D1100.10 BOOL  ; #2腔体机构关腔体氦检阀/关腔体抽气阀/关#2-1电池抽气阀（自动单检步）
D1100.11 BOOL  ; #2腔体机构关闭#2-1腔体阀/清氦判定（自动单检步）
D1100.12 BOOL  ; #2腔体机构打开#2-2腔体阀（自动单检步）
D1100.13 BOOL  ; #2腔体机构腔体抽气阀打开/延时开#2-2电池抽气阀（自动单检步）
D1100.14 BOOL  ; #2腔体机构关#2-2电池抽气阀（自动单检步）
D1100.15 BOOL  ; #2腔体机构开#2-2电池注氦阀（自动单检步）
D1101.00 BOOL  ; #2腔体机构关#2-2电池注氦阀（自动单检步）
D1101.01 BOOL  ; #2腔体机构（自动单检步）
D1101.02 BOOL  ; #2腔体机构开腔体氦检阀/延时关腔体抽气阀（自动单检步）
D1101.03 BOOL  ; #2腔体机构关腔体氦检阀（自动单检步）
D1101.04 BOOL  ; #2腔体机构开腔体#2-1阀（自动单检步）
D1101.05 BOOL  ; #2腔体机构开腔体抽真空阀/开电池抽真空阀（自动单检步）
D1101.06 BOOL  ; #2腔体机构关腔体抽真空阀/关电池抽真空阀（自动单检步）
D1101.07 BOOL  ; #2腔体机构清氦需求判定（自动单检步）
D1101.08 BOOL  ; #2腔体机构开腔体破真空阀/开电池破真空阀（自动单检步）
D1101.09 BOOL  ; #2腔体机构关腔体破真空阀/关电池破真空阀（自动单检步）
D1101.10 BOOL  ; #2腔体机构腔体顶升气缸下降（自动单检步）
D1101.11 BOOL  ; #2腔体机构腔体平移气缸到出料位（自动单检步）
D1101.12 BOOL  ; #2腔体机构腔体等待取料完成信号（自动单检步）
D1101.13 BOOL  ; #2腔体机构腔体平移气缸到上料位（自动单检步）
D1101.14 BOOL  ; #2腔体机构（自动单检步）
D1101.15 BOOL  ; #2腔体机构循环结束（自动单检步）
D1104 CHANNEL  ; #2腔体机构清氦步序号
D1104.00 BOOL  ; #2腔体机构自动开始（清氦步）
D1104.01 BOOL  ; #2腔体机构平移气缸到氦检位/数据初始化（清氦步）
D1104.02 BOOL  ; #2腔体机构腔体顶升气缸上升（清氦步）
D1104.03 BOOL  ; #2腔体机构氦检仪真空阀关闭（清氦步）
D1104.04 BOOL  ; #2腔体机构正压开腔体阀/负压关腔体阀/氦检阀打开
D1104.05 BOOL  ; #2腔体机构（清氦步）
D1104.06 BOOL  ; #2腔体机构腔体抽气阀打开/电池抽气阀打开（清氦步）
D1104.07 BOOL  ; #2腔体机构腔体抽气阀关闭/电池抽气阀关闭（清氦步）
D1104.08 BOOL  ; #2腔体机构（清氦步）
D1104.09 BOOL  ; #2腔体机构氦检清洁阀打开/电池破真空阀打开（清氦步）
D1104.10 BOOL  ; #2腔体机构氦检清洁阀关闭/电池破真空阀关闭（清氦步）
D1104.11 BOOL  ; #2腔体机构（清氦步）
D1104.12 BOOL  ; #2腔体机构清氦次数判定（清氦步）
D1104.13 BOOL  ; #2腔体机构（清氦步）
D1104.14 BOOL  ; #2腔体机构腔体抽气阀打开/电池抽气阀打开（清氦步）
D1104.15 BOOL  ; #2腔体机构关闭电池抽气阀（清氦步）
D1105.00 BOOL  ; #2腔体机构腔体氦检阀仪真空阀打开/延时关腔体抽气阀（清氦步）
D1105.01 BOOL  ; #2腔体机构（清氦步）
D1105.02 BOOL  ; #2腔体机构腔体氦检阀关闭（清氦步）
D1105.03 BOOL  ; #2腔体机构腔体抽气阀关闭/电池抽气阀关闭（清氦步）
D1105.04 BOOL  ; #2腔体机构是否需要重新清氦判定（清氦步）
D1105.05 BOOL  ; #2腔体机构（清氦步）
D1105.06 BOOL  ; #2腔体机构开腔体破真空阀/开电池破真空阀/开腔体阀（清氦步）
D1105.07 BOOL  ; #2腔体机构关腔体破真空阀/关电池破真空阀（清氦步）
D1105.08 BOOL  ; #2腔体机构（清氦步）
D1105.09 BOOL  ; #2腔体机构清氦完成标志（清氦步）
D1105.10 BOOL  ; #2腔体机构（清氦步）
D1105.11 BOOL  ; #2腔体机构腔体顶升气缸下降（清氦步）
D1105.12 BOOL  ; #2腔体机构腔体平移气缸到初始位（清氦步）
D1105.13 BOOL  ; #2腔体机构（清氦步）
D1105.14 BOOL  ; #2腔体机构（清氦步）
D1105.15 BOOL  ; #2腔体机构循环结束（清氦步）
D1107.00 BOOL  ; #2腔体机构复位（M）
D1107.01 BOOL  ; #2腔体关闭除破真空阀以外全部阀门（复位）
D1107.02 BOOL  ; #2腔体打开腔体阀门（复位）
D1107.03 BOOL  ; #2腔体破真空值未到达开破真空阀（复位）
D1107.04 BOOL  ; #2腔体破真空值到达关破真空阀（复位）
D1107.05 BOOL  ; #2腔体腔体顶升气缸下降（复位）
D1107.06 BOOL  ; #2腔体腔体平移气缸伸出（复位）
D1115.00 BOOL  ; #2腔体抽气阀打开允许（自检）
D1115.01 BOOL  ; #2腔体抽气阀打开需求（自检）
D1115.02 BOOL  ; #2腔体平移气缸在初始位（自检）
D1115.03 BOOL  ; #2腔体平移气缸在氦检位（自检）
D1115.04 BOOL  ; #2腔体真空泵开（自检）
D1115.05 BOOL  ; #2腔体平移气缸到初始位（自检）
D1115.06 BOOL  ; #2腔体平移气缸到氦检位（自检）
D1115.07 BOOL  ; #2腔体顶升气缸下降（自检）
D1115.08 BOOL  ; #2腔体顶升气缸上升（自检）
D1115.09 BOOL  ; #2腔体开抽真空阀（自检）
D1115.10 BOOL  ; #2腔体关抽真空阀（自检）
D1115.11 BOOL  ; #2腔体开破真空阀（自检）
D1115.12 BOOL  ; #2腔体关破真空阀（自检）
D1115.13 BOOL  ; #2腔体破真空阀状态（自检）
D1115.14 BOOL  ; #2腔体抽真空阀状态（自检）
D1117.00 BOOL  ; #2腔体机构标漏运行条件
D1117.01 BOOL  ; #2腔体机构标漏开始运行条件
D1117.02 BOOL  ; #2腔体机构标漏步进条件
D1117.15 BOOL  ; #2腔体机构标漏步进
D1118 CHANNEL  ; #2腔体标漏步序号
D1118.00 BOOL  ; #2腔体机构自动开始（标漏步）
D1118.01 BOOL  ; #2腔体机构（标漏步）
D1118.02 BOOL  ; #2腔体机构（标漏步）
D1118.03 BOOL  ; #2腔体机构（标漏步）
D1118.04 BOOL  ; #2腔体机构（标漏步）
D1118.05 BOOL  ; #2腔体机构（标漏步）
D1118.06 BOOL  ; #2腔体机构（标漏步）
D1118.07 BOOL  ; #2腔体机构开#2-1腔体阀（标漏步）
D1118.08 BOOL  ; #2腔体机构开#2腔抽气阀（标漏步）
D1118.09 BOOL  ; #2腔体机构关#2腔体抽气阀（标漏步）
D1118.10 BOOL  ; #2腔体机构（标漏步）
D1118.11 BOOL  ; #2腔体机构（标漏步）
D1118.12 BOOL  ; #2腔体机构开始#2-1氦检（标漏步）
D1118.13 BOOL  ; #2腔体机构关#2腔体氦检阀（标漏步）
D1118.14 BOOL  ; #2腔体机构关#2-1腔体阀（标漏步）
D1118.15 BOOL  ; #2腔体机构开#2-2腔体阀（标漏步）
D1119.00 BOOL  ; #2腔体机构开#2腔抽真空阀（标漏步）
D1119.01 BOOL  ; #2腔体机构关#2腔抽真空阀（标漏步）
D1119.02 BOOL  ; #2腔体机构（标漏步）
D1119.03 BOOL  ; #2腔体机构（标漏步）
D1119.04 BOOL  ; #2腔体机构开始#2-2氦检（标漏步）
D1119.05 BOOL  ; #2腔体机构关#2腔体氦检阀（标漏步）
D1119.06 BOOL  ; #2腔体机构关#2-2腔体阀（标漏步）
D1119.07 BOOL  ; #2腔体机构（标漏步）
D1119.08 BOOL  ; #2腔体机构（标漏步）
D1119.09 BOOL  ; #2腔体机构（标漏步）
D1119.10 BOOL  ; #2腔体机构（标漏步）
D1119.11 BOOL  ; #2腔体机构（标漏步）
D1119.12 BOOL  ; #2腔体机构（标漏步）
D1119.13 BOOL  ; #2腔体机构（标漏步）
D1119.14 BOOL  ; #2腔体机构跳转至#3腔标漏步（标漏步）
D1119.15 BOOL  ; #2腔体机构循环结束（标漏步）
D112 CHANNEL  ; 泄漏率（Pa.m3/s_Float）
D1120.00 BOOL  ; #3氦检机构初始位
D1120.05 BOOL  ; #3氦检机构停止标志
D1120.06 BOOL  ; #3氦检机构清料完成标志
D1120.07 BOOL  ; #3腔体机构异常标志
D1121.00 BOOL  ; #3腔体机构运行条件（自动步）
D1121.01 BOOL  ; #3腔体机构运行条件（自动单检步）
D1121.02 BOOL  ; #3腔体机构运行条件（清氦步）
D1122.00 BOOL  ; #3腔体机构平移气缸安全移动条件
D1122.12 BOOL  ; #3腔体机构腔体抽真空需求（测试）
D1122.13 BOOL  ; #3腔体机构正常清氦需求（正压测试）
D1122.14 BOOL  ; #3腔体氦检阀打开允许条件
D1122.15 BOOL  ; #3腔体机构腔体抽气阀打开允许
D1123.00 BOOL  ; #3腔体机构单步/自动循环运行中（总）
D1123.10 BOOL  ; $?St$Bk?_#[183] / #3腔体机构记忆清除(SW) / $?St$Bk?_#[183]
D1123.12 BOOL  ; #3腔体自检启动(SW)
D1123.13 BOOL  ; #3腔体自检停止(SW)
D1123.14 BOOL  ; #3腔体机构复位按钮（SW）
D1123.15 BOOL  ; #3腔体机构单步（SW）
D1124.00 BOOL  ; #3腔体机构单步运行中
D1124.01 BOOL  ; #3腔体机构单步/自动循环运行中（自动步）
D1124.02 BOOL  ; #3腔体机构自动循环运行中（自动单检步）
D1124.03 BOOL  ; #3腔体机构自动循环运行中（清氦步）
D1124.04 BOOL  ; #3-1腔体单腔自检(SW)
D1124.05 BOOL  ; #3-2腔体单腔自检(SW)
D1124.06 BOOL  ; #3腔体自检运行中
D1125.00 BOOL  ; #3腔体机构开始运行条件（自动步）
D1125.01 BOOL  ; #3腔体机构步进条件（自动步）
D1125.02 BOOL  ; #3腔体机构开始运行条件（自动单检步）
D1125.03 BOOL  ; #3腔体机构步进条件（自动单检步）
D1125.04 BOOL  ; #3腔体机构开始运行条件（清氦步）
D1125.05 BOOL  ; #3腔体机构步进条件（清氦步）
D1125.13 BOOL  ; #3腔体机构步进（清氦步）
D1125.14 BOOL  ; #3腔体机构步进（自动单检步）
D1125.15 BOOL  ; #3腔体机构步进（自动步）
D1126 CHANNEL  ; #3腔体机构自动步序号
D1126.00 BOOL  ; #3腔体机构自动开始（自动步）
D1126.01 BOOL  ; #3腔体机构平移气缸到氦检位/数据初始化（自动步）
D1126.02 BOOL  ; #3腔体机构腔体顶升气缸上升（自动步）
D1126.03 BOOL  ; #3腔体机构等待氦检阀打开条件及腔体抽气阀打开条件/开腔体阀（自动步）
D1126.04 BOOL  ; #3腔体机构（自动步）
D1126.05 BOOL  ; #3腔体机构腔体抽气阀打开/延时开电池抽气阀（自动步）
D1126.06 BOOL  ; #3腔体机构关电池抽气阀（自动步）
D1126.07 BOOL  ; #3腔体机构开电池注氦阀（自动步）
D1126.08 BOOL  ; #3腔体机构关电池注氦阀（自动步）
D1126.09 BOOL  ; #3腔体机构（自动步）
D1126.10 BOOL  ; #3腔体机构开腔体氦检阀/延时关腔体抽气阀（自动步）
D1126.11 BOOL  ; #3腔体机构（自动步）
D1126.12 BOOL  ; #3腔体机构关腔体氦检阀（自动步）
D1126.13 BOOL  ; #3腔体机构（自动步）
D1126.14 BOOL  ; #3腔体机构开腔体#3-1腔体阀/开腔体#3-2腔体阀（自动步）
D1126.15 BOOL  ; #3腔体机构开腔体抽真空阀/开电池抽真空阀（自动步）
D1127.00 BOOL  ; #3腔体机构关腔体抽真空阀/关电池抽真空阀/开腔体阀（自动步）
D1127.01 BOOL  ; #3腔体机构清氦需求判定（自动步）
D1127.02 BOOL  ; #3腔体机构开腔体破真空阀/开电池破真空阀（自动步）
D1127.03 BOOL  ; #3腔体机构关腔体破真空阀/关电池破真空阀（自动步）
D1127.04 BOOL  ; #3腔体机构复测需求判定（自动步）
D1127.05 BOOL  ; #3腔体机构（自动步）
D1127.06 BOOL  ; #3腔体机构腔体顶升气缸下降（自动步）
D1127.07 BOOL  ; #3腔体机构（自动步）
D1127.08 BOOL  ; #3腔体机构腔体平移气缸到出料位（自动步）
D1127.09 BOOL  ; #3腔体机构腔体等待取料完成信号（自动步）
D1127.10 BOOL  ; #3腔体机构（自动步）
D1127.11 BOOL  ; #3腔体机构平移气缸到上料位（自动步）
D1127.12 BOOL  ; #3腔体机构（自动步）
D1127.13 BOOL  ; #3腔体机构（自动步）
D1127.14 BOOL  ; #3腔体机构（自动步）
D1127.15 BOOL  ; #3腔体机构循环结束（自动步）
D1130 CHANNEL  ; #3腔体机构单检步序号
D1130.00 BOOL  ; #3腔体机构自动开始（自动单检步）
D1130.01 BOOL  ; #3腔体机构平移气缸到氦检位/数据初始化（自动单检步）
D1130.02 BOOL  ; #3腔体机构腔体顶升气缸上升（自动单检步）
D1130.03 BOOL  ; #3腔体机构关闭#3-2腔体阀（自动单检步）
D1130.04 BOOL  ; #3腔体机构腔体抽气阀打开/延时开#3-1电池抽气阀（自动单检步）
D1130.05 BOOL  ; #3腔体机构关#3-1电池抽气阀（自动单检步）
D1130.06 BOOL  ; #3腔体机构开#3-1电池注氦阀（自动单检步）
D1130.07 BOOL  ; #3腔体机构关#3-1电池注氦阀（自动单检步）
D1130.08 BOOL  ; #3腔体机构（自动单检步）
D1130.09 BOOL  ; #3腔体机构开腔体氦检阀/延时关腔体抽气阀（自动单检步）
D1130.10 BOOL  ; #3腔体机构关腔体氦检阀/关腔体抽气阀/关#3-1电池抽气阀（自动单检步）
D1130.11 BOOL  ; #3腔体机构关闭#3-1腔体阀/清氦判定（自动单检步）
D1130.12 BOOL  ; #3腔体机构打开#3-2腔体阀（自动单检步）
D1130.13 BOOL  ; #3腔体机构腔体抽气阀打开/延时开#3-2电池抽气阀（自动单检步）
D1130.14 BOOL  ; #3腔体机构关#3-2电池抽气阀（自动单检步）
D1130.15 BOOL  ; #3腔体机构开#3-2电池注氦阀（自动单检步）
D1131.00 BOOL  ; #3腔体机构关#3-2电池注氦阀（自动单检步）
D1131.01 BOOL  ; #3腔体机构（自动单检步）
D1131.02 BOOL  ; #3腔体机构开腔体氦检阀/延时关腔体抽气阀（自动单检步）
D1131.03 BOOL  ; #3腔体机构关腔体氦检阀（自动单检步）
D1131.04 BOOL  ; #3腔体机构开腔体#3-1阀（自动单检步）
D1131.05 BOOL  ; #3腔体机构开腔体抽真空阀/开电池抽真空阀（自动单检步）
D1131.06 BOOL  ; #3腔体机构关腔体抽真空阀/关电池抽真空阀（自动单检步）
D1131.07 BOOL  ; #3腔体机构清氦需求判定（自动单检步）
D1131.08 BOOL  ; #3腔体机构开腔体破真空阀/开电池破真空阀（自动单检步）
D1131.09 BOOL  ; #3腔体机构关腔体破真空阀/关电池破真空阀（自动单检步）
D1131.10 BOOL  ; #3腔体机构腔体顶升气缸下降（自动单检步）
D1131.11 BOOL  ; #3腔体机构腔体平移气缸到出料位（自动单检步）
D1131.12 BOOL  ; #3腔体机构腔体等待取料完成信号（自动单检步）
D1131.13 BOOL  ; #3腔体机构腔体平移气缸到上料位（自动单检步）
D1131.14 BOOL  ; #3腔体机构（自动单检步）
D1131.15 BOOL  ; #3腔体机构循环结束（自动单检步）
D1134 CHANNEL  ; #3腔体机构清氦步序号
D1134.00 BOOL  ; #3腔体机构自动开始（清氦步）
D1134.01 BOOL  ; #3腔体机构平移气缸到氦检位/数据初始化（清氦步）
D1134.02 BOOL  ; #3腔体机构腔体顶升气缸上升（清氦步）
D1134.03 BOOL  ; #3腔体机构氦检仪真空阀关闭（清氦步）
D1134.04 BOOL  ; #3腔体机构正压开腔体阀/负压关腔体阀/氦检阀打开
D1134.05 BOOL  ; #3腔体机构（清氦步）
D1134.06 BOOL  ; #3腔体机构腔体抽气阀打开/电池抽气阀打开（清氦步）
D1134.07 BOOL  ; #3腔体机构腔体抽气阀关闭/电池抽气阀关闭（清氦步）
D1134.08 BOOL  ; #3腔体机构（清氦步）
D1134.09 BOOL  ; #3腔体机构氦检清洁阀打开/电池破真空阀打开（清氦步）
D1134.10 BOOL  ; #3腔体机构氦检清洁阀关闭/电池破真空阀关闭（清氦步）
D1134.11 BOOL  ; #3腔体机构（清氦步）
D1134.12 BOOL  ; #3腔体机构清氦次数判定（清氦步）
D1134.13 BOOL  ; #3腔体机构（清氦步）
D1134.14 BOOL  ; #3腔体机构腔体抽气阀打开/电池抽气阀打开（清氦步）
D1134.15 BOOL  ; #3腔体机构关闭电池抽气阀（清氦步）
D1135.00 BOOL  ; #3腔体机构腔体氦检阀仪真空阀打开/延时关腔体抽气阀（清氦步）
D1135.01 BOOL  ; #3腔体机构（清氦步）
D1135.02 BOOL  ; #3腔体机构腔体氦检阀关闭（清氦步）
D1135.03 BOOL  ; #3腔体机构腔体抽气阀关闭/电池抽气阀关闭（清氦步）
D1135.04 BOOL  ; #3腔体机构是否需要重新清氦判定（清氦步）
D1135.05 BOOL  ; #3腔体机构（清氦步）
D1135.06 BOOL  ; #3腔体机构开腔体破真空阀/开电池破真空阀/开腔体阀（清氦步）
D1135.07 BOOL  ; #3腔体机构关腔体破真空阀/关电池破真空阀（清氦步）
D1135.08 BOOL  ; #3腔体机构（清氦步）
D1135.09 BOOL  ; #3腔体机构清氦完成标志（清氦步）
D1135.10 BOOL  ; #3腔体机构（清氦步）
D1135.11 BOOL  ; #3腔体机构腔体顶升气缸下降（清氦步）
D1135.12 BOOL  ; #3腔体机构腔体平移气缸到初始位（清氦步）
D1135.13 BOOL  ; #3腔体机构（清氦步）
D1135.14 BOOL  ; #3腔体机构（清氦步）
D1135.15 BOOL  ; #3腔体机构循环结束（清氦步）
D1137.00 BOOL  ; #3腔体机构复位（M）
D1137.01 BOOL  ; #3腔体关闭除破真空阀以外全部阀门（复位）
D1137.02 BOOL  ; #3腔体打开腔体阀门（复位）
D1137.03 BOOL  ; #3腔体破真空值未到达开破真空阀（复位）
D1137.04 BOOL  ; #3腔体破真空值到达关破真空阀（复位）
D1137.05 BOOL  ; #3腔体腔体顶升气缸下降（复位）
D1137.06 BOOL  ; #3腔体腔体平移气缸伸出（复位）
D114 CHANNEL  ; 泄漏率（Pa.m3/s_Float_指数）
D1143.00 BOOL  ; 进料机械手执行清料动作
D1145.00 BOOL  ; #3腔体抽气阀打开允许（自检）
D1145.01 BOOL  ; #3腔体抽气阀打开需求（自检）
D1145.02 BOOL  ; #3腔体平移气缸在初始位（自检）
D1145.03 BOOL  ; #3腔体平移气缸在氦检位（自检）
D1145.04 BOOL  ; #3腔体真空泵开（自检）
D1145.05 BOOL  ; #3腔体平移气缸到初始位（自检）
D1145.06 BOOL  ; #3腔体平移气缸到氦检位（自检）
D1145.07 BOOL  ; #3腔体顶升气缸下降（自检）
D1145.08 BOOL  ; #3腔体顶升气缸上升（自检）
D1145.09 BOOL  ; #3腔体开抽真空阀（自检）
D1145.10 BOOL  ; #3腔体关抽真空阀（自检）
D1145.11 BOOL  ; #3腔体开破真空阀（自检）
D1145.12 BOOL  ; #3腔体关破真空阀（自检）
D1145.13 BOOL  ; #3腔体破真空阀状态（自检）
D1145.14 BOOL  ; #3腔体抽真空阀状态（自检）
D1147.00 BOOL  ; #3腔体机构标漏运行条件
D1147.01 BOOL  ; #3腔体机构标漏开始运行条件
D1147.02 BOOL  ; #3腔体机构标漏步进条件
D1147.15 BOOL  ; #3腔体机构标漏步进
D1148 CHANNEL  ; #3腔体标漏步序号
D1148.00 BOOL  ; #3腔体机构自动开始（标漏步）
D1148.01 BOOL  ; #3腔体机构（标漏步）
D1148.02 BOOL  ; #3腔体机构（标漏步）
D1148.03 BOOL  ; #3腔体机构（标漏步）
D1148.04 BOOL  ; #3腔体机构（标漏步）
D1148.05 BOOL  ; #3腔体机构（标漏步）
D1148.06 BOOL  ; #3腔体机构（标漏步）
D1148.07 BOOL  ; #3腔体机构开#3-1腔体阀（标漏步）
D1148.08 BOOL  ; #3腔体机构开#3腔抽气阀（标漏步）
D1148.09 BOOL  ; #3腔体机构关#3腔体抽气阀（标漏步）
D1148.10 BOOL  ; #3腔体机构（标漏步）
D1148.11 BOOL  ; #3腔体机构（标漏步）
D1148.12 BOOL  ; #3腔体机构开始#3-1氦检（标漏步）
D1148.13 BOOL  ; #3腔体机构关#3腔体氦检阀（标漏步）
D1148.14 BOOL  ; #3腔体机构关#3-1腔体阀（标漏步）
D1148.15 BOOL  ; #3腔体机构开#3-2腔体阀（标漏步）
D1149.00 BOOL  ; #3腔体机构开#3腔抽真空阀（标漏步）
D1149.01 BOOL  ; #3腔体机构关#3腔抽真空阀（标漏步）
D1149.02 BOOL  ; #3腔体机构（标漏步）
D1149.03 BOOL  ; #3腔体机构（标漏步）
D1149.04 BOOL  ; #3腔体机构开始#3-2氦检（标漏步）
D1149.05 BOOL  ; #3腔体机构关#3腔体氦检阀（标漏步）
D1149.06 BOOL  ; #3腔体机构关#3-2腔体阀（标漏步）
D1149.07 BOOL  ; #3腔体机构开所有腔体总阀（标漏步）
D1149.08 BOOL  ; #3腔体机构开所有腔体破真空阀（标漏步）
D1149.09 BOOL  ; #3腔体机构关所有腔体破真空阀（标漏步）
D1149.10 BOOL  ; #3腔体机构所有顶升气缸下降（标漏步）
D1149.11 BOOL  ; #3腔体机构所有腔体平移气缸回初始位（标漏步）
D1149.12 BOOL  ; #3腔体机构关标漏阀（标漏步）
D1149.13 BOOL  ; #3腔体机构（标漏步）
D1149.14 BOOL  ; #3腔体机构（标漏步）
D1149.15 BOOL  ; #3腔体机构循环结束（标漏步）
D1150.00 BOOL  ; 出料伺服机构初始位
D1150.05 BOOL  ; 出料伺服机构停止标志
D1150.06 BOOL  ; 出料伺服机构清料完成标志
D1150.07 BOOL  ; 出料伺服机构异常标志
D1153.00 BOOL  ; 出料机械手执行清料动作
D1153.10 BOOL  ; 下料夹爪有料记忆清除（SW）
D1153.14 BOOL  ; 出料伺服机构复位按钮（SW）
D1156 CHANNEL  ; 下料模组自动流程
D1156.00 BOOL  ; 下料模组运行前检测
D1156.01 BOOL  ; 下料模组运行备用
D1156.02 BOOL  ; 下料x模组运行到对应下料位
D1156.03 BOOL  ; 下料Z模组运行前检测
D1156.04 BOOL  ; 下料Z模组运行
D1156.05 BOOL  ; 下料模组夹爪夹紧
D1156.06 BOOL  ; 下料模组运行备用
D1156.07 BOOL  ; 下料Z模组到待机位
D1156.08 BOOL  ; 等待数据校验完成
D1156.09 BOOL  ; 下料模组是否放全OK料检测
D1156.10 BOOL  ; 下料X模组到OK下料位
D1156.11 BOOL  ; 下料Z模组OK下降检测
D1156.12 BOOL  ; 下料Z模组到OK下料位
D1156.13 BOOL  ; 下料模组放全OK料开夹爪
D1156.14 BOOL  ; 下料Z模组到待机位
D1156.15 BOOL  ; *下料模组去腔体取料流程&全OK下料结束
D1158 CHANNEL  ; 下料模组全NG流程
D1158.00 BOOL  ; 下料模组全OK/NG料流程准备
D1158.01 BOOL  ; 下料模组放NG料：预留
D1158.02 BOOL  ; 下料模组放NG：预留
D1158.03 BOOL  ; 下料模组放NG料：出料X轴到NG缓存位/变距气缸缩回
D1158.04 BOOL  ; 预留
D1158.05 BOOL  ; 预留
D1158.06 BOOL  ; 预留
D1158.07 BOOL  ; 预留
D1158.08 BOOL  ; 下料模组放1#NG Z轴下降
D1158.09 BOOL  ; 下料模组开夹爪放NG料
D1158.10 BOOL  ; 下料Z模组放完1#NG回待机位
D1158.11 BOOL  ; 下料模组放双NG:放NG料完成，有腔体测试完成直接跳过，无腔体测试完成X轴返回待机位
D1158.12 BOOL  ; 下料模组放双NG备用
D1158.13 BOOL  ; 下料模组放双NG备用
D1158.14 BOOL  ; 下料模组放双NG备用
D1158.15 BOOL  ; 下料模组放双NG结束
D116 CHANNEL  ; 检漏口压力（Pa_Float）
D1160 CHANNEL  ; 下料模组（取）放1OK/1NG流程
D1160.00 BOOL  ; *下料模组（取）放1OK/1NG流程运行前检测
D1160.01 BOOL  ; 下料X模组到达对应X位置
D1160.02 BOOL  ; 下料Z模组下降前检测
D1160.03 BOOL  ; 下料Z模组下降放NG料
D1160.04 BOOL  ; 下料模组开NG夹爪
D1160.05 BOOL  ; 下料Z模组放完NG回待机位
D1160.06 BOOL  ; 下料模组放缓存OR取缓存
D1160.07 BOOL  ; 下料X模组到放缓存位
D1160.08 BOOL  ; 下料Z模组下降放缓存
D1160.09 BOOL  ; 下料模组放缓存开夹爪or夹紧
D1160.10 BOOL  ; 下料模组缓存有料检测
D1160.11 BOOL  ; 下料Z模组到待机位
D1160.12 BOOL  ; *下料模组（取）放1OK/1NG X轴到OK下料位
D1160.13 BOOL  ; *下料模组（取）放1OK/1NG流程备用
D1160.14 BOOL  ; *下料模组（取）放1OK/1NG流程备用
D1160.15 BOOL  ; *下料模组（取）放1OK/1NG流程结束
D1166 CHANNEL  ; 下料模组X/Z初始化
D1166.00 BOOL  ; 下料模组初始化准备
D1166.01 BOOL  ; 下料Z模组初始化
D1166.02 BOOL  ; 下料Z模组到待机位
D1166.03 BOOL  ; 下料X模组初始化
D1166.04 BOOL  ; 下料X模组到待机位
D1166.05 BOOL  ; 下料模组运行许可
D1166.06 BOOL  ; 下料模组初始化结束
D1168 CHANNEL  ; 下料模组手动跟踪联动
D1168.00 BOOL  ; 下料模组手动跟踪Z回待机位
D1168.01 BOOL  ; 下料模组手动跟踪X到对应位置
D1168.02 BOOL  ; 下料Z轴手动下降前安全判定
D1168.03 BOOL  ; 下料Z模组手动下降
D1168.04 BOOL  ; 下料X/Z模组跟踪联动需求清除
D1168.05 BOOL  ; 下料X/Z模组手动联动结束
D1170.00 BOOL  ; #4氦检机构初始位
D1170.05 BOOL  ; #4氦检机构停止标志
D1170.06 BOOL  ; #4氦检机构清料完成标志
D1170.07 BOOL  ; #4腔体机构异常标志
D1171.00 BOOL  ; #4腔体机构运行条件（自动步）
D1171.01 BOOL  ; #4腔体机构运行条件（自动单检步）
D1171.02 BOOL  ; #4腔体机构运行条件（清氦步）
D1172.00 BOOL  ; #4腔体机构平移气缸安全移动条件
D1172.12 BOOL  ; #4腔体机构腔体抽真空需求（测试）
D1172.13 BOOL  ; #4腔体机构正常清氦需求（正压测试）
D1172.14 BOOL  ; #4腔体氦检阀打开允许条件
D1172.15 BOOL  ; #4腔体机构腔体抽气阀打开允许
D1173.00 BOOL  ; #4腔体机构单步/自动循环运行中（总）
D1173.10 BOOL  ; #4腔体机构记忆清除(SW)
D1173.11 BOOL  ; #4腔体标漏(SW)
D1173.12 BOOL  ; #4腔体自检启动(SW)
D1173.13 BOOL  ; #4腔体自检停止(SW)
D1173.14 BOOL  ; #4腔体机构复位按钮（SW）
D1173.15 BOOL  ; #4腔体机构单步（SW）
D1174.00 BOOL  ; #4腔体机构单步运行中
D1174.01 BOOL  ; #4腔体机构单步/自动循环运行中（自动步）
D1174.02 BOOL  ; #4腔体机构自动循环运行中（自动单检步）
D1174.03 BOOL  ; #4腔体机构自动循环运行中（清氦步）
D1174.04 BOOL  ; #4-1腔体单腔自检(SW)
D1174.05 BOOL  ; #4-2腔体单腔自检(SW)
D1174.06 BOOL  ; #4腔体自检运行中
D1174.10 BOOL  ; #4腔体机构单步运行条件
D1175.00 BOOL  ; #4腔体机构开始运行条件（自动步）
D1175.01 BOOL  ; #4腔体机构步进条件（自动步）
D1175.02 BOOL  ; #4腔体机构开始运行条件（自动单检步）
D1175.03 BOOL  ; #4腔体机构步进条件（自动单检步）
D1175.04 BOOL  ; #4腔体机构开始运行条件（清氦步）
D1175.05 BOOL  ; #4腔体机构步进条件（清氦步）
D1175.13 BOOL  ; #4腔体机构步进（清氦步）
D1175.14 BOOL  ; #4腔体机构步进（自动单检步）
D1175.15 BOOL  ; #4腔体机构步进（自动步）
D1176 CHANNEL  ; #4腔体机构自动步序号
D1176.00 BOOL  ; #4腔体机构自动开始（自动步）
D1176.01 BOOL  ; #4腔体机构平移气缸到氦检位/数据初始化（自动步）
D1176.02 BOOL  ; #4腔体机构腔体顶升气缸上升（自动步）
D1176.03 BOOL  ; #4腔体机构等待氦检阀打开条件及腔体抽气阀打开条件/开腔体阀（自动步）
D1176.04 BOOL  ; #4腔体机构（自动步）
D1176.05 BOOL  ; #4腔体机构腔体抽气阀打开/延时开电池抽气阀（自动步）
D1176.06 BOOL  ; #4腔体机构关电池抽气阀（自动步）
D1176.07 BOOL  ; #4腔体机构开电池注氦阀（自动步）
D1176.08 BOOL  ; #4腔体机构关电池注氦阀（自动步）
D1176.09 BOOL  ; #4腔体机构（自动步）
D1176.10 BOOL  ; #4腔体机构开腔体氦检阀/延时关腔体抽气阀（自动步）
D1176.11 BOOL  ; #4腔体机构（自动步）
D1176.12 BOOL  ; #4腔体机构关腔体氦检阀（自动步）
D1176.13 BOOL  ; #4腔体机构（自动步）
D1176.14 BOOL  ; #4腔体机构开腔体#4-1腔体阀/开腔体#4-2腔体阀（自动步）
D1176.15 BOOL  ; #4腔体机构开腔体抽真空阀/开电池抽真空阀（自动步）
D1177.00 BOOL  ; #4腔体机构关腔体抽真空阀/关电池抽真空阀/开腔体阀（自动步）
D1177.01 BOOL  ; #4腔体机构清氦需求判定（自动步）
D1177.02 BOOL  ; #4腔体机构开腔体破真空阀/开电池破真空阀（自动步）
D1177.03 BOOL  ; #4腔体机构关腔体破真空阀/关电池破真空阀（自动步）
D1177.04 BOOL  ; #4腔体机构复测需求判定（自动步）
D1177.05 BOOL  ; #4腔体机构（自动步）
D1177.06 BOOL  ; #4腔体机构腔体顶升气缸下降（自动步）
D1177.07 BOOL  ; #4腔体机构（自动步）
D1177.08 BOOL  ; #4腔体机构腔体平移气缸到出料位（自动步）
D1177.09 BOOL  ; #4腔体机构腔体等待取料完成信号（自动步）
D1177.10 BOOL  ; #4腔体机构（自动步）
D1177.11 BOOL  ; #4腔体机构平移气缸到上料位（自动步）
D1177.12 BOOL  ; #4腔体机构（自动步）
D1177.13 BOOL  ; #4腔体机构（自动步）
D1177.14 BOOL  ; #4腔体机构（自动步）
D1177.15 BOOL  ; #4腔体机构循环结束（自动步）
D118 CHANNEL  ; 检漏口压力（Pa_Float_指数）
D1180 CHANNEL  ; #4腔体机构单检步序号
D1180.00 BOOL  ; #4腔体机构自动开始（自动单检步）
D1180.01 BOOL  ; #4腔体机构平移气缸到氦检位/数据初始化（自动单检步）
D1180.02 BOOL  ; #4腔体机构腔体顶升气缸上升（自动单检步）
D1180.03 BOOL  ; #4腔体机构关闭#4-2腔体阀（自动单检步）
D1180.04 BOOL  ; #4腔体机构腔体抽气阀打开/延时开#4-1电池抽气阀（自动单检步）
D1180.05 BOOL  ; #4腔体机构关#4-1电池抽气阀（自动单检步）
D1180.06 BOOL  ; #4腔体机构开#4-1电池注氦阀（自动单检步）
D1180.07 BOOL  ; #4腔体机构关#4-1电池注氦阀（自动单检步）
D1180.08 BOOL  ; #4腔体机构（自动单检步）
D1180.09 BOOL  ; #4腔体机构开腔体氦检阀/延时关腔体抽气阀（自动单检步）
D1180.10 BOOL  ; #4腔体机构关腔体氦检阀/关腔体抽气阀/关#4-1电池抽气阀（自动单检步）
D1180.11 BOOL  ; #4腔体机构关闭#4-1腔体阀/清氦判定（自动单检步）
D1180.12 BOOL  ; #4腔体机构打开#4-2腔体阀（自动单检步）
D1180.13 BOOL  ; #4腔体机构腔体抽气阀打开/延时开#4-2电池抽气阀（自动单检步）
D1180.14 BOOL  ; #4腔体机构关#4-2电池抽气阀（自动单检步）
D1180.15 BOOL  ; #4腔体机构开#4-2电池注氦阀（自动单检步）
D1181.00 BOOL  ; #4腔体机构关#4-2电池注氦阀（自动单检步）
D1181.01 BOOL  ; #4腔体机构（自动单检步）
D1181.02 BOOL  ; #4腔体机构开腔体氦检阀/延时关腔体抽气阀（自动单检步）
D1181.03 BOOL  ; #4腔体机构关腔体氦检阀（自动单检步）
D1181.04 BOOL  ; #4腔体机构开腔体#4-1阀（自动单检步）
D1181.05 BOOL  ; #4腔体机构开腔体抽真空阀/开电池抽真空阀（自动单检步）
D1181.06 BOOL  ; #4腔体机构关腔体抽真空阀/关电池抽真空阀（自动单检步）
D1181.07 BOOL  ; #4腔体机构清氦需求判定（自动单检步）
D1181.08 BOOL  ; #4腔体机构开腔体破真空阀/开电池破真空阀（自动单检步）
D1181.09 BOOL  ; #4腔体机构关腔体破真空阀/关电池破真空阀（自动单检步）
D1181.10 BOOL  ; #4腔体机构腔体顶升气缸下降（自动单检步）
D1181.11 BOOL  ; #4腔体机构腔体平移气缸到出料位（自动单检步）
D1181.12 BOOL  ; #4腔体机构腔体等待取料完成信号（自动单检步）
D1181.13 BOOL  ; #4腔体机构腔体平移气缸到上料位（自动单检步）
D1181.14 BOOL  ; #4腔体机构（自动单检步）
D1181.15 BOOL  ; #4腔体机构循环结束（自动单检步）
D1184 CHANNEL  ; #4腔体机构清氦步序号
D1184.00 BOOL  ; #4腔体机构自动开始（清氦步）
D1184.01 BOOL  ; #4腔体机构平移气缸到氦检位/数据初始化（清氦步）
D1184.02 BOOL  ; #4腔体机构腔体顶升气缸上升（清氦步）
D1184.03 BOOL  ; #4腔体机构氦检仪真空阀关闭（清氦步）
D1184.04 BOOL  ; #4腔体机构正压开腔体阀/负压关腔体阀/氦检阀打开
D1184.05 BOOL  ; #4腔体机构（清氦步）
D1184.06 BOOL  ; #4腔体机构腔体抽气阀打开/电池抽气阀打开（清氦步）
D1184.07 BOOL  ; #4腔体机构腔体抽气阀关闭/电池抽气阀关闭（清氦步）
D1184.08 BOOL  ; #4腔体机构（清氦步）
D1184.09 BOOL  ; #4腔体机构氦检清洁阀打开/电池破真空阀打开（清氦步）
D1184.10 BOOL  ; #4腔体机构氦检清洁阀关闭/电池破真空阀关闭（清氦步）
D1184.11 BOOL  ; #4腔体机构（清氦步）
D1184.12 BOOL  ; #4腔体机构清氦次数判定（清氦步）
D1184.13 BOOL  ; #4腔体机构（清氦步）
D1184.14 BOOL  ; #4腔体机构腔体抽气阀打开/电池抽气阀打开（清氦步）
D1184.15 BOOL  ; #4腔体机构关闭电池抽气阀（清氦步）
D1185.00 BOOL  ; #4腔体机构腔体氦检阀仪真空阀打开/延时关腔体抽气阀（清氦步）
D1185.01 BOOL  ; #4腔体机构（清氦步）
D1185.02 BOOL  ; #4腔体机构腔体氦检阀关闭（清氦步）
D1185.03 BOOL  ; #4腔体机构腔体抽气阀关闭/电池抽气阀关闭（清氦步）
D1185.04 BOOL  ; #4腔体机构是否需要重新清氦判定（清氦步）
D1185.05 BOOL  ; #4腔体机构（清氦步）
D1185.06 BOOL  ; #4腔体机构开腔体破真空阀/开电池破真空阀/开腔体阀（清氦步）
D1185.07 BOOL  ; #4腔体机构关腔体破真空阀/关电池破真空阀（清氦步）
D1185.08 BOOL  ; #4腔体机构（清氦步）
D1185.09 BOOL  ; #4腔体机构清氦完成标志（清氦步）
D1185.10 BOOL  ; #4腔体机构（清氦步）
D1185.11 BOOL  ; #4腔体机构腔体顶升气缸下降（清氦步）
D1185.12 BOOL  ; #4腔体机构腔体平移气缸到初始位（清氦步）
D1185.13 BOOL  ; #4腔体机构（清氦步）
D1185.14 BOOL  ; #4腔体机构（清氦步）
D1185.15 BOOL  ; #4腔体机构循环结束（清氦步）
D1187.00 BOOL  ; #4腔体机构复位（M）
D1187.01 BOOL  ; #4腔体关闭除破真空阀以外全部阀门（复位）
D1187.02 BOOL  ; #4腔体打开腔体阀门（复位）
D1187.03 BOOL  ; #4腔体破真空值未到达开破真空阀（复位）
D1187.04 BOOL  ; #4腔体破真空值到达关破真空阀（复位）
D1187.05 BOOL  ; #4腔体腔体顶升气缸下降（复位）
D1187.06 BOOL  ; #4腔体腔体平移气缸伸出（复位）
D1195.00 BOOL  ; #4腔体抽气阀打开允许（自检）
D1195.01 BOOL  ; #4腔体抽气阀打开需求（自检）
D1195.02 BOOL  ; #4腔体平移气缸在初始位（自检）
D1195.03 BOOL  ; #4腔体平移气缸在氦检位（自检）
D1195.04 BOOL  ; #4腔体真空泵开（自检）
D1195.05 BOOL  ; #4腔体平移气缸到初始位（自检）
D1195.06 BOOL  ; #4腔体平移气缸到氦检位（自检）
D1195.07 BOOL  ; #4腔体顶升气缸下降（自检）
D1195.08 BOOL  ; #4腔体顶升气缸上升（自检）
D1195.09 BOOL  ; #4腔体开抽真空阀（自检）
D1195.10 BOOL  ; #4腔体关抽真空阀（自检）
D1195.11 BOOL  ; #4腔体开破真空阀（自检）
D1195.12 BOOL  ; #4腔体关破真空阀（自检）
D1195.13 BOOL  ; #4腔体破真空阀状态（自检）
D1195.14 BOOL  ; #4腔体抽真空阀状态（自检）
D1195.15 BOOL  ; （自检）
D1197.00 BOOL  ; #4腔体机构标漏运行条件
D1197.01 BOOL  ; #4腔体机构标漏开始运行条件
D1197.02 BOOL  ; #4腔体机构标漏步进条件
D1197.03 BOOL  ; #4腔体机构标漏运行中
D1197.15 BOOL  ; #4腔体机构标漏步进
D1198 CHANNEL  ; #4腔体标漏步序号
D1198.00 BOOL  ; #4腔体机构自动开始（标漏步）
D1198.01 BOOL  ; #4腔体机构（标漏步）
D1198.02 BOOL  ; #4腔体机构（标漏步）
D1198.03 BOOL  ; #4腔体机构（标漏步）
D1198.04 BOOL  ; #4腔体机构（标漏步）
D1198.05 BOOL  ; #4腔体机构（标漏步）
D1198.06 BOOL  ; #4腔体机构（标漏步）
D1198.07 BOOL  ; #4腔体机构开#4-1腔体阀（标漏步）
D1198.08 BOOL  ; #4腔体机构开#4腔抽气阀（标漏步）
D1198.09 BOOL  ; #4腔体机构关#4腔体抽气阀（标漏步）
D1198.10 BOOL  ; #4腔体机构（标漏步）
D1198.11 BOOL  ; #4腔体机构（标漏步）
D1198.12 BOOL  ; #4腔体机构开始#4-1氦检（标漏步）
D1198.13 BOOL  ; #4腔体机构关#4腔体氦检阀（标漏步）
D1198.14 BOOL  ; #4腔体机构关#4-1腔体阀（标漏步）
D1198.15 BOOL  ; #4腔体机构开#4-2腔体阀（标漏步）
D1199.00 BOOL  ; #4腔体机构开#4腔抽真空阀（标漏步）
D1199.01 BOOL  ; #4腔体机构关#4腔抽真空阀（标漏步）
D1199.02 BOOL  ; #4腔体机构（标漏步）
D1199.03 BOOL  ; #4腔体机构（标漏步）
D1199.04 BOOL  ; #4腔体机构开始#4-2氦检（标漏步）
D1199.05 BOOL  ; #4腔体机构关#4腔体氦检阀（标漏步）
D1199.06 BOOL  ; #4腔体机构关#4-2腔体阀（标漏步）
D1199.07 BOOL  ; #4腔体机构开所有腔体总阀（标漏步）
D1199.08 BOOL  ; #4腔体机构开所有腔体破真空阀（标漏步）
D1199.09 BOOL  ; #4腔体机构关所有腔体破真空阀（标漏步）
D1199.10 BOOL  ; #4腔体机构所有顶升气缸下降（标漏步）
D1199.11 BOOL  ; #4腔体机构所有腔体平移气缸回初始位（标漏步）
D1199.12 BOOL  ; #4腔体机构（标漏步）
D1199.13 BOOL  ; #4腔体机构（标漏步）
D1199.14 BOOL  ; #4腔体机构（标漏步）
D1199.15 BOOL  ; #4腔体机构循环结束（标漏步）
D120 CHANNEL  ; 稳定漏率（Pa.m3/s_Float）
D1200.00 BOOL  ; 复测移载机构：初始位
D1200.05 BOOL  ; 复测移载机构：停止标志
D1200.06 BOOL  ; 氦检移载机构：清料完成标志
D1200.07 BOOL  ; 复测移载机构：异常标志
D1201.00 BOOL  ; 复测移载机构：运行条件（取/放待测料步）
D1201.01 BOOL  ; 复测移载机构：运行条件（取/放已测料步）
D1201.02 BOOL  ; $?St$Bk?_#[184] / 复测移载机构：运行条件（缓存步） / $?St$Bk?_#[184]
D1202.00 BOOL  ; 复测移载机构：移载伺服X轴移动条件
D1202.01 BOOL  ; 复测移载机构：移载伺服Z轴移动条件
D1202.02 BOOL  ; 允许出料机械手到复测取放料位
D1202.03 BOOL  ; 复测移载机构：缓存拨料气缸移动条件
D1202.15 BOOL  ; 复测移载机构：正常腔体待料条件(启动复测)
D1203.00 BOOL  ; 复测移载机构：单步/自动循环运行中（总）
D1203.10 BOOL  ; 复测移载机构：夹爪记忆清除(SW)
D1203.11 BOOL  ; 复测移载机构：缓存位记忆清除(SW)
D1203.12 BOOL  ; 复测移载机构：配对位记忆清除(SW)
D1203.14 BOOL  ; 复测移载机构：复位按钮（SW）
D1203.15 BOOL  ; 复测移载机构：单步（SW）
D1204.00 BOOL  ; 复测移载机构：单步运行中
D1204.01 BOOL  ; 复测移载机构：单步/自动循环运行中（取/放待测料步）
D1204.02 BOOL  ; 复测移载机构：单步/自动循环运行中（取/放已测料步）
D1205.00 BOOL  ; 复测移载机构：开始运行条件（取/放待测料步）
D1205.01 BOOL  ; 复测移载机构：步进条件（取/放待测料步）
D1205.02 BOOL  ; 复测移载机构：开始运行条件（取/放已测料步）
D1205.03 BOOL  ; 复测移载机构：步进条件（取/放已测料步）
D1205.04 BOOL  ; 复测移载机构：开始运行条件（缓存步）
D1205.05 BOOL  ; $?St$Bk?_#[185] / 复测移载机构：步进条件（缓存步） / $?St$Bk?_#[185]
D1205.13 BOOL  ; 复测移载机构：步进（缓存步）
D1205.14 BOOL  ; 复测移载机构：步进（取/放待测料步）
D1205.15 BOOL  ; 复测移载机构：步进（取/放已测料步）
D1206 CHANNEL  ; 复测移载机构：取/放待测料步序号
D1206.00 BOOL  ; 复测移载机构：自动开始（取/放待测料步）
D1206.01 BOOL  ; 复测移载机构：预留（取/放待测料步）
D1206.02 BOOL  ; 复测移载机构：复测移载伺服X轴判断取料位置（取/放待测料步）
D1206.03 BOOL  ; 复测移载机构：预留（取/放待测料步）
D1206.04 BOOL  ; 复测移载机构：复测移载伺服Z轴在取料位下降（取/放待测料步）
D1206.05 BOOL  ; 复测移载机构：预留（取/放待测料步）
D1206.06 BOOL  ; 复测移载机构：复测移载机械手夹爪夹紧（取/放待测料步）
D1206.07 BOOL  ; 复测移载机构：预留（取/放待测料步）
D1206.08 BOOL  ; 复测移载机构：复测移载伺服Z轴取料完成回待机位（取/放待测料步）
D1206.09 BOOL  ; 复测移载机构：预留（取/放待测料步）
D1206.10 BOOL  ; 复测移载机构：复测移载伺服X轴去腔体位（取/放待测料步）
D1206.11 BOOL  ; 复测移载机构：预留（取/放待测料步）
D1206.12 BOOL  ; 复测移载机构：复测移载伺服Z轴在腔体位置下降（取/放待测料步）
D1206.13 BOOL  ; 复测移载机构：预留（取/放待测料步）
D1206.14 BOOL  ; 复测移载机构：复测移载机械手夹爪松开（取/放待测料步）
D1206.15 BOOL  ; 复测移载机构：预留（取/放待测料步）
D1207.00 BOOL  ; 复测移载机构：预留（取/放待测料步）
D1207.01 BOOL  ; 复测移载机构：复测移载伺服Z轴放料完成回待机位（取/放待测料步）
D1207.02 BOOL  ; 复测移载机构：预留（取/放待测料步）
D1207.03 BOOL  ; 复测移载机构：预留（取/放待测料步）
D1207.04 BOOL  ; 复测移载机构：复测移载伺服X轴放料完成回待机位（取/放待测料步）
D1207.05 BOOL  ; 复测移载机构：预留（取/放待测料步）
D1207.06 BOOL  ; 复测移载机构：预留（取/放待测料步）
D1207.07 BOOL  ; 复测移载机构：预留（取/放待测料步）
D1207.08 BOOL  ; 复测移载机构：预留（取/放待测料步）
D1207.09 BOOL  ; 复测移载机构：预留（取/放待测料步）
D1207.10 BOOL  ; 复测移载机构：预留（取/放待测料步）
D1207.11 BOOL  ; 复测移载机构：预留（取/放待测料步）
D1207.12 BOOL  ; 复测移载机构：预留（取/放待测料步）
D1207.13 BOOL  ; 复测移载机构：预留（取/放待测料步）
D1207.14 BOOL  ; 复测移载机构：预留（取/放待测料步）
D1207.15 BOOL  ; 复测移载机构：循环结束（取/放待测料步）
D1210 CHANNEL  ; 复测移载机构：取/放已测料步序号
D1210.00 BOOL  ; 复测移载机构：自动开始（取/放已测料步）
D1210.01 BOOL  ; 复测移载机构：预留（取/放已测料步）
D1210.02 BOOL  ; 复测移载机构：预留（取/放已测料步）
D1210.03 BOOL  ; 复测移载机构：预留（取/放已测料步）
D1210.04 BOOL  ; 复测移载机构：复测移载伺服X轴去腔体位取料（取/放已测料步）
D1210.05 BOOL  ; 复测移载机构：预留（取/放已测料步）
D1210.06 BOOL  ; 复测移载机构：复测移载伺服Z轴下降至腔体位取料（取/放已测料步）
D1210.07 BOOL  ; 复测移载机构：预留（取/放已测料步）
D1210.08 BOOL  ; 复测移载机构：预留（取/放已测料步）
D1210.09 BOOL  ; 复测移载机构：复测移载机械手夹爪夹紧（取/放已测料步）
D1210.10 BOOL  ; 复测移载机构：预留（取/放已测料步）
D1210.11 BOOL  ; 复测移载机构：复测移载伺服Z轴取料完成回待机位（取/放已测料步）
D1210.12 BOOL  ; 复测移载机构：预留（取/放已测料步）
D1210.13 BOOL  ; 复测移载机构：预留（取/放已测料步）
D1210.14 BOOL  ; 复测移载机构：复测移载伺服X轴判断放料位置（取/放已测料步）
D1210.15 BOOL  ; 复测移载机构：预留（取/放已测料步）
D1211.00 BOOL  ; 复测移载机构：复测移载伺服Z轴在放料位下降（取/放已测料步）
D1211.01 BOOL  ; 复测移载机构：预留（取/放已测料步）
D1211.02 BOOL  ; 复测移载机构：复测移载机械手夹爪松开放料（取/放已测料步）
D1211.03 BOOL  ; 复测移载机构：预留（取/放已测料步）
D1211.04 BOOL  ; 复测移载机构：复测移载伺服Z轴放料完成回待机位（取/放已测料步）
D1211.05 BOOL  ; 复测移载机构：预留（取/放已测料步）
D1211.06 BOOL  ; 复测移载机构：预留（取/放已测料步）
D1211.07 BOOL  ; 复测移载机构：复测移载伺服X轴判断是否继续取待测料（取/放已测料步）
D1211.08 BOOL  ; 复测移载机构：预留（取/放已测料步）
D1211.09 BOOL  ; 复测移载机构：预留（取/放已测料步）
D1211.10 BOOL  ; 复测移载机构：预留（取/放已测料步）
D1211.11 BOOL  ; 复测移载机构：预留（取/放已测料步）
D1211.12 BOOL  ; 复测移载机构：预留（取/放已测料步）
D1211.13 BOOL  ; 复测移载机构：预留（取/放已测料步）
D1211.14 BOOL  ; 复测移载机构：预留（取/放已测料步）
D1211.15 BOOL  ; 复测移载机构：循环结束（取/放已测料步）
D1214 CHANNEL  ; 复测缓存机构：缓存步序号
D1214.00 BOOL  ; 复测移载机构：自动开始（缓存步）
D1214.01 BOOL  ; 复测移载机构：预留（缓存步）
D1214.02 BOOL  ; 复测移载机构：判定缓存类型（缓存步）
D1214.03 BOOL  ; 复测移载机构：预留（缓存步）
D1214.04 BOOL  ; 复测移载机构：缓存顶升气缸上升（缓存步）
D1214.05 BOOL  ; 复测移载机构：缓存拨料气缸伸出（缓存步）
D1214.06 BOOL  ; 复测移载机构：预留（缓存步）
D1214.07 BOOL  ; 复测移载机构：预留（缓存步）
D1214.08 BOOL  ; 复测移载机构：预留（缓存步）
D1214.09 BOOL  ; 复测移载机构：预留（缓存步）
D1214.10 BOOL  ; 复测移载机构：缓存顶升气缸下降（缓存步）
D1214.11 BOOL  ; 复测移载机构：缓存拨料气缸缩回（缓存步）
D1214.12 BOOL  ; 复测移载机构：预留（缓存步）
D1214.13 BOOL  ; 复测移载机构：预留（缓存步）
D1214.14 BOOL  ; 复测移载机构：预留（缓存步）
D1214.15 BOOL  ; 复测移载机构：循环结束（缓存步）
D1215.00 BOOL  ; 复测移载机构：自动开始（缓存步）
D1215.01 BOOL  ; 复测移载机构：预留（缓存步）
D1215.02 BOOL  ; 复测移载机构：预留（缓存步）
D1215.03 BOOL  ; 复测移载机构：缓存拨料气缸伸出（缓存步）
D1215.04 BOOL  ; 复测移载机构：缓存顶升气缸伸出（缓存步）
D1215.05 BOOL  ; 复测移载机构：缓存拨料气缸缩回（缓存步）
D1215.06 BOOL  ; 复测移载机构：预留（缓存步）
D1215.07 BOOL  ; 复测移载机构：预留（缓存步）
D1215.08 BOOL  ; 复测移载机构：预留（缓存步）
D1215.09 BOOL  ; 复测移载机构：预留（缓存步）
D1215.10 BOOL  ; 复测移载机构：预留（缓存步）
D1215.11 BOOL  ; 复测移载机构：缓存顶升气缸下降（缓存步）
D1215.12 BOOL  ; 复测移载机构：预留（缓存步）
D1215.13 BOOL  ; 复测移载机构：预留（缓存步）
D1215.14 BOOL  ; 复测移载机构：预留（缓存步）
D1215.15 BOOL  ; 复测移载机构：循环结束（缓存步）
D1217.00 BOOL  ; 复测移载机构：复位（M）
D1217.01 BOOL  ; 复测移载伺服Z轴回原点（复位）
D1217.02 BOOL  ; 复测移载伺服Z轴回待机位（复位）
D1217.03 BOOL  ; 复测移载伺服X轴回原点（复位）
D1217.04 BOOL  ; 复测移载伺服X轴回待机位（复位）
D1217.05 BOOL  ; 复测移载机构：复测缓存拨料气缸回初始位
D1217.06 BOOL  ; 复测缓存机构：复测缓存顶升气缸下降
D122 CHANNEL  ; 稳定漏率（Pa.m3/s_Float_指数）
D1230.00 BOOL  ; 复检腔体机构：初始位
D1230.05 BOOL  ; 复检腔体机构：停止标志
D1230.06 BOOL  ; 复检腔体机构：清料完成标志
D1230.07 BOOL  ; 复检腔体机构：异常标志
D1231.00 BOOL  ; 复检腔体机构：运行条件（自动步）
D1231.02 BOOL  ; 复检腔体机构：运行条件（清氦步）
D1232.00 BOOL  ; 复检腔体机构：平移气缸安全移动条件
D1232.12 BOOL  ; 复检腔体机构：腔体抽真空需求（测试）
D1232.13 BOOL  ; 复检腔体机构：正常清氦需求（正压测试）
D1232.14 BOOL  ; 复检腔体氦检阀打开允许条件
D1232.15 BOOL  ; 复检腔体机构：腔体抽气阀打开允许
D1233.00 BOOL  ; 复检腔体机构：单步/自动循环运行中（总）
D1233.10 BOOL  ; 复检腔体机构：记忆清除(SW)
D1233.12 BOOL  ; 复检腔体机构：自检启动(SW)
D1233.13 BOOL  ; 复检腔体机构：自检停止(SW)
D1233.14 BOOL  ; 复检腔体机构：复位按钮（SW）
D1233.15 BOOL  ; 复检腔体机构：单步（SW）
D1234.00 BOOL  ; 复检腔体机构：单步运行中
D1234.01 BOOL  ; 复检腔体机构：单步/自动循环运行中（自动步）
D1234.03 BOOL  ; 复检腔体机构：自动循环运行中（清氦步）
D1234.06 BOOL  ; 复检腔体机构：自检运行中
D1235.00 BOOL  ; 复检腔体机构：开始运行条件（自动步）
D1235.01 BOOL  ; 复检腔体机构：步进条件（自动步）
D1235.04 BOOL  ; 复检腔体机构：开始运行条件（清氦步）
D1235.05 BOOL  ; 复检腔体机构：步进条件（清氦步）
D1235.13 BOOL  ; 复检腔体机构：步进（清氦步）
D1235.15 BOOL  ; 复检腔体机构：步进（自动步）
D1236 CHANNEL  ; 复检腔体机构：自动流程步序号
D1236.00 BOOL  ; 复检腔体机构：自动开始（自动步）
D1236.01 BOOL  ; 复检腔体机构：平移气缸到氦检位/数据初始化（自动步）
D1236.02 BOOL  ; 复检腔体机构：腔体顶升气缸上升（自动步）
D1236.03 BOOL  ; 复检腔体机构：等待氦检阀打开条件及腔体抽气阀打开条件/开腔体阀（自动步）
D1236.04 BOOL  ; 复检腔体机构：（自动步）
D1236.05 BOOL  ; 复检腔体机构：腔体抽气阀打开/延时开电池抽气阀（自动步）
D1236.06 BOOL  ; 复检腔体机构：关电池抽气阀（自动步）
D1236.07 BOOL  ; 复检腔体机构：开电池注氦阀（自动步）
D1236.08 BOOL  ; 复检腔体机构：关电池注氦阀（自动步）
D1236.09 BOOL  ; 复检腔体机构：（自动步）
D1236.10 BOOL  ; 复检腔体机构：开腔体氦检阀/延时关腔体抽气阀（自动步）
D1236.11 BOOL  ; 复检腔体机构：（自动步）
D1236.12 BOOL  ; 复检腔体机构：关腔体氦检阀（自动步）
D1236.13 BOOL  ; 复检腔体机构：（自动步）
D1236.14 BOOL  ; 复检腔体机构：开腔体阀（自动步）
D1236.15 BOOL  ; 复检腔体机构：开腔体抽真空阀/开电池抽真空阀（自动步）
D1237.00 BOOL  ; 复检腔体机构：关腔体抽真空阀/关电池抽真空阀/开腔体阀（自动步）
D1237.01 BOOL  ; 复检腔体机构：清氦需求判定（自动步）
D1237.02 BOOL  ; 复检腔体机构：开腔体破真空阀/开电池破真空阀（自动步）
D1237.03 BOOL  ; 复检腔体机构：关腔体破真空阀/关电池破真空阀（自动步）
D1237.04 BOOL  ; 复检腔体机构：（自动步）
D1237.05 BOOL  ; 复检腔体机构：（自动步）
D1237.06 BOOL  ; 复检腔体机构：腔体顶升气缸下降（自动步）
D1237.07 BOOL  ; 复检腔体机构：（自动步）
D1237.08 BOOL  ; 复检腔体机构：腔体平移气缸到出料位（自动步）
D1237.09 BOOL  ; 复检腔体机构：（自动步）
D1237.10 BOOL  ; 复检腔体机构：（自动步）
D1237.11 BOOL  ; 复检腔体机构：（自动步）
D1237.12 BOOL  ; 复检腔体机构：（自动步）
D1237.13 BOOL  ; 复检腔体机构：（自动步）
D1237.14 BOOL  ; 复检腔体机构：（自动步）
D1237.15 BOOL  ; 复检腔体机构：循环结束（自动步）
D124 CHANNEL  ; 腔体测试设定清氦次数（次_UInt）
D1244 CHANNEL  ; 复测腔体机构：清氦流程步序号
D1244.00 BOOL  ; 复检腔体机构：自动开始（清氦步）
D1244.01 BOOL  ; 复检腔体机构：平移气缸到氦检位/数据初始化（清氦步）
D1244.02 BOOL  ; 复检腔体机构：腔体顶升气缸上升（清氦步）
D1244.03 BOOL  ; 复检腔体机构：氦检仪真空阀关闭（清氦步）
D1244.04 BOOL  ; 复检腔体机构：正压开腔体阀/负压关腔体阀/氦检阀打开
D1244.05 BOOL  ; 复检腔体机构：（清氦步）
D1244.06 BOOL  ; 复检腔体机构：腔体抽气阀打开/电池抽气阀打开（清氦步）
D1244.07 BOOL  ; 复检腔体机构：腔体抽气阀关闭/电池抽气阀关闭（清氦步）
D1244.08 BOOL  ; 复检腔体机构：（清氦步）
D1244.09 BOOL  ; 复检腔体机构：氦检清洁阀打开/电池破真空阀打开（清氦步）
D1244.10 BOOL  ; 复检腔体机构：氦检清洁阀关闭/电池破真空阀关闭（清氦步）
D1244.11 BOOL  ; 复检腔体机构：（清氦步）
D1244.12 BOOL  ; 复检腔体机构：清氦次数判定（清氦步）
D1244.13 BOOL  ; 复检腔体机构：（清氦步）
D1244.14 BOOL  ; 复检腔体机构：腔体抽气阀打开/电池抽气阀打开（清氦步）
D1244.15 BOOL  ; 复检腔体机构：关闭电池抽气阀（清氦步）
D1245.00 BOOL  ; 复检腔体机构：腔体氦检阀仪真空阀打开/延时关腔体抽气阀（清氦步）
D1245.01 BOOL  ; 复检腔体机构：（清氦步）
D1245.02 BOOL  ; 复检腔体机构：腔体氦检阀关闭（清氦步）
D1245.03 BOOL  ; 复检腔体机构：腔体抽气阀关闭/电池抽气阀关闭（清氦步）
D1245.04 BOOL  ; 复检腔体机构：是否需要重新清氦判定（清氦步）
D1245.05 BOOL  ; 复检腔体机构：（清氦步）
D1245.06 BOOL  ; 复检腔体机构：开腔体破真空阀/开电池破真空阀/开腔体阀（清氦步）
D1245.07 BOOL  ; 复检腔体机构：关腔体破真空阀/关电池破真空阀（清氦步）
D1245.08 BOOL  ; 复检腔体机构：（清氦步）
D1245.09 BOOL  ; 复检腔体机构：清氦完成标志（清氦步）
D1245.10 BOOL  ; 复检腔体机构：（清氦步）
D1245.11 BOOL  ; 复检腔体机构：腔体顶升气缸下降（清氦步）
D1245.12 BOOL  ; 复检腔体机构：腔体平移气缸到初始位（清氦步）
D1245.13 BOOL  ; 复检腔体机构：（清氦步）
D1245.14 BOOL  ; 复检腔体机构：（清氦步）
D1245.15 BOOL  ; 复检腔体机构：循环结束（清氦步）
D1247.00 BOOL  ; 复检腔体机构：复位（M）
D1247.01 BOOL  ; 复检腔体机构：关闭除破真空阀以外全部阀门（复位）
D1247.02 BOOL  ; 复检腔体机构：打开腔体阀门（复位）
D1247.03 BOOL  ; 复检腔体机构：破真空值未到达开破真空阀（复位）
D1247.04 BOOL  ; 复检腔体机构：破真空值到达关破真空阀（复位）
D1247.05 BOOL  ; 复检腔体机构：腔体顶升气缸下降（复位）
D1247.06 BOOL  ; 复检腔体机构：腔体平移气缸初始位（复位）
D1255.00 BOOL  ; 复检腔体机构：抽气阀打开允许（自检）
D1255.01 BOOL  ; 复检腔体机构：抽气阀打开需求（自检）
D1255.04 BOOL  ; 复检腔体机构：真空泵开（自检）
D1255.05 BOOL  ; 复检腔体机构：平移气缸到初始位（自检）
D1255.06 BOOL  ; 复检腔体机构：平移气缸到氦检位（自检）
D1255.07 BOOL  ; 复检腔体机构：顶升气缸下降（自检）
D1255.08 BOOL  ; 复检腔体机构：顶升气缸上升（自检）
D1255.09 BOOL  ; 复检腔体机构：开抽真空阀（自检）
D1255.10 BOOL  ; 复检腔体机构：关抽真空阀（自检）
D1255.11 BOOL  ; 复检腔体机构：开破真空阀（自检）
D1255.12 BOOL  ; 复检腔体机构：关破真空阀（自检）
D1255.13 BOOL  ; 复检腔体机构：破真空阀状态（自检）
D1255.14 BOOL  ; 复检腔体机构：抽真空阀状态（自检）
D126 CHANNEL  ; 腔体测试设定氦检时腔体抽气阀关延时（S_UInt）
D128 CHANNEL  ; 腔体连续NG次数
D1300 CHANNEL  ; #4-1腔体状态（0停用，1待料中，2测试中，3测试完成）
D1302 CHANNEL  ; #4-1腔体测试漏率（Pa.m3/s_Float）
D1304 CHANNEL  ; #4-1腔体测试检漏口压力（Pa_Float）
D1306 CHANNEL  ; #4-1电池充氦压力（Pa_Float）
D1308 CHANNEL  ; #4-1腔体测试结果（1 OK，2腔体泄漏，3气密NG，4注氦超时，5氦检异常，6电池泄漏，7注氦NG，8氦嘴泄漏）
D1310 CHANNEL  ; #4-1充氦嘴压力（Pa_Float）
D1312 CHANNEL  ; #4-1腔体抽气时间（S_UInt）
D1314 CHANNEL  ; #4-1腔体真空压力（Pa_Float）
D1316 CHANNEL  ; #4-1电池抽气时间（S_UInt）
D1318 CHANNEL  ; #4-1电池真空压力（Pa_Float）
D1320 CHANNEL  ; #4-1泄氦后真空度（Pa_Float）
D1322 CHANNEL  ; #4-1电池泄漏量（Pa_Float）
D1330 CHANNEL  ; #4-1腔体自检抽气时间（S_UInt）
D1332 CHANNEL  ; #4-1腔体自检前保压时间（S_UInt）
D1334 CHANNEL  ; #4-1腔体自检保压时间（S_UInt）
D1336 CHANNEL  ; #4-1腔体自检保压前真空（Pa_Float）
D1338 CHANNEL  ; #4-1腔体自检保压后真空（Pa_Float）
D1340 CHANNEL  ; #4-1腔体自检泄漏量（Pa_Float）
D1342 CHANNEL  ; #4-1腔体自检结果（1-OK，2-NG）
D1358 CHANNEL  ; #4-1清氦泄漏率（清氦）
D136 CHANNEL  ; 腔体测试设定腔体预抽检测时间（S_UInt）
D1360 CHANNEL  ; #4-1氦检时真空值（标漏）
D1362 CHANNEL  ; #4-1氦检漏率（标漏）
D1370 CHANNEL  ; #4腔体抽真空需求计时
D1372 CHANNEL  ; #4-1腔体管路清氦计数
D138 CHANNEL  ; $?St$Bk?_#[186] / 管路清氦注氮时间（S_UInt） / $?St$Bk?_#[186]
D14 CHANNEL  ; 感应器ON延时设定值
D1400 CHANNEL  ; #4-2腔体状态（0停用，1待料中，2测试中，3测试完成）
D1402 CHANNEL  ; #4-2腔体测试漏率（Pa.m3/s_Float）
D1404 CHANNEL  ; #4-2腔体测试检漏口压力（Pa_Float）
D1406 CHANNEL  ; #4-2电池充氦压力（Pa_Float）
D1408 CHANNEL  ; #4-2腔体测试结果（1 OK，2腔体泄漏，3气密NG，4注氦超时，5氦检异常，6电池泄漏，7注氦NG，8氦嘴泄漏）
D1410 CHANNEL  ; #4-2充氦嘴压力（Pa_Float）
D1412 CHANNEL  ; #4-2腔体抽气时间（S_UInt）
D1414 CHANNEL  ; #4-2腔体真空压力（Pa_Float）
D1416 CHANNEL  ; #4-2电池抽气时间（S_UInt）
D1418 CHANNEL  ; #4-2电池真空压力（Pa_Float）
D1420 CHANNEL  ; #4-2泄氦后真空度（Pa_Float）
D1422 CHANNEL  ; #4-2电池泄漏量（Pa_Float）
D1430 CHANNEL  ; #4-2腔体自检抽气时间（S_UInt）
D1432 CHANNEL  ; #4-2腔体自检前保压时间（S_UInt）
D1434 CHANNEL  ; #4-2腔体自检保压时间（S_UInt）
D1436 CHANNEL  ; #4-2腔体自检保压前真空（Pa_Float）
D1438 CHANNEL  ; #4-2腔体自检保压后真空（Pa_Float）
D1440 CHANNEL  ; #4-2腔体自检泄漏量（Pa_Float）
D1442 CHANNEL  ; #4-2腔体自检结果（1-OK，2-NG）
D1458 CHANNEL  ; #4-2清氦泄漏率（清氦）
D1460 CHANNEL  ; #4-2氦检时真空值（标漏）
D1462 CHANNEL  ; #4-2氦检漏率（标漏）
D15 CHANNEL  ; 感应器ON延时设定值_1
D150 CHANNEL  ; 腔体自检真空到达阈值SV（Pa_Float）
D1500 CHANNEL  ; #4-1电池真空偏值设定(Float)
D1502 CHANNEL  ; #4-1电池实际真空值(Float)
D1504 CHANNEL  ; #4-1电池真空模拟量读数(Int)
D1510 CHANNEL  ; #4-2电池真空偏值设定(Float)
D1512 CHANNEL  ; #4-2电池实际真空值（Pa_Float）
D1514 CHANNEL  ; #4-2电池真空模拟量读数(Int)
D152 CHANNEL  ; 腔体自检抽真空时间上限SV（S_UInt）
D1522 CHANNEL  ; #4腔体实际真空值(Float)
D1524 CHANNEL  ; #4腔体真空模拟量读数(Int)
D1530 CHANNEL  ; 复测电池真空偏值设定(Float)
D1532 CHANNEL  ; 复测电池实际真空值(Float)
D1534 CHANNEL  ; 复测电池真空模拟量读数(Int)
D154 CHANNEL  ; 腔体自检泄漏量阈值SV（Pa_Float）
D1542 CHANNEL  ; 复测腔体实际真空值(Float)
D1544 CHANNEL  ; 复测腔体真空模拟量读数(Int)
D156 CHANNEL  ; 清氦泄漏率（Pa.m3/s_Float）
D158 CHANNEL  ; 清氦泄漏率（Pa.m3/s_Float_指数）
D16 CHANNEL  ; 感应器延时时间
D160 CHANNEL  ; 电池测试设定真空阈值（Pa_Float）
D162 CHANNEL  ; 电池测试设定抽真空时间上限（S_UInt）
D168 CHANNEL  ; 电池测试设定注氦时间上限（S_UInt）
D17 CHANNEL  ; 感应器ON延时设定值_3
D170 CHANNEL  ; 电池测试设定清氦压力（Pa_Float）
D1700 CHANNEL  ; 复测腔体状态（0停用，1待料中，2测试中，3测试完成 4-清氦中  5-放料完成）
D1702 CHANNEL  ; 复测腔体测试漏率（Pa.m3/s_Float）
D1704 CHANNEL  ; 复测腔体测试检漏口压力（Pa_Float）
D1706 CHANNEL  ; 复测电池充氦压力（Pa_Float）
D1708 CHANNEL  ; 复测腔体测试结果（1 OK，2腔体泄漏，3气密NG，4注氦超时，5氦检异常，6电池泄漏，7注氦NG，8氦嘴泄漏）
D1710 CHANNEL  ; 复测充氦嘴压力（Pa_Float）
D1712 CHANNEL  ; 复测腔体抽气时间（S_UInt）
D1714 CHANNEL  ; 复测腔体真空压力（Pa_Float）
D1716 CHANNEL  ; 复测电池抽气时间（S_UInt）
D1718 CHANNEL  ; 复测电池真空压力（Pa_Float）
D172 CHANNEL  ; 电池测试设定破真空阈值（Pa_Float）
D1720 CHANNEL  ; 复测泄氦后真空度（Pa_Float）
D1722 CHANNEL  ; 复测电池泄漏量（Pa_Float）
D1730 CHANNEL  ; 复测腔体自检抽气时间（S_UInt）
D1732 CHANNEL  ; 复测腔体自检前保压时间（S_UInt）
D1734 CHANNEL  ; 复测腔体自检保压时间（S_UInt）
D1736 CHANNEL  ; 复测腔体自检保压前真空（Pa_Float）
D1738 CHANNEL  ; 复测腔体自检保压后真空（Pa_Float）
D174 CHANNEL  ; 电池测试设定预抽检测压力（Pa_Float）
D1740 CHANNEL  ; 复测腔体自检泄漏量（Pa_Float）
D1742 CHANNEL  ; 复测腔体自检结果（1-OK，2-NG）
D176 CHANNEL  ; 电池测试设定注氦压力（Pa_Float）
D1770 CHANNEL  ; 复检腔体抽真空需求计时
D1772 CHANNEL  ; 复测腔体管路清氦计数
D178 CHANNEL  ; 注氦压力下限值（Pa_Float）
D18 CHANNEL  ; 自动运行条件延时时间
D180 CHANNEL  ; 注氦压力上限值
D182 CHANNEL  ; 注氦压力上限
D188 CHANNEL  ; 漏率设定值（Pa.m3/s_Float）
D19 CHANNEL  ; 自动运行步间间隔时间
D190 CHANNEL  ; 检漏口压力设定值（Pa_Float）
D196 CHANNEL  ; 氦检仪漏率（Pa.m3/s_Float）
D198 CHANNEL  ; 氦检仪检漏口压力（Pa_Float）
D20 CHANNEL  ; 感应器ON延时设定值_6
D200 CHANNEL  ; #1-1腔体状态（0停用，1待料中，2测试中，3测试完成，4-清氦中）
D20124 CHANNEL  ; 进料伺服X轴目标位置
D20126 CHANNEL  ; 进料X轴 速度
D20128 CHANNEL  ; 进料X轴 加速时间
D20130 CHANNEL  ; 进料X轴 减速时间
D20136 CHANNEL  ; 进料Z轴 目标位置
D20138 CHANNEL  ; 进料Z轴 速度
D20140 CHANNEL  ; 进料Z轴 加速时间
D20142 CHANNEL  ; 进料Z轴 减速时间
D20148 CHANNEL  ; 出料X轴 目标位置
D20148 CHANNEL  ; 出料伺服X轴自动目标位置
D20150 CHANNEL  ; 出料X轴 速度
D20152 CHANNEL  ; 出料X轴 加速时间
D20154 CHANNEL  ; 出料X轴 减速时间
D20160 CHANNEL  ; 出料Z轴 目标位置
D20160 CHANNEL  ; 出料伺服Z轴目标位置
D20160 CHANNEL  ; 出料伺服Z轴自动目标位置
D20162 CHANNEL  ; 出料Z轴 速度
D20164 CHANNEL  ; 出料Z轴 加速时间
D20166 CHANNEL  ; 出料Z轴 减速时间
D20172 CHANNEL  ; 进料X轴 当前位置
D20176 CHANNEL  ; 进料Z轴 当前位置
D20180 CHANNEL  ; 出料X轴 当前位置
D20184 CHANNEL  ; 出料Z轴 当前位置
D202 CHANNEL  ; #1-1腔体测试漏率（Pa.m3/s_Float）
D204 CHANNEL  ; #1-1腔体测试检漏口压力（Pa_Float）
D206 CHANNEL  ; #1-1电池充氦压力（Pa_Float）
D208 CHANNEL  ; #1-1腔体测试结果（1 OK，2腔体泄漏，3气密NG，4注氦超时，5氦检异常，6电池泄漏）
D21 CHANNEL  ; 报警长延时
D210 CHANNEL  ; $?St$Bk?_#[187] / #1-1充氦嘴压力（Pa_Float） / #1-1充氦嘴压力（Pa_Float） / #1-1充氦嘴压力（Pa_Float）$?St$Bk?_#[187]
D212 CHANNEL  ; #1-1腔体抽气时间（S_UInt）
D214 CHANNEL  ; #1-1腔体真空压力（Pa_Float）
D216 CHANNEL  ; #1-1电池抽气时间（S_UInt）
D2160 CHANNEL  ; 氦检仪状态(1.检漏；2.待机；3.定标；4.启动；5.错误；6.暂停)
D2162 CHANNEL  ; 氦检实时漏率显示
D218 CHANNEL  ; #1-1电池真空压力（Pa_Float）
D22 CHANNEL  ; 报警短延时
D220 CHANNEL  ; #1-1泄氦后真空度
D222 CHANNEL  ; #1-1电池泄漏量（Pa_Float）
D23 CHANNEL  ; 氦检相关无传感器阀开关到位延时设定
D230 CHANNEL  ; #1-1腔体自检抽气时间（S_UInt）
D232 CHANNEL  ; #1-1腔体自检前保压时间（S_UInt）
D234 CHANNEL  ; #1-1腔体自检保压时间（S_UInt）
D236 CHANNEL  ; #1-1腔体自检保压前真空（Pa_Float）
D238 CHANNEL  ; #1-1腔体自检保压后真空（Pa_Float）
D24 CHANNEL  ; 伺服到位延时
D240 CHANNEL  ; #1-1腔体自检泄漏量（Pa_Float）
D242 CHANNEL  ; #1-1腔体自检结果（1-OK，2-NG）
D25 CHANNEL  ; 夹爪报警延时
D2500 CHANNEL  ; #1扫码阻挡气缸缩回位延时设定值
D2501 CHANNEL  ; #1扫码阻挡气缸伸出位延时设定值
D2502 CHANNEL  ; #1隔离气缸缩回位延时设定值
D2503 CHANNEL  ; 0延时设定值
D2504 CHANNEL  ; #2扫码阻挡气缸缩回位延时设定值
D2505 CHANNEL  ; #2扫码阻挡气缸伸出位延时设定值
D2506 CHANNEL  ; #2隔离气缸缩回位延时设定值
D2507 CHANNEL  ; 0延时设定值
D2508 CHANNEL  ; #1进料夹爪夹紧位延时设定值
D2509 CHANNEL  ; #1进料夹爪松开位延时设定值
D2510 CHANNEL  ; #2进料夹爪夹紧位延时设定值
D2511 CHANNEL  ; #2进料夹爪松开位延时设定值
D2512 CHANNEL  ; 进料夹爪变距气缸伸出位延时设定值
D2513 CHANNEL  ; 进料夹爪变距气缸缩回位延时设定值
D2514 CHANNEL  ; #1出料夹爪夹紧位延时设定值
D2515 CHANNEL  ; #1出料夹爪松开位延时设定值
D2516 CHANNEL  ; #2出料夹爪夹紧位延时设定值
D2517 CHANNEL  ; #2出料夹爪松开位延时设定值
D2518 CHANNEL  ; 出料夹爪变距气缸伸出位延时设定值
D2519 CHANNEL  ; 出料夹爪变距气缸缩回位延时设定值
D2520 CHANNEL  ; #1腔体平移一级气缸缩回位延时设定值
D2521 CHANNEL  ; #1腔体平移一级气缸伸出位延时设定值
D2522 CHANNEL  ; #1腔体平移二级气缸缩回位延时设定值
D2523 CHANNEL  ; #1腔体平移二级气缸伸出位延时设定值
D2524 CHANNEL  ; #1腔体顶伸气缸上升位延时设定值
D2525 CHANNEL  ; #1腔体顶伸气缸下降位延时设定值
D2526 CHANNEL  ; #1腔体氦检阀开到位延时设定值
D2527 CHANNEL  ; #1腔体氦检阀关到位延时设定值
D2528 CHANNEL  ; 0延时设定值
D2529 CHANNEL  ; 0延时设定值
D2530 CHANNEL  ; 0延时设定值
D2531 CHANNEL  ; 0延时设定值
D2532 CHANNEL  ; 0延时设定值
D2533 CHANNEL  ; #2腔体平移一级气缸缩回位延时设定值
D2534 CHANNEL  ; #2腔体平移一级气缸伸出位延时设定值
D2535 CHANNEL  ; #2腔体平移二级气缸缩回位延时设定值
D2536 CHANNEL  ; #2腔体平移二级气缸伸出位延时设定值
D2537 CHANNEL  ; #2腔体顶伸气缸上升位延时设定值
D2538 CHANNEL  ; #2腔体顶伸气缸下降位延时设定值
D2539 CHANNEL  ; #2腔体氦检阀开到位延时设定值
D2540 CHANNEL  ; #2腔体氦检阀关到位延时设定值
D2541 CHANNEL  ; 0延时设定值
D2542 CHANNEL  ; 0延时设定值
D2543 CHANNEL  ; 0延时设定值
D2544 CHANNEL  ; 0延时设定值
D2545 CHANNEL  ; 0延时设定值
D2546 CHANNEL  ; #3腔体平移一级气缸缩回位延时设定值
D2547 CHANNEL  ; #3腔体平移一级气缸伸出位延时设定值
D2548 CHANNEL  ; #3腔体平移二级气缸缩回位延时设定值
D2549 CHANNEL  ; #3腔体平移二级气缸伸出位延时设定值
D2550 CHANNEL  ; #3腔体顶伸气缸上升位延时设定值
D2551 CHANNEL  ; #3腔体顶伸气缸下降位延时设定值
D2552 CHANNEL  ; #3腔体氦检阀开到位延时设定值
D2553 CHANNEL  ; #3腔体氦检阀关到位延时设定值
D2554 CHANNEL  ; 氦检仪准备好了信号延时设定值
D2555 CHANNEL  ; 氦检仪故障信号延时设定值
D2556 CHANNEL  ; 0延时设定值
D2557 CHANNEL  ; 0延时设定值
D2558 CHANNEL  ; 0延时设定值
D2559 CHANNEL  ; 进料伺服X轴准备好了信号延时设定值
D2560 CHANNEL  ; 进料伺服X轴故障信号延时设定值
D2561 CHANNEL  ; 进料伺服Z轴准备好了信号延时设定值
D2562 CHANNEL  ; 进料伺服Z轴故障信号延时设定值
D2563 CHANNEL  ; 0延时设定值
D2564 CHANNEL  ; 出料伺服X轴准备好了信号延时设定值
D2565 CHANNEL  ; 出料伺服X轴故障信号延时设定值
D2566 CHANNEL  ; 出料伺服Z轴准备好了信号延时设定值
D2567 CHANNEL  ; 出料伺服Z轴故障信号延时设定值
D2568 CHANNEL  ; 0延时设定值
D2569 CHANNEL  ; 腔体抽真空泵运行信号延时设定值
D2570 CHANNEL  ; 腔体抽真空泵过载信号延时设定值
D2571 CHANNEL  ; 氦检前置泵运行信号延时设定值
D2572 CHANNEL  ; 氦检前置泵过载信号延时设定值
D2573 CHANNEL  ; 启动按钮延时设定值
D2574 CHANNEL  ; 停止按钮延时设定值
D2575 CHANNEL  ; 复位按钮延时设定值
D2576 CHANNEL  ; 急停按钮延时设定值
D2577 CHANNEL  ; 手自动选择延时设定值
D2578 CHANNEL  ; #1进料夹爪防下坠感应延时设定值
D2579 CHANNEL  ; #2进料夹爪防下坠感应延时设定值
D258 CHANNEL  ; #1-1清氦泄漏率（清氦）
D2580 CHANNEL  ; #1出料夹爪防下坠感应延时设定值
D2581 CHANNEL  ; #2出料夹爪防下坠感应延时设定值
D2582 CHANNEL  ; 0延时设定值
D2583 CHANNEL  ; 进料对接输入延时设定值
D2584 CHANNEL  ; 出料对接输入延时设定值
D2585 CHANNEL  ; 0延时设定值
D2586 CHANNEL  ; 0延时设定值
D2587 CHANNEL  ; 设备总气压信号延时设定值
D2588 CHANNEL  ; #1来料位有料感应延时设定值
D2589 CHANNEL  ; #2来料位有料感应延时设定值
D2590 CHANNEL  ; #1隔离位有料感应延时设定值
D2591 CHANNEL  ; #2隔离位有料感应延时设定值
D2592 CHANNEL  ; #1扫码位有料感应延时设定值
D2593 CHANNEL  ; #2扫码位有料感应延时设定值
D2594 CHANNEL  ; #1-1进料位有料感应延时设定值
D2595 CHANNEL  ; #1-2进料位有料感应延时设定值
D2596 CHANNEL  ; #2-1进料位有料感应延时设定值
D2597 CHANNEL  ; #2-2进料位有料感应延时设定值
D2598 CHANNEL  ; 进料夹爪柔性感应延时设定值
D2599 CHANNEL  ; 出料夹爪柔性感应延时设定值
D260 CHANNEL  ; #1-1氦检时真空值（标漏）
D2600 CHANNEL  ; #1进料夹爪对应腔体有料感应延时设定值
D2601 CHANNEL  ; #2进料夹爪对应腔体有料感应延时设定值
D2602 CHANNEL  ; 扫码NG放料#1位有料感应延时设定值
D2603 CHANNEL  ; 扫码NG放料#2位有料感应延时设定值
D2604 CHANNEL  ; 扫码NG料满位有料感应延时设定值
D2605 CHANNEL  ; 进料配对位有料感应延时设定值
D2606 CHANNEL  ; 出料配对位有料感应延时设定值
D2607 CHANNEL  ; 氦检NG放料#1位有料感应延时设定值
D2608 CHANNEL  ; 氦检NG放料#2位有料感应延时设定值
D2609 CHANNEL  ; 氦检NG料满位有料感应延时设定值
D2610 CHANNEL  ; #1-1出料位有料感应延时设定值
D2611 CHANNEL  ; #1-2出料位有料感应延时设定值
D2612 CHANNEL  ; #2-1出料位有料感应延时设定值
D2613 CHANNEL  ; #2-2出料位有料感应延时设定值
D2614 CHANNEL  ; #1门磁开关延时设定值
D2615 CHANNEL  ; #2门磁开关延时设定值
D2616 CHANNEL  ; #3门磁开关延时设定值
D2617 CHANNEL  ; #4门磁开关延时设定值
D2618 CHANNEL  ; #5门磁开关延时设定值
D2619 CHANNEL  ; #6门磁开关延时设定值
D262 CHANNEL  ; #1-1氦检漏率（标漏）
D2620 CHANNEL  ; #7门磁开关延时设定值
D2621 CHANNEL  ; #8门磁开关延时设定值
D2622 CHANNEL  ; #9门磁开关延时设定值
D2623 CHANNEL  ; #10门磁开关延时设定值
D2624 CHANNEL  ; #11门磁开关延时设定值
D2625 CHANNEL  ; #12门磁开关延时设定值
D2626 CHANNEL  ; #13门磁开关延时设定值
D2627 CHANNEL  ; #14门磁开关延时设定值
D2663 CHANNEL  ; $?St$Bk?_#[188] / #1隔离气缸伸出位延时设定值 / $?St$Bk?_#[188]
D2667 CHANNEL  ; $?St$Bk?_#[189] / #2隔离气缸伸出位延时设定值 / $?St$Bk?_#[189]
D270 CHANNEL  ; #1腔体抽真空需求计时
D272 CHANNEL  ; #1-1腔体管路清氦计数
D2916 CHANNEL  ; 复测夹爪气缸夹紧位延时设定值
D2917 CHANNEL  ; 复测夹爪气缸松开位延时设定值
D2918 CHANNEL  ; 复检夹爪柔性感应延时设定值
D2919 CHANNEL  ; 复测腔体移栽气缸缩回位延时设定值
D2920 CHANNEL  ; 复测腔体移栽气缸伸出位延时设定值
D2921 CHANNEL  ; 复测腔体顶升气缸缩回位延时设定值
D2922 CHANNEL  ; 复测腔体顶升气缸伸出位延时设定值
D2923 CHANNEL  ; 复测腔体氦检阀开到位延时设定值
D2924 CHANNEL  ; 复测腔体氦检阀关到位延时设定值
D2925 CHANNEL  ; 复测腔体感应有料感应延时设定值
D2926 CHANNEL  ; 0延时设定值
D2927 CHANNEL  ; 出料配对位有料感应2延时设定值
D2928 CHANNEL  ; 0延时设定值
D2929 CHANNEL  ; 0延时设定值
D2930 CHANNEL  ; 0延时设定值
D2931 CHANNEL  ; 0延时设定值
D2932 CHANNEL  ; 腔体抽真空泵M2运行信号延时设定值
D2933 CHANNEL  ; 腔体抽真空泵M2过载信号延时设定值
D2934 CHANNEL  ; 测伺服X轴准备好信号延时设定值
D2935 CHANNEL  ; 复测伺服X轴故障信号延时设定值
D2936 CHANNEL  ; 复测伺服Z轴准备好信号延时设定值
D2937 CHANNEL  ; 复测伺服Z轴故障信号延时设定值
D2938 CHANNEL  ; 0延时设定值
D2939 CHANNEL  ; 0延时设定值
D2940 CHANNEL  ; 0延时设定值
D2941 CHANNEL  ; 0延时设定值
D2942 CHANNEL  ; 设备真空压力信号#1延时设定值
D2943 CHANNEL  ; 设备真空压力信号#2延时设定值
D2944 CHANNEL  ; 设备氦气压力信号#1延时设定值
D2945 CHANNEL  ; 设备氦气压力信号#2延时设定值
D2946 CHANNEL  ; 设备注氦压力调节阀#1延时设定值
D2947 CHANNEL  ; 设备注氦压力调节阀#2延时设定值
D2948 CHANNEL  ; 复测缓存拨料气缸缩回位延时设定值
D2949 CHANNEL  ; 复测缓存拨料气缸伸出位延时设定值
D2950 CHANNEL  ; 复测缓存顶升气缸缩回位延时设定值
D2951 CHANNEL  ; 复测缓存顶升气缸伸出位延时设定值
D2952 CHANNEL  ; 复测缓存#1有料感应1延时设定值
D2953 CHANNEL  ; 复测缓存#1有料感应2延时设定值
D2954 CHANNEL  ; 复测缓存#1有料感应3延时设定值
D2955 CHANNEL  ; 复测缓存#1有料感应4延时设定值
D2956 CHANNEL  ; 复测缓存#2有料感应1延时设定值
D2957 CHANNEL  ; 复测缓存#2有料感应2延时设定值
D2958 CHANNEL  ; 复测缓存#2有料感应3延时设定值
D2959 CHANNEL  ; 复测缓存#2有料感应4延时设定值
D296 CHANNEL  ; 字符表示形式
D297 CHANNEL  ; 全位数
D298 CHANNEL  ; 小数位数
D2984 CHANNEL  ; #4腔体平移一级气缸缩回位延时设定值
D2985 CHANNEL  ; #4腔体平移一级气缸伸出位延时设定值
D2986 CHANNEL  ; #4腔体平移二级气缸缩回位延时设定值
D2987 CHANNEL  ; #4腔体平移二级气缸伸出位延时设定值
D2988 CHANNEL  ; #4腔体顶伸气缸上升位延时设定值
D2989 CHANNEL  ; #4腔体顶伸气缸下降位延时设定值
D2990 CHANNEL  ; #4腔体氦检阀开到位延时设定值
D2991 CHANNEL  ; #4腔体氦检阀关到位延时设定值
D30 CHANNEL  ; NG扫码重试次数设置
D300 CHANNEL  ; #2-1腔体状态（0停用，1待料中，2测试中，3测试完成，4-清氦中）
D3000 CHANNEL  ; 设备PPM测试时间设置
D3002 CHANNEL  ; 设备PPM测试时间累计
D3004 CHANNEL  ; 设备PPM测试#1出料夹爪数量累计
D3006 CHANNEL  ; 设备PPM测试#2出料夹爪数量累计
D3008 CHANNEL  ; 设备PPM测试出料夹爪总数量累计
D302 CHANNEL  ; #2-1腔体测试漏率（Pa.m3/s_Float）
D304 CHANNEL  ; #2-1腔体测试检漏口压力（Pa_Float）
D306 CHANNEL  ; #2-1电池充氦压力（Pa_Float）
D308 CHANNEL  ; #2-1腔体测试结果（1 OK，2腔体泄漏，3气密NG，4注氦超时，5氦检异常，6电池泄漏，7注氦NG，8氦嘴泄漏）
D310 CHANNEL  ; #2-1充氦嘴压力（Pa_Float）
D3102 CHANNEL  ; 腔体测试设定抽真空时间上限（S_UInt）浮点
D3110 CHANNEL  ; 腔体测试设定氦检时间（S_UInt）浮点
D312 CHANNEL  ; #2-1腔体抽气时间（S_UInt）
D3136 CHANNEL  ; 腔体测试设定腔体预抽检测时间（S_UInt）浮点
D314 CHANNEL  ; #2-1腔体真空压力（Pa_Float）
D316 CHANNEL  ; #2-1电池抽气时间（S_UInt）
D3162 CHANNEL  ; 电池测试设定抽真空时间上限（S_UInt）浮点
D318 CHANNEL  ; #2-1电池真空压力（Pa_Float）
D320 CHANNEL  ; #2-1泄氦后真空度
D322 CHANNEL  ; #2-1电池泄漏量（Pa_Float）
D330 CHANNEL  ; #2-1腔体自检抽气时间（S_UInt）
D3300 CHANNEL  ; 浮点10
D332 CHANNEL  ; #2-1腔体自检前保压时间（S_UInt）
D334 CHANNEL  ; #2-1腔体自检保压时间（S_UInt）
D336 CHANNEL  ; #2-1腔体自检保压前真空（Pa_Float）
D338 CHANNEL  ; #2-1腔体自检保压后真空（Pa_Float）
D340 CHANNEL  ; #2-1腔体自检泄漏量（Pa_Float）
D342 CHANNEL  ; #2-1腔体自检结果（1-OK，2-NG）
D358 CHANNEL  ; $?St$Bk?_#[190] / #2-1清氦泄漏率（清氦） / $?St$Bk?_#[190]
D360 CHANNEL  ; #2-1氦检时真空值（标漏）
D362 CHANNEL  ; #2-1氦检漏率（标漏）
D370 CHANNEL  ; #2腔体抽真空需求计时
D372 CHANNEL  ; #2-1腔体管路清氦计数
D40 CHANNEL  ; #1出料夹爪OK料计数（DINT）
D400 CHANNEL  ; #3-1腔体状态（0停用，1待料中，2测试中，3测试完成，4-清氦中）
D402 CHANNEL  ; #3-1腔体测试漏率（Pa.m3/s_Float）
D404 CHANNEL  ; #3-1腔体测试检漏口压力（Pa_Float）
D406 CHANNEL  ; #3-1电池充氦压力（Pa_Float）
D408 CHANNEL  ; #3-1腔体测试结果（1 OK，2腔体泄漏，3气密NG，4注氦超时，5氦检异常，6电池泄漏，7注氦NG，8氦嘴泄漏）
D410 CHANNEL  ; #3-1充氦嘴压力（Pa_Float）
D4100 CHANNEL  ; 腔体测试设定真空阈值（Pa_Float）储存
D4102 CHANNEL  ; 腔体测试设定抽真空时间上限（S_UInt）储存
D4104 CHANNEL  ; 腔体测试设定清氦压力（Pa_Float）储存
D4110 CHANNEL  ; 腔体测试设定氦检时间（S_UInt）储存
D412 CHANNEL  ; #3-1腔体抽气时间（S_UInt）
D4136 CHANNEL  ; 腔体测试设定腔体预抽检测时间（S_UInt）储存
D414 CHANNEL  ; #3-1腔体真空压力（Pa_Float）
D416 CHANNEL  ; #3-1电池抽气时间（S_UInt）
D4160 CHANNEL  ; 电池测试设定真空阈值（Pa_Float）储存
D4162 CHANNEL  ; 电池测试设定抽真空时间上限（S_UInt）储存
D4170 CHANNEL  ; 电池测试设定清氦压力（Pa_Float）储存
D4174 CHANNEL  ; 电池测试设定预抽检测压力（Pa_Float）储存
D4176 CHANNEL  ; 电池测试设定清氦压力（Pa_Float）储存
D418 CHANNEL  ; #3-1电池真空压力（Pa_Float）
D42 CHANNEL  ; #1出料夹爪NG料计数（DINT）
D420 CHANNEL  ; #3-1泄氦后真空度
D422 CHANNEL  ; #3-1电池泄漏量（Pa_Float）
D430 CHANNEL  ; #3-1腔体自检抽气时间（S_UInt）
D432 CHANNEL  ; #3-1腔体自检前保压时间（S_UInt）
D434 CHANNEL  ; #3-1腔体自检保压时间（S_UInt）
D436 CHANNEL  ; #3-1腔体自检保压前真空（Pa_Float）
D438 CHANNEL  ; #3-1腔体自检保压后真空（Pa_Float）
D44 CHANNEL  ; 出料夹爪OK料总计数（DINT）
D440 CHANNEL  ; #3-1腔体自检泄漏量（Pa_Float）
D442 CHANNEL  ; #3-1腔体自检结果（1-OK，2-NG）
D458 CHANNEL  ; $?St$Bk?_#[191] / #3-1清氦泄漏率（清氦） / $?St$Bk?_#[191]
D46 CHANNEL  ; 出料夹爪总计数（DINT）
D460 CHANNEL  ; #3-1氦检时真空值（标漏）
D462 CHANNEL  ; #3-1氦检漏率（标漏）
D470 CHANNEL  ; #3腔体抽真空需求计时
D472 CHANNEL  ; #3-1腔体管路清氦计数
D48 CHANNEL  ; 出料夹爪OK料总计数（Float）
D4994 CHANNEL  ; 泄漏率设定值（Pa.m3/s_Float）储存
D4996 CHANNEL  ; 检漏口压力设定值（Pa_Float）储存
D4998 CHANNEL  ; 清氦漏率设定值（Pa_Float）储存
D50 CHANNEL  ; #2出料夹爪OK料计数（DINT）
D500 CHANNEL  ; #1-2腔体状态（0停用，1待料中，2测试中，3测试完成，4-清氦中）
D502 CHANNEL  ; #1-2腔体测试漏率（Pa.m3/s_Float）
D504 CHANNEL  ; #1-2腔体测试检漏口压力（Pa_Float）
D506 CHANNEL  ; #1-2电池充氦压力（Pa_Float）
D508 CHANNEL  ; #1-2腔体测试结果（1 OK，2腔体泄漏，3气密NG，4注氦超时，5氦检异常，6电池泄漏，7注氦NG，8氦嘴泄漏）
D510 CHANNEL  ; #1-2充氦嘴压力（Pa_Float）
D512 CHANNEL  ; #1-2腔体抽气时间（S_UInt）
D514 CHANNEL  ; #1-2腔体真空压力（Pa_Float）
D516 CHANNEL  ; #1-2电池抽气时间（S_UInt）
D518 CHANNEL  ; #1-2电池真空压力（Pa_Float）
D52 CHANNEL  ; #2出料夹爪NG料计数（DINT）
D520 CHANNEL  ; #1-2泄氦后真空度
D5200 CHANNEL  ; 发送内容“T”+“0D”
D5201 CHANNEL  ; 发送内容“0A”
D5210 CHANNEL  ; 进料#1扫码数据开始字
D522 CHANNEL  ; #1-2电池泄漏量（Pa_Float）
D5240 CHANNEL  ; 进料#1扫码条码开始字
D5259 CHANNEL  ; 进料#1扫码数据结束字
D530 CHANNEL  ; #1-2腔体自检抽气时间（S_UInt）
D5300 CHANNEL  ; 进料#2扫码长度
D5301 CHANNEL  ; 进料#2扫码条码开始字
D5319 CHANNEL  ; 进料#2扫码结束字
D532 CHANNEL  ; #1-2腔体自检前保压时间（S_UInt）
D534 CHANNEL  ; #1-2腔体自检保压时间（S_UInt）
D536 CHANNEL  ; #1-2腔体自检保压前真空（Pa_Float）
D538 CHANNEL  ; #1-2腔体自检保压后真空（Pa_Float）
D54 CHANNEL  ; 出料夹爪NG料总计数（DINT）
D540 CHANNEL  ; #1-2腔体自检泄漏量（Pa_Float）
D542 CHANNEL  ; #1-2腔体自检结果（1-OK，2-NG,3-抽真空NG）
D56 CHANNEL  ; 出料夹爪总计数（Float）
D560 CHANNEL  ; #1-2氦检时真空值（标漏）
D562 CHANNEL  ; #1-2氦检漏率（标漏）
D58 CHANNEL  ; 出料夹爪OK料百分比（Float）
D5800 CHANNEL  ; #1批次号开始字
D5850 CHANNEL  ; #2批次号开始字
D60 CHANNEL  ; 合格比例
D600 CHANNEL  ; #2-2腔体状态（0停用，1待料中，2测试中，3测试完成，4-清氦中）
D6000 CHANNEL  ; 进料伺服X轴加速比率
D6001 CHANNEL  ; 进料伺服X轴减速比率
D6002 CHANNEL  ; 进料伺服X轴目标速度
D6003 CHANNEL  ; 进料伺服X轴目标速度
D6005 CHANNEL  ; 进料伺服X轴目标位置
D6006 CHANNEL  ; 进料伺服X轴启动频率
D6007 CHANNEL  ; 进料伺服X轴启动频率
D602 CHANNEL  ; #2-2腔体测试漏率（Pa.m3/s_Float）
D6022 CHANNEL  ; 进料伺服X轴JOG运行速度
D6031 CHANNEL  ; 进料伺服X轴JOG停止速度
D6032 CHANNEL  ; 进料伺服X轴JOG停止速度
D604 CHANNEL  ; #2-2腔体测试检漏口压力（Pa_Float）
D6040 CHANNEL  ; 进料伺服X轴当前位置
D6041 CHANNEL  ; 进料伺服X轴当前位置
D6042 CHANNEL  ; 进料伺服X轴当前速度
D6043 CHANNEL  ; 进料伺服X轴当前速度
D6050 CHANNEL  ; 进/出料伺服急停位置预置
D606 CHANNEL  ; #2-2电池充氦压力（Pa_Float）
D608 CHANNEL  ; #2-2腔体测试结果（1 OK，2腔体泄漏，3气密NG，4注氦超时，5氦检异常，6电池泄漏，7注氦NG，8氦嘴泄漏）
D610 CHANNEL  ; #2-2充氦嘴压力（Pa_Float）
D6100 CHANNEL  ; 进料伺服X轴加速比率SV
D6101 CHANNEL  ; 进料伺服X轴减速比率SV
D6102 CHANNEL  ; 进料伺服X轴目标速度SV
D6103 CHANNEL  ; 进料伺服X轴目标速度SV
D6106 CHANNEL  ; 进料伺服X轴启动频率SV
D6107 CHANNEL  ; 进料伺服X轴启动频率SV
D612 CHANNEL  ; #2-2腔体抽气时间（S_UInt）
D6120 CHANNEL  ; 进料伺服X轴JOG运行/停止加减速SV
D6121 CHANNEL  ; 进料伺服X轴JOG运行速度SV
D6122 CHANNEL  ; 进料伺服X轴JOG运行速度SV
D6131 CHANNEL  ; 进料伺服X轴JOG停止速度SV
D6132 CHANNEL  ; 进料伺服X轴JOG停止速度SV
D614 CHANNEL  ; #2-2腔体真空压力（Pa_Float）
D6152 CHANNEL  ; 进料伺服X轴取料位SV
D6153 CHANNEL  ; 进料伺服X轴取料位SV
D6154 CHANNEL  ; 进料伺服X轴#1腔放料位SV
D6155 CHANNEL  ; 进料伺服X轴#1腔放料位SV
D6156 CHANNEL  ; 进料伺服X轴#2腔放料位SV
D6157 CHANNEL  ; 进料伺服X轴#2腔放料位SV
D6158 CHANNEL  ; 进料伺服X轴#3腔放料位SV
D6159 CHANNEL  ; 进料伺服X轴#3腔放料位SV
D616 CHANNEL  ; #2-2电池抽气时间（S_UInt）
D6160 CHANNEL  ; 进料伺服X轴#1夹爪扫码NG放料位SV
D6161 CHANNEL  ; 进料伺服X轴#1夹爪扫码NG放料位SV
D6162 CHANNEL  ; 进料伺服X轴#2夹爪扫码NG放料位SV
D6163 CHANNEL  ; 进料伺服X轴#2夹爪扫码NG放料位SV
D6164 CHANNEL  ; 进料伺服X轴#1夹爪配对取放料位SV
D6165 CHANNEL  ; 进料伺服X轴#1夹爪配对取放料位SV
D6166 CHANNEL  ; 进料伺服X轴#2夹爪配对取放料位SV
D6167 CHANNEL  ; 进料伺服X轴#2夹爪配对取放料位SV
D6168 CHANNEL  ; 进料伺服X轴#1腔有料检测位SV
D6169 CHANNEL  ; 进料伺服X轴#1腔有料检测位SV
D6170 CHANNEL  ; 进料伺服X轴#2腔有料检测位SV
D6171 CHANNEL  ; 进料伺服X轴#2腔有料检测位SV
D6172 CHANNEL  ; 进料伺服X轴#3腔有料检测位SV
D6173 CHANNEL  ; 进料伺服X轴#3腔有料检测位SV
D6174 CHANNEL  ; 进料伺服X轴#4腔放料位SV
D618 CHANNEL  ; #2-2电池真空压力（Pa_Float）
D620 CHANNEL  ; #2-2泄氦后真空度
D6200 CHANNEL  ; 进料伺服Z轴加速比率
D6201 CHANNEL  ; 进料伺服Z轴减速比率
D6202 CHANNEL  ; 进料伺服Z轴目标速度
D6203 CHANNEL  ; 进料伺服Z轴目标速度
D6205 CHANNEL  ; 进料伺服Z轴目标位置
D6206 CHANNEL  ; 进料伺服Z轴启动频率
D6207 CHANNEL  ; 进料伺服Z轴启动频率
D622 CHANNEL  ; #2-2电池泄漏量（Pa_Float）
D6222 CHANNEL  ; 进料伺服Z轴JOG运行速度
D6231 CHANNEL  ; 进料伺服Z轴JOG停止速度
D6232 CHANNEL  ; 进料伺服Z轴JOG停止速度
D6240 CHANNEL  ; 进料伺服Z轴当前位置
D6241 CHANNEL  ; 进料伺服Z轴当前位置
D6242 CHANNEL  ; 进料伺服Z轴当前速度
D6243 CHANNEL  ; 进料伺服Z轴当前速度
D6254 CHANNEL  ; 进料伺服Z轴#1腔放料位SV1
D6255 CHANNEL  ; 进料伺服Z轴#1腔放料位SV1
D6256 CHANNEL  ; 进料伺服Z轴#2腔放料位SV1
D6257 CHANNEL  ; 进料伺服Z轴#2腔放料位SV1
D6258 CHANNEL  ; 进料伺服Z轴#3腔放料位SV1
D6259 CHANNEL  ; 进料伺服Z轴#3腔放料位SV1
D6260 CHANNEL  ; 进料伺服Z轴#4腔放料位SV1
D630 CHANNEL  ; #2-2腔体自检抽气时间（S_UInt）
D6300 CHANNEL  ; 进料伺服Z轴加速比率SV
D6301 CHANNEL  ; 进料伺服Z轴减速比率SV
D6302 CHANNEL  ; 进料伺服Z轴目标速度SV
D6303 CHANNEL  ; 进料伺服Z轴目标速度SV
D6306 CHANNEL  ; 进料伺服Z轴启动频率SV
D6307 CHANNEL  ; 进料伺服Z轴启动频率SV
D632 CHANNEL  ; #2-2腔体自检前保压时间（S_UInt）
D6320 CHANNEL  ; 进料伺服Z轴JOG运行/停止加减速SV
D6321 CHANNEL  ; 进料伺服Z轴JOG运行速度SV
D6322 CHANNEL  ; 进料伺服Z轴JOG运行速度SV
D6331 CHANNEL  ; 进料伺服Z轴JOG停止速度SV
D6332 CHANNEL  ; 进料伺服Z轴JOG停止速度SV
D634 CHANNEL  ; #2-2腔体自检保压时间（S_UInt）
D6350 CHANNEL  ; 进料伺服Z轴待料位SV
D6351 CHANNEL  ; 进料伺服Z轴待料位SV
D6352 CHANNEL  ; 进料伺服Z轴取料位SV
D6353 CHANNEL  ; 进料伺服Z轴取料位SV
D6354 CHANNEL  ; 进料伺服Z轴#1腔放料位SV
D6355 CHANNEL  ; 进料伺服Z轴#1腔放料位SV
D6356 CHANNEL  ; 进料伺服Z轴#2腔放料位SV
D6357 CHANNEL  ; 进料伺服Z轴#2腔放料位SV
D6358 CHANNEL  ; 进料伺服Z轴#3腔放料位SV
D6359 CHANNEL  ; 进料伺服Z轴#3腔放料位SV
D636 CHANNEL  ; #2-2腔体自检保压前真空（Pa_Float）
D6360 CHANNEL  ; 进料伺服Z轴#1夹爪扫码NG放料位SV
D6361 CHANNEL  ; 进料伺服Z轴#1夹爪扫码NG放料位SV
D6362 CHANNEL  ; 进料伺服Z轴#2夹爪扫码NG放料位SV
D6363 CHANNEL  ; 进料伺服Z轴#2夹爪扫码NG放料位SV
D6364 CHANNEL  ; 进料伺服Z轴#1夹爪配对取放料位SV
D6365 CHANNEL  ; 进料伺服Z轴#1夹爪配对取放料位SV
D6366 CHANNEL  ; 进料伺服Z轴#2夹爪配对取放料位SV
D6367 CHANNEL  ; 进料伺服Z轴#2夹爪配对取放料位SV
D6368 CHANNEL  ; 进料伺服Z轴#4腔放料位SV
D638 CHANNEL  ; #2-2腔体自检保压后真空（Pa_Float）
D64 CHANNEL  ; 批次号设定长度
D640 CHANNEL  ; #2-2腔体自检泄漏量（Pa_Float）
D6403 CHANNEL  ; 出料伺服X轴目标速度
D6405 CHANNEL  ; 出料伺服X轴目标位置
D6406 CHANNEL  ; 出料伺服X轴启动频率
D6407 CHANNEL  ; 出料伺服X轴启动频率
D6410 CHANNEL  ; 出料伺服X轴自动加速比率SV
D6411 CHANNEL  ; 出料伺服X轴自动减速比率SV
D6412 CHANNEL  ; 出料伺服X轴自动目标速度SV
D6416 CHANNEL  ; 出料伺服X轴自动启动频率
D642 CHANNEL  ; #2-2腔体自检结果（1-OK，2-NG,3-抽真空NG）
D6420 CHANNEL  ; 出料伺服X轴JOG运行加减速
D6421 CHANNEL  ; 出料伺服X轴JOG运行速度
D6422 CHANNEL  ; 出料伺服X轴JOG运行速度
D6430 CHANNEL  ; 出料伺服X轴JOG停止加减速
D6431 CHANNEL  ; 出料伺服X轴JOG停止速度
D6432 CHANNEL  ; 出料伺服X轴JOG停止速度
D6440 CHANNEL  ; 出料伺服X轴当前位置
D6441 CHANNEL  ; 出料伺服X轴当前位置
D6442 CHANNEL  ; 出料伺服X轴当前速度
D6443 CHANNEL  ; 出料伺服X轴当前速度
D6450 CHANNEL  ; 下料Z模组当前位置（CAENNEL）
D6500 CHANNEL  ; 出料伺服X轴加速比率SV
D6501 CHANNEL  ; 出料伺服X轴减速比率SV
D6502 CHANNEL  ; 出料伺服X轴目标速度SV
D6503 CHANNEL  ; 出料伺服X轴目标速度SV
D6504 CHANNEL  ; 出料伺服X轴目标位置（CHANNEL)
D6506 CHANNEL  ; 出料伺服X轴启动频率SV
D6507 CHANNEL  ; 出料伺服X轴启动频率SV
D6520 CHANNEL  ; 出料伺服X轴JOG运行/停止加减速SV
D6521 CHANNEL  ; 出料伺服X轴JOG运行速度SV
D6522 CHANNEL  ; 出料伺服X轴JOG运行速度SV
D6530 CHANNEL  ; 出料伺服X轴JOG停止加减速
D6531 CHANNEL  ; 出料伺服X轴JOG停止速度SV
D6532 CHANNEL  ; 出料伺服X轴JOG停止速度SV
D6540 CHANNEL  ; 出料伺服X轴当前位置（CAENNEL）
D6542 CHANNEL  ; 出料伺服X轴当前速度
D6544 CHANNEL  ; 出料伺服X轴当前位置（REAL）（mm）
D6550 CHANNEL  ; 出料伺服X轴出料OK位（设定）
D6552 CHANNEL  ; 出料伺服X轴#1腔取料位SV
D6553 CHANNEL  ; 出料伺服X轴放料位SV
D6554 CHANNEL  ; 出料伺服X轴#2腔取料位SV
D6555 CHANNEL  ; 出料伺服X轴#1腔取料位SV
D6556 CHANNEL  ; 出料伺服X轴#3腔取料位SV
D6557 CHANNEL  ; 出料伺服X轴#2腔取料位SV
D6558 CHANNEL  ; 出料伺服X轴NG缓存放料位SV
D6559 CHANNEL  ; 出料伺服X轴#3腔取料位SV
D6560 CHANNEL  ; 出料伺服X轴
D6561 CHANNEL  ; 出料伺服X轴#1夹爪氦检NG放料位SV
D6562 CHANNEL  ; 出料伺服X轴复测配对取料位SV
D6563 CHANNEL  ; 出料伺服X轴#2夹爪氦检NG放料位SV
D6564 CHANNEL  ; 出料伺服X轴
D6565 CHANNEL  ; 出料伺服X轴#1夹爪配对取放料位SV
D6566 CHANNEL  ; 出料伺服X轴#4腔体取放料位SV
D6567 CHANNEL  ; 出料伺服X轴#2夹爪配对取放料位SV
D6568 CHANNEL  ; 出料伺服X轴#4腔取料位SV
D66 CHANNEL  ; 设定条码长度
D660 CHANNEL  ; #2-2氦检时真空值（标漏）
D6603 CHANNEL  ; 出料伺服Z轴目标速度
D6605 CHANNEL  ; 出料伺服Z轴目标位置
D6606 CHANNEL  ; 出料伺服Z轴启动频率
D6607 CHANNEL  ; 出料伺服Z轴启动频率
D6610 CHANNEL  ; 出料伺服Z轴自动加速比率SV
D6611 CHANNEL  ; 出料伺服Z轴自动减速比率SV
D6612 CHANNEL  ; 出料伺服Z轴自动目标速度SV
D6616 CHANNEL  ; 出料伺服Z轴自动启动频率
D662 CHANNEL  ; #2-2氦检漏率（标漏）
D6620 CHANNEL  ; 出料伺服Z轴JOG运行加减速
D6621 CHANNEL  ; 出料伺服Z轴JOG运行速度
D6622 CHANNEL  ; 出料伺服Z轴JOG运行速度
D6630 CHANNEL  ; 出料伺服Z轴JOG停止加减速
D6631 CHANNEL  ; 出料伺服Z轴JOG停止速度
D6632 CHANNEL  ; 出料伺服Z轴JOG停止速度
D6640 CHANNEL  ; 出料伺服Z轴当前位置
D6641 CHANNEL  ; 出料伺服Z轴当前位置
D6642 CHANNEL  ; 出料伺服Z轴当前速度
D6643 CHANNEL  ; 出料伺服Z轴当前速度
D6650 CHANNEL  ; 出料伺服X轴出料OK位
D6654 CHANNEL  ; 出料伺服Z轴#1腔取料位SV1
D6655 CHANNEL  ; 出料伺服Z轴#1腔取料位SV1
D6656 CHANNEL  ; 出料伺服Z轴#2腔取料位SV1
D6657 CHANNEL  ; 出料伺服Z轴#2腔取料位SV1
D6658 CHANNEL  ; 出料伺服Z轴#3腔取料位SV1
D6659 CHANNEL  ; 出料伺服Z轴#3腔取料位SV1
D6660 CHANNEL  ; 出料伺服Z轴#4腔取料位SV1
D6700 CHANNEL  ; 出料伺服Z轴加速比率SV
D6701 CHANNEL  ; 出料伺服Z轴减速比率SV
D6702 CHANNEL  ; 出料伺服Z轴目标速度SV
D6703 CHANNEL  ; 出料伺服Z轴目标速度SV
D6704 CHANNEL  ; 出料伺服Z轴目标位置(CHANNEL）
D6706 CHANNEL  ; 出料伺服Z轴启动频率SV
D6707 CHANNEL  ; 出料伺服Z轴启动频率SV
D6720 CHANNEL  ; 出料伺服Z轴JOG运行/停止加减速SV
D6721 CHANNEL  ; 出料伺服Z轴JOG运行速度SV
D6722 CHANNEL  ; 出料伺服Z轴JOG运行速度SV
D6730 CHANNEL  ; 出料伺服Z轴JOG停止加减速
D6731 CHANNEL  ; 出料伺服Z轴JOG停止速度SV
D6732 CHANNEL  ; 出料伺服Z轴JOG停止速度SV
D6742 CHANNEL  ; 出料伺服Z轴当前速度
D6750 CHANNEL  ; 出料伺服Z轴待料位SV
D6751 CHANNEL  ; 出料伺服Z轴待料位SV
D6752 CHANNEL  ; 出料伺服Z轴放料位SV
D6753 CHANNEL  ; 出料伺服Z轴放料位SV
D6754 CHANNEL  ; 出料伺服Z轴#1腔取料位SV
D6755 CHANNEL  ; 出料伺服Z轴#1腔取料位SV
D6756 CHANNEL  ; 出料伺服Z轴#2腔取料位SV
D6757 CHANNEL  ; 出料伺服Z轴#2腔取料位SV
D6758 CHANNEL  ; 出料伺服Z轴#3腔取料位SV
D6759 CHANNEL  ; 出料伺服Z轴#3腔取料位SV
D6760 CHANNEL  ; 出料伺服Z轴氦检NG缓存放料位SV
D6761 CHANNEL  ; 出料伺服Z轴#1夹爪氦检NG放料位SV
D6762 CHANNEL  ; 出料伺服Z轴位SV
D6763 CHANNEL  ; 出料伺服Z轴#2夹爪氦检NG放料位SV
D6764 CHANNEL  ; 出料伺服Z轴缓存配对取料位SV
D6765 CHANNEL  ; 出料伺服Z轴#1夹爪配对取放料位SV
D6766 CHANNEL  ; 出料伺服Z轴#位SV
D6767 CHANNEL  ; 出料伺服Z轴#2夹爪配对取放料位SV
D6768 CHANNEL  ; 出料伺服Z轴#4腔取料位SV
D68 CHANNEL  ; 设定条码字长度
D6800 CHANNEL  ; 复测移载伺服X轴加速比率
D6801 CHANNEL  ; 复测移载伺服X轴 减速比率
D6802 CHANNEL  ; 复测移载伺服X轴 速度
D6804 CHANNEL  ; 复测移载伺服X轴目标位置
D6806 CHANNEL  ; 复测移载伺服X轴启动频率
D6820 CHANNEL  ; 复测移载伺服X轴JOG运行加减速
D6821 CHANNEL  ; 复测移载伺服X轴JOG运行速度
D6830 CHANNEL  ; 复测移载伺服X轴JOG停止加减速
D6831 CHANNEL  ; 复测移载伺服X轴JOG停止速度
D6840 CHANNEL  ; 复测移载伺服X轴当前位置
D6842 CHANNEL  ; 复测移载伺服X轴当前速度
D6850 CHANNEL  ; 复测移载伺服X/Z轴急停预留位置
D6902 CHANNEL  ; 复测X轴 自动速度SV
D6921 CHANNEL  ; 复测移载伺服X轴JOG运行速度SV
D6952 CHANNEL  ; 复测移载伺服X轴待料位SV
D6954 CHANNEL  ; 复测移载伺服X轴测试腔体位SV
D6956 CHANNEL  ; 复测移载伺服X轴#1取料位SV
D6958 CHANNEL  ; 复测移载伺服X轴#2取料位SV
D6960 CHANNEL  ; 复测移载伺服X轴#1配对位SV
D6962 CHANNEL  ; 复测移载伺服X轴#2配对位SV
D6964 CHANNEL  ; 复测移载伺服X轴NG放料位SV
D70 CHANNEL  ; 设定条码批次号
D700 CHANNEL  ; #3-2腔体状态（0停用，1待料中，2测试中，3测试完成，4-清氦中）
D7000 CHANNEL  ; 复测移载伺服Z轴加速比率
D7001 CHANNEL  ; 复测移载伺服Z轴减速比率
D7002 CHANNEL  ; 复测移载伺服Z轴速度
D7004 CHANNEL  ; 复测移载伺服Z轴目标位置
D7006 CHANNEL  ; 复测移载伺服Z轴启动频率
D702 CHANNEL  ; #3-2腔体测试漏率（Pa.m3/s_Float）
D7020 CHANNEL  ; 复测移载伺服Z轴JOG运行加减速
D7021 CHANNEL  ; 复测移载伺服Z轴JOG运行速度
D7030 CHANNEL  ; 复测移载伺服Z轴JOG停止加减速
D7031 CHANNEL  ; 复测移载伺服Z轴JOG停止速度
D704 CHANNEL  ; #3-2腔体测试检漏口压力（Pa_Float）
D7040 CHANNEL  ; 复测移载伺服Z轴当前位置
D7042 CHANNEL  ; 复测移载伺服Z轴当前速度
D706 CHANNEL  ; #3-2电池充氦压力（Pa_Float）
D708 CHANNEL  ; #3-2腔体测试结果（1 OK，2腔体泄漏，3气密NG，4注氦超时，5氦检异常，6电池泄漏，7注氦NG，8氦嘴泄漏）
D710 CHANNEL  ; #3-2充氦嘴压力（Pa_Float）
D7102 CHANNEL  ; 复测Z轴 自动速度SV
D712 CHANNEL  ; #3-2腔体抽气时间（S_UInt）
D7121 CHANNEL  ; 复测移载伺服Z轴JOG运行速度SV
D714 CHANNEL  ; #3-2腔体真空压力（Pa_Float）
D7150 CHANNEL  ; 复测移载伺服Z轴待料位SV
D7152 CHANNEL  ; 复测移载伺服Z轴取料位SV
D7154 CHANNEL  ; 复测移载伺服Z轴OK放料位SV
D7156 CHANNEL  ; 复测移载伺服Z轴NG放料位SV
D7158 CHANNEL  ; 复测移载伺服Z轴腔体取放料位SV
D716 CHANNEL  ; #3-2电池抽气时间（S_UInt）
D718 CHANNEL  ; #3-2电池真空压力（Pa_Float）
D720 CHANNEL  ; #3-2泄氦后真空度
D722 CHANNEL  ; #3-2电池泄漏量（Pa_Float）
D730 CHANNEL  ; #3-2腔体自检抽气时间（S_UInt）
D732 CHANNEL  ; #3-2腔体自检前保压时间（S_UInt）
D734 CHANNEL  ; #3-2腔体自检保压时间（S_UInt）
D736 CHANNEL  ; #3-2腔体自检保压前真空（Pa_Float）
D738 CHANNEL  ; #3-2腔体自检保压后真空（Pa_Float）
D740 CHANNEL  ; #3-2腔体自检泄漏量（Pa_Float）
D742 CHANNEL  ; #3-2腔体自检结果（1-OK，2-NG,3-抽真空NG）
D760 CHANNEL  ; #3-2氦检时真空值（标漏）
D762 CHANNEL  ; #3-2氦检漏率（标漏）
D80 CHANNEL  ; 进料#1扫码接收条码长度
D82 CHANNEL  ; 进料#2扫码接收条码长度
D900 CHANNEL  ; #1-1电池真空偏值设定(Float)
D902 CHANNEL  ; #1-1电池实际真空值(Float)
D904 CHANNEL  ; #1-1电池真空模拟量读数(Int)
D910 CHANNEL  ; #1-2电池真空偏值设定(Float)
D912 CHANNEL  ; #1-2电池实际真空值(Float)
D914 CHANNEL  ; #1-2电池真空模拟量读数(Int)
D920 CHANNEL  ; #2-1电池真空偏值设定(Float)
D922 CHANNEL  ; #2-1电池实际真空值(Float)
D924 CHANNEL  ; #2-1电池真空模拟量读数(Int)
D930 CHANNEL  ; #2-2电池真空偏值设定(Float)
D932 CHANNEL  ; #2-2电池实际真空值(Float)
D934 CHANNEL  ; #2-2电池真空模拟量读数(Int)
D940 CHANNEL  ; #3-1电池真空偏值设定(Float)
D942 CHANNEL  ; #3-1电池实际真空值(Float)
D944 CHANNEL  ; #3-1电池真空模拟量读数(Int)
D950 CHANNEL  ; #3-2电池真空偏值设定(Float)
D952 CHANNEL  ; #3-2电池实际真空值(Float)
D954 CHANNEL  ; #3-2电池真空模拟量读数(Int)
D962 CHANNEL  ; #1腔体实际真空值(Float)
D964 CHANNEL  ; #1腔体真空模拟量读数(Int)
D972 CHANNEL  ; #2腔体实际真空值(Float)
D974 CHANNEL  ; #2腔体真空模拟量读数(Int)
D982 CHANNEL  ; #3腔体实际真空值(Float)
D984 CHANNEL  ; #3腔体真空模拟量读数(Int)
D990 CHANNEL  ; 实时漏率（Pa.m3/s_Float）
D992 CHANNEL  ; 实时检漏口压力（Pa_Float）
D994 CHANNEL  ; 泄漏率设定值（Pa.m3/s_Float）
D996 CHANNEL  ; 检漏口压力设定值（Pa_Float）
D998 CHANNEL  ; 清氦漏率设定值（Pa_Float）
E0_0 CHANNEL  ; PC&PLC通讯心跳检测
E0_10 CHANNEL  ; 进料拉带机构#1扫码MES入站就绪通知
E0_1000 CHANNEL  ; 进料#1扫码MES出站读取条码开始字
E0_104 CHANNEL  ; 工艺参数变更通知to pc
E0_1049 CHANNEL  ; 进料#1扫码MES出站读取条码结束字
E0_105 CHANNEL  ; 工艺变更确认
E0_1050 CHANNEL  ; 出料伺服机构#1夹爪MES出站生产数据开始字
E0_1099 CHANNEL  ; 出料伺服机构#1夹爪MES出站生产数据结束字
E0_11 CHANNEL  ; 进料拉带机构#2扫码MES入站就绪通知
E0_1100 CHANNEL  ; 进料#2扫码MES入站读取条码开始字
E0_1149 CHANNEL  ; 进料#2扫码MES入站读取条码结束字
E0_1150 CHANNEL  ; 出料伺服机构#2夹爪MES出站生产数据开始字
E0_1199 CHANNEL  ; 出料伺服机构#2夹爪MES出站生产数据结束字
E0_1200 CHANNEL  ; 复测机械手出料请求
E0_1.00 BOOL  ; 设备上电状态
E0_1.01 BOOL  ; 设备复位状态
E0_1.02 BOOL  ; 设备自动状态
E0_1.03 BOOL  ; 设备停止状态
E0_1.04 BOOL  ; 设备启动状态
E0_1.05 BOOL  ; 设备待料状态
E0_1.06 BOOL  ; 设备手动状态
E0_1.07 BOOL  ; 设备故障状态
E0_1.08 BOOL  ; 设备急停状态
E0_1.09 BOOL  ; 设备关电状态
E0_20 CHANNEL  ; 进料拉带机构#1扫码MES入站就绪确认
E0_2000 CHANNEL  ; 进料#1扫码MES入站读取条码开始字
E0_2049 CHANNEL  ; 进料#1扫码MES入站读取条码结束字
E0_2050 CHANNEL  ; 进料#2扫码MES入站读取条码开始字
E0_2099 CHANNEL  ; 进料#2扫码MES入站读取条码结束字
E0_21 CHANNEL  ; 进料拉带机构#2扫码MES入站就绪确认
E0_300 CHANNEL  ; 泄漏率设定值to pc（Pa.m3/s_Float)to pc
E0_302 CHANNEL  ; 检漏口压力设定值（Pa_Float）to pc
E0_304 CHANNEL  ; 腔体测试设定氦检时间（S_UInt）to pc
E0_306 CHANNEL  ; 腔体测试设定真空阈值（Pa_Float）to pc
E0_308 CHANNEL  ; 电池测试设定真空阈值（Pa_Float）to pc
E0_310 CHANNEL  ; 电池测试设定注氦压力（Pa_Float）to pc
E0_312 CHANNEL  ; 注氦压力上限值（Pa_Float）to pc
E0_314 CHANNEL  ; 注氦压力下限值
E0_316 CHANNEL  ; 腔体测试设定抽真空时间上限（S_UInt）to pc
E0_318 CHANNEL  ; 电池测试设定抽真空时间上限（S_UInt）to pc
E0_320 CHANNEL  ; 腔体测试设定腔体预抽检测时间（S_UInt）to pc
E0_322 CHANNEL  ; 电池测试设定预抽检测压力（Pa_Float）to pc
E0_324 CHANNEL  ; 腔体测试设定清氦压力（Pa_Float）to pc
E0_326 CHANNEL  ; 清氦漏率设定值（Pa_Float）to pc
E0_328 CHANNEL  ; 清氦漏率设定值（Pa_Float）to pc
E0_349 CHANNEL  ; 出料伺服机构#1夹爪MES出站工艺参数结束字
E0_350 CHANNEL  ; 出料伺服机构#2夹爪MES出站工艺参数开始字
E0_399 CHANNEL  ; 出料伺服机构#2夹爪MES出站工艺参数结束字
E0_50 CHANNEL  ; 出料伺服机构#1夹爪MES出站就绪通知
E0_51 CHANNEL  ; 出料伺服机构#2夹爪MES出站就绪通知
E0_52 CHANNEL  ; 复测机械手出站校验通知
E0_60 CHANNEL  ; 出料伺服机构#1夹爪MES出站就绪确认
E0_61 CHANNEL  ; 出料伺服机构#2夹爪MES出站就绪确认
E0_62 CHANNEL  ; 出站就绪确认通知
E0_900 CHANNEL  ; 工站故障
E2_1000 CHANNEL  ; 进料#1扫码条码开始字（传递）
E2_1001 CHANNEL  ; 进料#1扫码条码开始字（传递）
E2_1030 CHANNEL  ; 进料#1扫码条码结束字（传递）
E2_1100 CHANNEL  ; 进料#2扫码条码开始字（传递）
E2_1130 CHANNEL  ; 进料#2扫码条码结束字（传递）
E2_1200 CHANNEL  ; #1进料位条码开始字（传递）
E2_1299 CHANNEL  ; #1进料位数据结束字（传递）
E2_1300 CHANNEL  ; #2进料位条码开始字（传递）
E2_1399 CHANNEL  ; #2进料位数据结束字（传递）
E2_1400 CHANNEL  ; #1进料夹爪条码开始字（传递）
E2_1499 CHANNEL  ; #1进料夹爪数据结束字（传递）
E2_1500 CHANNEL  ; #2进料夹爪条码开始字（传递）
E2_1599 CHANNEL  ; #2进料夹爪数据结束字（传递）
E2_1600 CHANNEL  ; 扫码OK缓存条码开始字（传递）
E2_1699 CHANNEL  ; 扫码OK缓存数据结束字（传递）
E2_1800 CHANNEL  ; #1-1氦检腔条码开始字（传递）
E2_1850 CHANNEL  ; #1-1氦检腔工位开始字（传递）
E2_1899 CHANNEL  ; #1-1氦检腔数据结束字（传递）
E2_1900 CHANNEL  ; #1-2氦检腔条码开始字（传递）
E2_1950 CHANNEL  ; #1-2氦检腔工位开始字（传递）
E2_1999 CHANNEL  ; #1-2氦检腔数据结束字（传递）
E2_2000 CHANNEL  ; #2-1氦检腔条码开始字（传递）
E2_2050 CHANNEL  ; #2-1氦检腔工位开始字（传递）
E2_2099 CHANNEL  ; #2-1氦检腔数据结束字（传递）
E2_2100 CHANNEL  ; #2-2氦检腔条码开始字（传递）
E2_2150 CHANNEL  ; #2-2氦检腔工位开始字（传递）
E2_2199 CHANNEL  ; #2-2氦检腔数据结束字（传递）
E2_2200 CHANNEL  ; #3-1氦检腔条码开始字（传递）
E2_2250 CHANNEL  ; #3-1氦检腔工位开始字（传递）
E2_2299 CHANNEL  ; #3-1氦检腔数据结束字（传递）
E2_2300 CHANNEL  ; #3-2氦检腔条码开始字（传递）
E2_2350 CHANNEL  ; #3-2氦检腔工位开始字（传递）
E2_2399 CHANNEL  ; #3-2氦检腔数据结束字（传递）
E2_2400 CHANNEL  ; #1出料夹爪条码开始字（传递）
E2_2450 CHANNEL  ; #1出料夹爪工位开始字（传递）
E2_2499 CHANNEL  ; #1出料夹爪数据结束字（传递）
E2_2500 CHANNEL  ; #2出料夹爪条码开始字（传递）
E2_2550 CHANNEL  ; #2出料夹爪工位开始字（传递）
E2_2599 CHANNEL  ; #2出料夹爪数据结束字（传递）
E2_2700 CHANNEL  ; #4-1氦检腔条码开始字（传递）
E2_2750 CHANNEL  ; #4-1氦检腔工位开始字（传递）
E2_2800 CHANNEL  ; #4-2氦检腔条码开始字（传递）
E2_2850 CHANNEL  ; #4-2氦检腔工位开始字（传递）
E2_3000 CHANNEL  ; 复测缓存左1位电芯条码50字（#1位）
E2_3050 CHANNEL  ; 复测缓存右1位电芯条码50字（#2位）
E2_3100 CHANNEL  ; 复测缓存左2位电芯条码50字（#1位）
E2_3150 CHANNEL  ; 复测缓存右2位电芯条码50字（#2位）
E2_3200 CHANNEL  ; 复测缓存左3位电芯条码50字（#1位）
E2_3250 CHANNEL  ; 复测缓存右3位电芯条码50字（#2位）
E2_3300 CHANNEL  ; 复测缓存左4位电芯条码50字（#1位）
E2_3350 CHANNEL  ; 复测缓存右4位电芯条码50字（#2位）
E2_3400 CHANNEL  ; OK配对#1位电芯条码50字
E2_3500 CHANNEL  ; OK配对#2位电芯条码50字
E2_3600 CHANNEL  ; 复测夹爪电芯条码50字
E2_3700 CHANNEL  ; 复测腔体电芯条码50字
E2_3750 CHANNEL  ; 复测腔体工位
E2_3752 CHANNEL  ; 复测腔体漏率
E2_3754 CHANNEL  ; 复测腔体检漏口压力
E2_3756 CHANNEL  ; 复测腔体充氦压力
E2_3758 CHANNEL  ; 复测腔体结果
E2_3760 CHANNEL  ; 复测腔体充氦嘴压力
E2_3762 CHANNEL  ; 复测腔体腔体抽真空时间
E2_3764 CHANNEL  ; 复测腔体腔体抽真空度
E2_3766 CHANNEL  ; 复测腔体电池抽真空时间
E2_3768 CHANNEL  ; 复测腔体电池抽真空度
E2_3770 CHANNEL  ; 复测腔体泄氦后真空度
E2_3772 CHANNEL  ; 复测腔体电池泄漏量
H100.00 BOOL  ; #1扫码阻挡气缸缩回位屏蔽
H100.01 BOOL  ; #1扫码阻挡气缸伸出位屏蔽
H100.02 BOOL  ; #1隔离气缸缩回位屏蔽
H100.03 BOOL  ; 0屏蔽
H100.04 BOOL  ; #2扫码阻挡气缸缩回位屏蔽
H100.05 BOOL  ; #2扫码阻挡气缸伸出位屏蔽
H100.06 BOOL  ; #2隔离气缸缩回位屏蔽
H100.07 BOOL  ; 0屏蔽
H100.08 BOOL  ; #1进料夹爪夹紧位屏蔽
H100.09 BOOL  ; #1进料夹爪松开位屏蔽
H100.10 BOOL  ; #2进料夹爪夹紧位屏蔽
H100.11 BOOL  ; #2进料夹爪松开位屏蔽
H100.12 BOOL  ; 进料夹爪变距气缸伸出位屏蔽
H100.13 BOOL  ; 进料夹爪变距气缸缩回位屏蔽
H100.14 BOOL  ; #1出料夹爪夹紧位屏蔽
H100.15 BOOL  ; #1出料夹爪松开位屏蔽
H101.00 BOOL  ; #2出料夹爪夹紧位屏蔽
H101.01 BOOL  ; #2出料夹爪松开位屏蔽
H101.02 BOOL  ; 出料夹爪变距气缸伸出位屏蔽
H101.03 BOOL  ; 出料夹爪变距气缸缩回位屏蔽
H101.04 BOOL  ; #1腔体平移一级气缸缩回位屏蔽
H101.05 BOOL  ; #1腔体平移一级气缸伸出位屏蔽
H101.06 BOOL  ; #1腔体平移二级气缸缩回位屏蔽
H101.07 BOOL  ; #1腔体平移二级气缸伸出位屏蔽
H101.08 BOOL  ; #1腔体顶伸气缸上升位屏蔽
H101.09 BOOL  ; #1腔体顶伸气缸下降位屏蔽
H101.10 BOOL  ; #1腔体氦检阀开到位屏蔽
H101.11 BOOL  ; #1腔体氦检阀关到位屏蔽
H101.12 BOOL  ; 0屏蔽
H101.13 BOOL  ; 0屏蔽
H101.14 BOOL  ; 0屏蔽
H101.15 BOOL  ; 0屏蔽
H102.00 BOOL  ; 0屏蔽
H102.01 BOOL  ; #2腔体平移一级气缸缩回位屏蔽
H102.02 BOOL  ; #2腔体平移一级气缸伸出位屏蔽
H102.03 BOOL  ; #2腔体平移二级气缸缩回位屏蔽
H102.04 BOOL  ; #2腔体平移二级气缸伸出位屏蔽
H102.05 BOOL  ; #2腔体顶伸气缸上升位屏蔽
H102.06 BOOL  ; #2腔体顶伸气缸下降位屏蔽
H102.07 BOOL  ; #2腔体氦检阀开到位屏蔽
H102.08 BOOL  ; #2腔体氦检阀关到位屏蔽
H102.09 BOOL  ; 0屏蔽
H102.10 BOOL  ; 0屏蔽
H102.11 BOOL  ; 0屏蔽
H102.12 BOOL  ; 0屏蔽
H102.13 BOOL  ; 0屏蔽
H102.14 BOOL  ; #3腔体平移一级气缸缩回位屏蔽
H102.15 BOOL  ; #3腔体平移一级气缸伸出位屏蔽
H103.00 BOOL  ; #3腔体平移二级气缸缩回位屏蔽
H103.01 BOOL  ; #3腔体平移二级气缸伸出位屏蔽
H103.02 BOOL  ; #3腔体顶伸气缸上升位屏蔽
H103.03 BOOL  ; #3腔体顶伸气缸下降位屏蔽
H103.04 BOOL  ; #3腔体氦检阀开到位屏蔽
H103.05 BOOL  ; #3腔体氦检阀关到位屏蔽
H103.06 BOOL  ; 氦检仪准备好了信号屏蔽
H103.07 BOOL  ; 氦检仪故障信号屏蔽
H103.08 BOOL  ; 0屏蔽
H103.09 BOOL  ; 0屏蔽
H103.10 BOOL  ; 0屏蔽
H103.11 BOOL  ; 进料伺服X轴准备好了信号屏蔽
H103.12 BOOL  ; 进料伺服X轴故障信号屏蔽
H103.13 BOOL  ; 进料伺服Z轴准备好了信号屏蔽
H103.14 BOOL  ; 进料伺服Z轴故障信号屏蔽
H103.15 BOOL  ; 0屏蔽
H104.00 BOOL  ; 出料伺服X轴准备好了信号屏蔽
H104.01 BOOL  ; 出料伺服X轴故障信号屏蔽
H104.02 BOOL  ; 出料伺服Z轴准备好了信号屏蔽
H104.03 BOOL  ; 出料伺服Z轴故障信号屏蔽
H104.04 BOOL  ; 0屏蔽
H104.05 BOOL  ; 腔体抽真空泵运行信号屏蔽
H104.06 BOOL  ; 腔体抽真空泵过载信号屏蔽
H104.07 BOOL  ; 氦检前置泵运行信号屏蔽
H104.08 BOOL  ; 氦检前置泵过载信号屏蔽
H104.09 BOOL  ; 启动按钮屏蔽
H104.10 BOOL  ; 停止按钮屏蔽
H104.11 BOOL  ; 复位按钮屏蔽
H104.12 BOOL  ; 急停按钮屏蔽
H104.13 BOOL  ; 手自动选择屏蔽
H104.14 BOOL  ; #1进料夹爪防下坠感应屏蔽
H104.15 BOOL  ; #2进料夹爪防下坠感应屏蔽
H105.00 BOOL  ; #1出料夹爪防下坠感应屏蔽
H105.01 BOOL  ; #2出料夹爪防下坠感应屏蔽
H105.02 BOOL  ; 0屏蔽
H105.03 BOOL  ; 进料对接输入屏蔽
H105.04 BOOL  ; 出料对接输入屏蔽
H105.05 BOOL  ; 0屏蔽
H105.06 BOOL  ; 0屏蔽
H105.07 BOOL  ; 设备总气压信号屏蔽
H105.08 BOOL  ; #1来料位有料感应屏蔽
H105.09 BOOL  ; #2来料位有料感应屏蔽
H105.10 BOOL  ; #1隔离位有料感应屏蔽
H105.11 BOOL  ; #2隔离位有料感应屏蔽
H105.12 BOOL  ; #1扫码位有料感应屏蔽
H105.13 BOOL  ; #2扫码位有料感应屏蔽
H105.14 BOOL  ; #1-1进料位有料感应屏蔽
H105.15 BOOL  ; #1-2进料位有料感应屏蔽
H106.00 BOOL  ; #2-1进料位有料感应屏蔽
H106.01 BOOL  ; #2-2进料位有料感应屏蔽
H106.02 BOOL  ; 进料夹爪柔性感应屏蔽
H106.03 BOOL  ; 出料夹爪柔性感应屏蔽
H106.04 BOOL  ; #1进料夹爪对应腔体有料感应屏蔽
H106.05 BOOL  ; #2进料夹爪对应腔体有料感应屏蔽
H106.06 BOOL  ; 扫码NG放料#1位有料感应屏蔽
H106.07 BOOL  ; 扫码NG放料#2位有料感应屏蔽
H106.08 BOOL  ; 扫码NG料满位有料感应屏蔽
H106.09 BOOL  ; 进料配对位有料感应屏蔽
H106.10 BOOL  ; 出料配对位有料感应屏蔽
H106.11 BOOL  ; 氦检NG放料#1位有料感应屏蔽
H106.12 BOOL  ; 氦检NG放料#2位有料感应屏蔽
H106.13 BOOL  ; 氦检NG料满位有料感应屏蔽
H106.14 BOOL  ; #1-1出料位有料感应屏蔽
H106.15 BOOL  ; #1-2出料位有料感应屏蔽
H107.00 BOOL  ; #2-1出料位有料感应屏蔽
H107.01 BOOL  ; #2-2出料位有料感应屏蔽
H107.02 BOOL  ; #1门磁开关屏蔽
H107.03 BOOL  ; #2门磁开关屏蔽
H107.04 BOOL  ; #3门磁开关屏蔽
H107.05 BOOL  ; #4门磁开关屏蔽
H107.06 BOOL  ; #5门磁开关屏蔽
H107.07 BOOL  ; #6门磁开关屏蔽
H107.08 BOOL  ; #7门磁开关屏蔽
H107.09 BOOL  ; #8门磁开关屏蔽
H107.10 BOOL  ; #9门磁开关屏蔽
H107.11 BOOL  ; #10门磁开关屏蔽
H107.12 BOOL  ; #11门磁开关屏蔽
H107.13 BOOL  ; #12门磁开关屏蔽
H107.14 BOOL  ; #13门磁开关屏蔽
H107.15 BOOL  ; #14门磁开关屏蔽
H10.00 BOOL  ; #1扫码阻挡有料记忆
H10.01 BOOL  ; #1进料位有料记忆
H10.02 BOOL  ; #1进料位有OK料记忆
H10.03 BOOL  ; #1进料位有NG料记忆
H10.04 BOOL  ; #1扫码阻挡有OK料记忆
H10.05 BOOL  ; #1扫码阻挡有NG料记忆
H10.06 BOOL  ; #1扫码阻挡扫码完成记忆
H10.07 BOOL  ; #1扫码阻挡扫码OK料记忆
H10.08 BOOL  ; #1扫码阻挡扫码NG料记忆
H10.09 BOOL  ; #1扫码阻挡MES校验完成记忆
H10.10 BOOL  ; #1扫码阻挡MES校验OK料记忆
H10.11 BOOL  ; #1扫码阻挡MES校验NG料记忆
H11.00 BOOL  ; #1隔离气缸放料中记忆
H11.01 BOOL  ; #1扫码阻挡气缸放料中记忆
H12.00 BOOL  ; #2扫码阻挡有料记忆
H12.01 BOOL  ; #2进料位有料记忆
H12.02 BOOL  ; #2进料位有OK料记忆
H12.03 BOOL  ; #2进料位有NG料记忆
H12.04 BOOL  ; #2扫码阻挡有OK料记忆
H12.05 BOOL  ; #2扫码阻挡有NG料记忆
H12.06 BOOL  ; #2扫码阻挡扫码完成记忆
H12.07 BOOL  ; #2扫码阻挡扫码OK料记忆
H12.08 BOOL  ; #2扫码阻挡扫码NG料记忆
H12.09 BOOL  ; #2扫码阻挡MES校验完成记忆
H12.10 BOOL  ; #2扫码阻挡MES校验OK料记忆
H12.11 BOOL  ; #2扫码阻挡MES校验NG料记忆
H130.04 BOOL  ; #4腔体平移一级气缸缩回位屏蔽
H130.05 BOOL  ; #4腔体平移一级气缸伸出位屏蔽
H130.06 BOOL  ; #4腔体平移二级气缸缩回位屏蔽
H130.07 BOOL  ; #4腔体平移二级气缸伸出位屏蔽
H130.08 BOOL  ; #4腔体顶伸气缸上升位屏蔽
H130.09 BOOL  ; #4腔体顶伸气缸下降位屏蔽
H130.10 BOOL  ; #4腔体氦检阀开到位屏蔽
H130.11 BOOL  ; #4腔体氦检阀关到位屏蔽
H131.00 BOOL  ; 复测夹爪气缸夹紧位屏蔽
H131.01 BOOL  ; 复测夹爪气缸松开位屏蔽
H131.02 BOOL  ; 复检夹爪柔性感应屏蔽
H131.03 BOOL  ; 复测腔体移栽气缸缩回位屏蔽
H131.04 BOOL  ; 复测腔体移栽气缸伸出位屏蔽
H131.05 BOOL  ; 复测腔体顶升气缸缩回位屏蔽
H131.06 BOOL  ; 复测腔体顶升气缸伸出位屏蔽
H131.07 BOOL  ; 复测腔体氦检阀开到位屏蔽
H131.08 BOOL  ; 复测腔体氦检阀关到位屏蔽
H131.09 BOOL  ; 复测腔体感应有料感应屏蔽
H131.10 BOOL  ; 0屏蔽
H131.11 BOOL  ; 出料配对位有料感应2屏蔽
H131.12 BOOL  ; 0屏蔽
H131.13 BOOL  ; 0屏蔽
H131.14 BOOL  ; 0屏蔽
H131.15 BOOL  ; 0屏蔽
H132.00 BOOL  ; 腔体抽真空泵M2运行信号屏蔽
H132.01 BOOL  ; 腔体抽真空泵M2过载信号屏蔽
H132.02 BOOL  ; 测伺服X轴准备好信号屏蔽
H132.03 BOOL  ; 复测伺服X轴故障信号屏蔽
H132.04 BOOL  ; 复测伺服Z轴准备好信号屏蔽
H132.05 BOOL  ; 复测伺服Z轴故障信号屏蔽
H132.06 BOOL  ; 0屏蔽
H132.07 BOOL  ; 0屏蔽
H132.08 BOOL  ; 0屏蔽
H132.09 BOOL  ; 0屏蔽
H132.10 BOOL  ; 设备真空压力信号#1屏蔽
H132.11 BOOL  ; 设备真空压力信号#2屏蔽
H132.12 BOOL  ; 设备氦气压力信号#1屏蔽
H132.13 BOOL  ; 设备氦气压力信号#2屏蔽
H132.14 BOOL  ; 设备注氦压力调节阀#1屏蔽
H132.15 BOOL  ; 设备注氦压力调节阀#2屏蔽
H133.00 BOOL  ; 复测缓存拨料气缸缩回位屏蔽
H133.01 BOOL  ; 复测缓存拨料气缸伸出位屏蔽
H133.02 BOOL  ; 复测缓存顶升气缸缩回位屏蔽
H133.03 BOOL  ; 复测缓存顶升气缸伸出位屏蔽
H133.04 BOOL  ; 复测缓存#1有料感应1屏蔽
H133.05 BOOL  ; 复测缓存#1有料感应2屏蔽
H133.06 BOOL  ; 复测缓存#1有料感应3屏蔽
H133.07 BOOL  ; 复测缓存#1有料感应4屏蔽
H133.08 BOOL  ; 复测缓存#2有料感应1屏蔽
H133.09 BOOL  ; 复测缓存#2有料感应2屏蔽
H133.10 BOOL  ; 复测缓存#2有料感应3屏蔽
H133.11 BOOL  ; 复测缓存#2有料感应4屏蔽
H13.00 BOOL  ; #2隔离气缸放料中记忆
H13.01 BOOL  ; #2扫码阻挡气缸放料中记忆
H15.00 BOOL  ; 扫码NG放料位有料记忆
H17.00 BOOL  ; 氦检NG放料位有料记忆
H20.00 BOOL  ; #1进料夹爪有料记忆
H20.01 BOOL  ; #2进料夹爪有料记忆
H20.02 BOOL  ; 进料配对位有料记忆
H20.03 BOOL  ; #1进料夹爪有OK料记忆
H20.04 BOOL  ; #1进料夹爪有NG料记忆
H20.05 BOOL  ; #2进料夹爪有OK料记忆
H20.06 BOOL  ; #2进料夹爪有NG料记忆
H24.00 BOOL  ; 进料伺服X轴回原点记忆
H24.01 BOOL  ; 进料伺服Z轴回原点记Z忆
H24.02 BOOL  ; 出料伺服X轴回原点记忆
H24.03 BOOL  ; 出料伺服Z轴回原点记忆
H25.00 BOOL  ; #1-1腔体有料记忆
H25.01 BOOL  ; #1-2腔体有料记忆
H25.02 BOOL  ; #1-1腔体有OK料记忆
H25.03 BOOL  ; #1-1腔体有NG料记忆
H25.04 BOOL  ; #1-2腔体有OK料记忆
H25.05 BOOL  ; #1-2腔体有NG料记忆
H25.06 BOOL  ; #1-1腔体测试完成记忆
H25.07 BOOL  ; #1-2腔体测试完成记忆
H26.00 BOOL  ; #1-1电池泄漏
H26.01 BOOL  ; #1-2电池泄漏
H26.02 BOOL  ; #1-1电池注氦超时
H26.03 BOOL  ; #1-2电池注氦超时
H26.04 BOOL  ; #1-1腔体抽真空NG
H26.05 BOOL  ; #1-2腔体抽真空NG
H26.06 BOOL  ; #1-1腔体氦检时腔体压力过高
H26.07 BOOL  ; #1-2腔体氦检时腔体压力过高
H26.08 BOOL  ; #1-1注氦超限
H26.09 BOOL  ; #1-2注氦超限
H27.00 BOOL  ; #1腔体有清氦需求
H27.05 BOOL  ; 腔体有复测需求
H27.10 BOOL  ; #1-1腔体清氦失败，重新进行清氦流程
H30.00 BOOL  ; #2-1腔体有料记忆
H30.01 BOOL  ; #2-2腔体有料记忆
H30.02 BOOL  ; #2-1腔体有OK料记忆
H30.03 BOOL  ; #2-1腔体有NG料记忆
H30.04 BOOL  ; #2-2腔体有OK料记忆
H30.05 BOOL  ; #2-2腔体有NG料记忆
H30.06 BOOL  ; #2-1腔体测试完成记忆
H30.07 BOOL  ; #2-2腔体测试完成记忆
H31.00 BOOL  ; #2-1电池泄漏
H31.01 BOOL  ; #2-2电池泄漏
H31.02 BOOL  ; #2-1电池注氦超时
H31.03 BOOL  ; #2-2电池注氦超时
H31.04 BOOL  ; #2-1腔体抽真空NG
H31.05 BOOL  ; #2-2腔体抽真空NG
H31.06 BOOL  ; #2-1腔体氦检时腔体压力过高
H31.07 BOOL  ; #2-2腔体氦检时腔体压力过高
H31.08 BOOL  ; #2-1注氦超限
H31.09 BOOL  ; #2-2注氦超限
H32.00 BOOL  ; #2腔体有清氦需求
H32.05 BOOL  ; 腔体有复测需求
H32.10 BOOL  ; #2-1腔体清氦失败，重新进行清氦流程
H35.00 BOOL  ; #3-1腔体有料记忆
H35.01 BOOL  ; #3-2腔体有料记忆
H35.02 BOOL  ; #3-1腔体有OK料记忆
H35.03 BOOL  ; #3-1腔体有NG料记忆
H35.04 BOOL  ; #3-2腔体有OK料记忆
H35.05 BOOL  ; #3-2腔体有NG料记忆
H35.06 BOOL  ; #3-1腔体测试完成记忆
H35.07 BOOL  ; #3-2腔体测试完成记忆
H36.00 BOOL  ; #3-1电池泄漏
H36.01 BOOL  ; #3-2电池泄漏
H36.02 BOOL  ; #3-1电池注氦超时
H36.03 BOOL  ; #3-2电池注氦超时
H36.04 BOOL  ; #3-1腔体抽真空NG
H36.05 BOOL  ; #3-2腔体抽真空NG
H36.06 BOOL  ; #3-1腔体氦检时腔体压力过高
H36.07 BOOL  ; #3-2腔体氦检时腔体压力过高
H36.08 BOOL  ; #3-1注氦超限
H36.09 BOOL  ; #3-2注氦超限
H37.00 BOOL  ; #3腔体有清氦需求
H37.05 BOOL  ; 腔体有复测需求
H37.10 BOOL  ; #3-1腔体清氦失败，重新进行清氦流程
H40.00 BOOL  ; #1出料夹爪有料记忆
H40.01 BOOL  ; #2出料夹爪有料记忆
H40.02 BOOL  ; 出料配对位有料记忆
H40.03 BOOL  ; #1出料夹爪有OK料记忆
H40.04 BOOL  ; #1出料夹爪有NG料记忆
H40.05 BOOL  ; #2出料夹爪有OK料记忆
H40.06 BOOL  ; #2出料夹爪有NG料记忆
H40.07 BOOL  ; #1出料夹爪MES校验完成记忆
H40.08 BOOL  ; #2出料夹爪MES校验完成记忆
H40.15 BOOL  ; 出料变距缩回记忆
H41.00 BOOL  ; 1#取料完成
H41.01 BOOL  ; 2#取料完成
H41.02 BOOL  ; 3#取料完成
H41.03 BOOL  ; 1#放NG，2#放缓存
H41.04 BOOL  ; 1#放NG，1#取缓存
H41.05 BOOL  ; 2#放NG,1#放缓存
H41.06 BOOL  ; 2#放NG,2#取缓存
H41.07 BOOL  ; 4#取料完成
H43.00 BOOL  ; 1#腔体下料需求
H43.01 BOOL  ; 2#腔体下料需求
H43.02 BOOL  ; 3#腔体下料需求
H43.03 BOOL  ; 4#腔体下料需求
H43.04 BOOL  ; 出料机械手放NG料需求
H43.05 BOOL  ; 出料机械手去OK配对位需求
H44.00 BOOL  ; 出料伺服X轴回原点记忆
H44.01 BOOL  ; 出料伺服Z轴回原点记忆
H45.00 BOOL  ; #4-1腔体有料记忆
H45.01 BOOL  ; #4-2腔体有料记忆
H45.02 BOOL  ; #4-1腔体有OK料记忆
H45.03 BOOL  ; #4-1腔体有NG料记忆
H45.04 BOOL  ; #4-2腔体有OK料记忆
H45.05 BOOL  ; #4-2腔体有NG料记忆
H45.06 BOOL  ; #4-1腔体测试完成记忆
H45.07 BOOL  ; #4-2腔体测试完成记忆
H46 CHANNEL  ; $?St$Bk?_#[192] / $?St$Bk?_#[192]
H46.00 BOOL  ; #4-1电池泄漏
H46.01 BOOL  ; #4-2电池泄漏
H46.02 BOOL  ; #4-1电池注氦超时
H46.03 BOOL  ; #4-2电池注氦超时
H46.04 BOOL  ; #4-1腔体抽真空NG
H46.05 BOOL  ; #4-2腔体抽真空NG
H46.06 BOOL  ; #4-1腔体氦检时腔体压力过高
H46.07 BOOL  ; #4-2腔体氦检时腔体压力过高
H46.08 BOOL  ; #4-1注氦超限
H46.09 BOOL  ; #4-2注氦超限
H47.00 BOOL  ; #4腔体有清氦需求
H47.05 BOOL  ; 腔体有复测需求
H47.10 BOOL  ; #4-1腔体清氦失败，重新进行清氦流程
H50.00 BOOL  ; 复测夹爪有料记忆
H50.01 BOOL  ; 复测夹爪有OK料记忆
H50.02 BOOL  ; 复测夹爪有NG料记忆
H50.10 BOOL  ; OK配对#1位有料记忆
H50.11 BOOL  ; OK配对#2位有料记忆
H51.00 BOOL  ; 复测缓存左1位有料记忆（#1位）
H51.01 BOOL  ; 复测缓存右1位有料记忆（#2位）
H51.02 BOOL  ; 复测缓存左2位有料记忆（#1位）
H51.03 BOOL  ; 复测缓存右2位有料记忆（#2位）
H51.04 BOOL  ; 复测缓存左3位有料记忆（#1位）
H51.05 BOOL  ; 复测缓存右3位有料记忆（#2位）
H51.06 BOOL  ; 复测缓存左4位有料记忆（#1位）
H51.07 BOOL  ; 复测缓存右4位有料记忆（#2位）
H51.08 BOOL  ; 复测缓存总记忆
H54.00 BOOL  ; 复测移载伺服X轴回原点完成标志（1-完成）
H54.01 BOOL  ; 复测移载伺服Z轴回原点完成标志（1-完成）
H55.00 BOOL  ; 复测腔有料记忆
H55.01 BOOL  ; 复测腔有OK料记忆
H55.02 BOOL  ; 复测腔有NG料记忆
H55.03 BOOL  ; 复测腔测试完成记忆
H56.00 BOOL  ; 复检电池泄漏
H56.02 BOOL  ; 复检电池注氦超时
H56.04 BOOL  ; 复检腔体抽真空NG
H56.06 BOOL  ; 复检腔体氦检时腔体压力过高
H56.08 BOOL  ; 复测腔注氦超限
H57.00 BOOL  ; 复检腔体有清氦需求
H57.10 BOOL  ; 复检腔体清氦失败，重新进行清氦流程
H5.00 BOOL  ; 扫码屏蔽（SW）
H5.01 BOOL  ; 进料拉带重新扫码模式选择（0=使用/1=屏蔽）
H5.02 BOOL  ; 氦检仪屏蔽
H5.03 BOOL  ; 1#腔体屏蔽（0=使用）
H5.04 BOOL  ; 2#腔体屏蔽（0=使用）
H5.05 BOOL  ; 3#腔体屏蔽（0=使用）
H5.06 BOOL  ; 4#腔体屏蔽（0=使用）
H5.07 BOOL  ; 电脑屏蔽-HMI
H5.08 BOOL  ; 批次号判断屏蔽
H5.09 BOOL  ; 复测腔停用（1-停用）
H5.10 BOOL  ; 空跑程序
H5.12 BOOL  ; 氦气源压力检测屏蔽
H5.13 BOOL  ; 复测模式（0-关闭 1-打开）
H5.14 BOOL  ; 测试模式（0-双检 1-单检）
H5.15 BOOL  ; 腔体模式（0-正压 1-负压）
H6.00 BOOL  ; 清氦模式（0-使用 1-不使用）
H6.01 BOOL  ; 负压进行空腔清氦（1-使用）
H6.02 BOOL  ; 加速模式（1-开启）
H6.03 BOOL  ; 不带复测腔体（1-带）
H6.04 BOOL  ; 真空泵屏蔽（1-屏蔽）
H6.05 BOOL  ; 清氦时使用清氦抽气阀（1-使用）
H6.06 BOOL  ; 氦气回收机屏蔽（0-屏蔽）
H6.07 BOOL  ; 氦检完成后关闭氦检保护阀（1-氦检后关闭）
H6.08 BOOL  ; 注氦超限判断启用（1-启用）
H6.09 BOOL  ; 注氦下超限判断启用（1-启用）
T0000 BOOL  ; PLC上电延时100ms
T0001 BOOL  ; 手动模式延时
T0002 BOOL  ; 自动模式延时
T0003 BOOL  ; X轴绝对移动复位延时
T0004 BOOL  ; Y轴绝对移动复位延时
T0006 BOOL  ; 复位延时
T0007 BOOL  ; 自动停止完成延时
T0008 BOOL  ; 启动按钮按下1s延时
T0009 BOOL  ; 停止按钮按下延时
T0010 BOOL  ; Z轴绝对移动复位延时
T0011 BOOL  ; U轴绝对移动复位延时
T0015 BOOL  ; 扫码NG取料延时
T0016 BOOL  ; 检测NG料满取料延时
T0019 BOOL  ; 清料停止完成延时
T0020 BOOL  ; 设备待料状态延时（参考进料）
T0021 BOOL  ; 设备待料状态延时（参考出料）
T0022 BOOL  ; 蜂鸣器屏蔽时间
T0024 BOOL  ; 氦检仪真空阀打开安全判定延时
T0025 BOOL  ; 清氦保护阀2打开判定延时
T0030 BOOL  ; 腔体真空泵M1停机1分钟内禁止启动保护延时
T0031 BOOL  ; 氦检前置泵泵停机1分钟内禁止启动保护延时
T0032 BOOL  ; 腔体真空泵M2停机1分钟内禁止启动保护延时
T0033 BOOL  ; 1#先开挡板阀再开两通阀延时
T0034 BOOL  ; 1#先关两通阀再开挡板阀延时
T0035 BOOL  ; 2#先开挡板阀再开两通阀延时
T0036 BOOL  ; 2#先关两通阀再开挡板阀延时
T0037 BOOL  ; 3#先开挡板阀再开两通阀延时
T0038 BOOL  ; 3#先关两通阀再开挡板阀延时
T0039 BOOL  ; 4#先开挡板阀再开两通阀延时
T0040 BOOL  ; 4#先关两通阀再开挡板阀延时
T0041 BOOL  ; 5#先开挡板阀再开两通阀延时
T0042 BOOL  ; 5#先关两通阀再开挡板阀延时
T0045 BOOL  ; 进料#1扫码枪通信异常
T0046 BOOL  ; 进料#2扫码枪通信异常
T0047 BOOL  ; 氦检仪通信异常
T0048 BOOL  ; 氦检仪启动异常
T0049 BOOL  ; 初次上电氦检仪故障延时
T0050 BOOL  ; PC&PLC通讯心跳检测异常延时
T0051 BOOL  ; 真空泵关闭延时时间
T0054 BOOL  ; 氦检仪状态延时
T0062 BOOL  ; 进料伺服X轴故障报警延时
T0063 BOOL  ; 进料伺服Z轴故障报警延时
T0064 BOOL  ; 复测移载伺服X轴故障报警延时
T0065 BOOL  ; 复测移载伺服Z轴故障报警延时
T0072 BOOL  ; 出料伺服X轴故障报警延时
T0073 BOOL  ; 出料伺服Z轴故障报警延时
T0100 BOOL  ; #1扫码阻挡气缸缩回位报警延时
T0101 BOOL  ; #1扫码阻挡气缸伸出位报警延时
T0102 BOOL  ; #1隔离气缸缩回位报警延时
T0103 BOOL  ; #1隔离气缸伸出位报警延时
T0104 BOOL  ; #2扫码阻挡气缸缩回位报警延时
T0105 BOOL  ; #2扫码阻挡气缸伸出位报警延时
T0106 BOOL  ; #2隔离气缸缩回位报警延时
T0107 BOOL  ; #2隔离气缸伸出位 报警延时
T0108 BOOL  ; #1进料夹爪夹紧位报警延时
T0109 BOOL  ; #1进料夹爪松开位报警延时
T0110 BOOL  ; #2进料夹爪夹紧位报警延时
T0111 BOOL  ; #2进料夹爪松开位报警延时
T0112 BOOL  ; 进料夹爪变距气缸伸出位报警延时
T0113 BOOL  ; 进料夹爪变距气缸缩回位报警延时
T0114 BOOL  ; #1出料夹爪夹紧位报警延时
T0115 BOOL  ; #1出料夹爪松开位报警延时
T0116 BOOL  ; #2出料夹爪夹紧位报警延时
T0117 BOOL  ; #2出料夹爪松开位报警延时
T0118 BOOL  ; 出料夹爪变距气缸伸出位报警延时
T0119 BOOL  ; 出料夹爪变距气缸缩回位报警延时
T0120 BOOL  ; #1腔体平移一级气缸缩回位报警延时
T0121 BOOL  ; #1腔体平移一级气缸伸出位报警延时
T0122 BOOL  ; #1腔体平移二级气缸缩回位报警延时
T0123 BOOL  ; #1腔体平移二级气缸伸出位报警延时
T0124 BOOL  ; #1腔体顶伸气缸上升位报警延时
T0125 BOOL  ; #1腔体顶伸气缸下降位报警延时
T0126 BOOL  ; #1腔体氦检阀开到位报警延时
T0127 BOOL  ; #1腔体氦检阀关到位报警延时
T0128 BOOL  ; #1腔体有料感应1报警延时
T0129 BOOL  ; #1腔体有料感应2报警延时
T0130 BOOL  ; 0报警延时
T0131 BOOL  ; 0报警延时
T0132 BOOL  ; 0报警延时
T0133 BOOL  ; #2腔体平移一级气缸缩回位报警延时
T0134 BOOL  ; #2腔体平移一级气缸伸出位报警延时
T0135 BOOL  ; #2腔体平移二级气缸缩回位报警延时
T0136 BOOL  ; #2腔体平移二级气缸伸出位报警延时
T0137 BOOL  ; #2腔体顶伸气缸上升位报警延时
T0138 BOOL  ; #2腔体顶伸气缸下降位报警延时
T0139 BOOL  ; #2腔体氦检阀开到位报警延时
T0140 BOOL  ; #2腔体氦检阀关到位报警延时
T0141 BOOL  ; 2#腔体有料感应1报警延时
T0142 BOOL  ; 2#腔体有料感应2报警延时
T0143 BOOL  ; 0报警延时
T0144 BOOL  ; 0报警延时
T0145 BOOL  ; 0报警延时
T0146 BOOL  ; #3腔体平移一级气缸缩回位报警延时
T0147 BOOL  ; #3腔体平移一级气缸伸出位报警延时
T0148 BOOL  ; #3腔体平移二级气缸缩回位报警延时
T0149 BOOL  ; #3腔体平移二级气缸伸出位报警延时
T0150 BOOL  ; #3腔体顶伸气缸上升位报警延时
T0151 BOOL  ; #3腔体顶伸气缸下降位报警延时
T0152 BOOL  ; #3腔体氦检阀开到位报警延时
T0153 BOOL  ; #3腔体氦检阀关到位报警延时
T0154 BOOL  ; 氦检仪准备好了信号报警延时
T0155 BOOL  ; 氦检仪故障信号报警延时
T0156 BOOL  ; #3腔体有料感应1报警延时
T0157 BOOL  ; #3腔体有料感应2报警延时
T0158 BOOL  ; 0报警延时
T0159 BOOL  ; 进料伺服X轴准备好了信号报警延时
T0160 BOOL  ; 进料伺服X轴故障信号报警延时
T0161 BOOL  ; 进料伺服Z轴准备好了信号报警延时
T0162 BOOL  ; 进料伺服Z轴故障信号报警延时
T0163 BOOL  ; 0报警延时
T0164 BOOL  ; 出料伺服X轴准备好了信号报警延时
T0165 BOOL  ; 出料伺服X轴故障信号报警延时
T0166 BOOL  ; 出料伺服Z轴准备好了信号报警延时
T0167 BOOL  ; 出料伺服Z轴故障信号报警延时
T0168 BOOL  ; 0报警延时
T0169 BOOL  ; 腔体抽真空泵运行信号报警延时
T0170 BOOL  ; 腔体抽真空泵过载信号报警延时
T0171 BOOL  ; 氦检前置泵运行信号报警延时
T0172 BOOL  ; 氦检前置泵过载信号报警延时
T0173 BOOL  ; 启动按钮报警延时
T0174 BOOL  ; 停止按钮报警延时
T0175 BOOL  ; 复位按钮报警延时
T0176 BOOL  ; 急停按钮报警延时
T0177 BOOL  ; 手自动选择报警延时
T0178 BOOL  ; #1进料夹爪防下坠感应报警延时
T0179 BOOL  ; #2进料夹爪防下坠感应报警延时
T0180 BOOL  ; #1出料夹爪防下坠感应报警延时
T0181 BOOL  ; #2出料夹爪防下坠感应报警延时
T0182 BOOL  ; 0报警延时
T0183 BOOL  ; 进料对接输入报警延时
T0184 BOOL  ; 出料对接输入报警延时
T0185 BOOL  ; 0报警延时
T0186 BOOL  ; 0报警延时
T0187 BOOL  ; 设备总气压信号报警延时
T0188 BOOL  ; #1来料位有料感应报警延时
T0189 BOOL  ; #2来料位有料感应报警延时
T0190 BOOL  ; #1隔离位有料感应报警延时
T0191 BOOL  ; #2隔离位有料感应报警延时
T0192 BOOL  ; #1扫码位有料感应报警延时
T0193 BOOL  ; #2扫码位有料感应报警延时
T0194 BOOL  ; #1-1进料位有料感应报警延时
T0195 BOOL  ; #1-2进料位有料感应报警延时
T0196 BOOL  ; #2-1进料位有料感应报警延时
T0197 BOOL  ; #2-2进料位有料感应报警延时
T0198 BOOL  ; 进料夹爪柔性感应报警延时
T0199 BOOL  ; 出料夹爪柔性感应报警延时
T0200 BOOL  ; #1进料夹爪对应腔体有料感应报警延时
T0201 BOOL  ; #2进料夹爪对应腔体有料感应报警延时
T0202 BOOL  ; 扫码NG放料#1位有料感应报警延时
T0203 BOOL  ; 扫码NG放料#2位有料感应报警延时
T0204 BOOL  ; 扫码NG料满位有料感应报警延时
T0205 BOOL  ; 进料配对位有料感应报警延时
T0206 BOOL  ; 出料配对位有料感应报警延时
T0207 BOOL  ; 氦检NG放料#1位有料感应报警延时
T0208 BOOL  ; 氦检NG放料#2位有料感应报警延时
T0209 BOOL  ; 氦检NG料满位有料感应报警延时
T0210 BOOL  ; #1-1出料位有料感应报警延时
T0211 BOOL  ; #1-2出料位有料感应报警延时
T0212 BOOL  ; #2-1出料位有料感应报警延时
T0213 BOOL  ; #2-2出料位有料感应报警延时
T0214 BOOL  ; #1门磁开关报警延时
T0215 BOOL  ; #2门磁开关报警延时
T0216 BOOL  ; #3门磁开关报警延时
T0217 BOOL  ; #4门磁开关报警延时
T0218 BOOL  ; #5门磁开关报警延时
T0219 BOOL  ; #6门磁开关报警延时
T0220 BOOL  ; #7门磁开关报警延时
T0221 BOOL  ; #8门磁开关报警延时
T0222 BOOL  ; #9门磁开关报警延时
T0223 BOOL  ; #10门磁开关报警延时
T0224 BOOL  ; #11门磁开关报警延时
T0225 BOOL  ; #12门磁开关报警延时
T0226 BOOL  ; #13门磁开关报警延时
T0227 BOOL  ; #14门磁开关报警延时
T0280 BOOL  ; 进料扫码MES入站就绪通知&确认超时报警延时
T0281 BOOL  ; 出料伺服MES出站就绪通知&确认超时报警延时
T0282 BOOL  ; 出料#2爪MES出站就绪通知&确认超时报警延时
T0283 BOOL  ; 复测爪MES出站就绪通知&确认超时报警延时
T0308 BOOL  ; 进料伺服X轴正极限报警延时
T0309 BOOL  ; 进料伺服X轴负极限报警延时
T0310 BOOL  ; 进料伺服X轴原点报警延时
T0311 BOOL  ; 进料伺服Z轴正极限报警延时
T0312 BOOL  ; 进料伺服Z轴负极限报警延时
T0313 BOOL  ; 进料伺服Z轴原点报警延时
T0314 BOOL  ; 出料伺服X轴正极限报警延时
T0315 BOOL  ; 出料伺服X轴负极限报警延时
T0316 BOOL  ; 出料伺服X轴原点报警延时
T0317 BOOL  ; 出料伺服Z轴正极限报警延时
T0318 BOOL  ; 出料伺服Z轴负极限报警延时
T0319 BOOL  ; 出料伺服Z轴原点报警延时
T0324 BOOL  ; 氦检仪不在检漏状态[alm]
T0338 BOOL  ; 整机复位超时报警延时
T0339 BOOL  ; 进料拉带工站复位超时报警延时
T0340 BOOL  ; 整机复位超时报警延时
T0341 BOOL  ; 进料拉带工站复位超时报警延时
T0342 BOOL  ; 进料伺服工站复位超时报警延时
T0343 BOOL  ; #1氦检工站复位超时报警延时
T0344 BOOL  ; #2氦检工站复位超时报警延时
T0345 BOOL  ; #3氦检工站复位超时报警延时
T0346 BOOL  ; 出料伺服工站复位超时报警延时
T0348 BOOL  ; 复测移载机构工站复位超时
T0349 BOOL  ; 复测腔体机构工站复位超时
T0356 BOOL  ; #1来料位有料记忆报警延时
T0357 BOOL  ; #2来料位有料记忆报警延时
T0358 BOOL  ; #1隔离位有料记忆报警延时
T0359 BOOL  ; #2隔离位有料记忆报警延时
T0360 BOOL  ; #1扫码位有料记忆报警延时
T0361 BOOL  ; #2扫码位有料记忆报警延时
T0362 BOOL  ; #1进料位有料记忆报警延时
T0363 BOOL  ; #2进料位有料记忆报警延时
T0364 BOOL  ; #1进料夹爪有料记忆报警延时
T0365 BOOL  ; #2进料夹爪有料记忆报警延时
T0366 BOOL  ; #1出料夹爪有料记忆报警延时
T0367 BOOL  ; #2出料夹爪有料记忆报警延时
T0368 BOOL  ; #1-1腔体有料记忆报警延时
T0369 BOOL  ; #1-2腔体有料记忆报警延时
T0370 BOOL  ; #2-1腔体有料记忆报警延时
T0371 BOOL  ; #2-2腔体有料记忆报警延时
T0372 BOOL  ; #3-1腔体有料记忆报警延时
T0373 BOOL  ; #3-2腔体有料记忆报警延时
T0374 BOOL  ; 进料配对位有料记忆报警延时
T0375 BOOL  ; 出料配对位有料记忆报警延时
T0376 BOOL  ; #1出料位有料记忆报警延时
T0377 BOOL  ; #2出料位有料记忆报警延时
T0378 BOOL  ; 扫码NG放料位有料记忆报警延时
T0379 BOOL  ; 氦检NG拉带下料位有料记忆报警延时
T0383 BOOL  ; 进料拉带跟料报警延时
T0384 BOOL  ; #4腔体平移一级气缸缩回位报警延时
T0385 BOOL  ; #4腔体平移一级气缸伸出位报警延时
T0386 BOOL  ; #4腔体平移二级气缸缩回位报警延时
T0387 BOOL  ; #4腔体平移二级气缸伸出位报警延时
T0388 BOOL  ; #4腔体顶伸气缸上升位报警延时
T0389 BOOL  ; #4腔体顶伸气缸下降位报警延时
T0390 BOOL  ; #4腔体氦检阀开到位报警延时
T0391 BOOL  ; #4腔体氦检阀关到位报警延时
T0392 BOOL  ; 4#腔体有料感应1报警延时
T0393 BOOL  ; 4#腔体有料感应2报警延时
T0396 BOOL  ; 复测夹爪气缸夹紧位报警延时
T0397 BOOL  ; 复测夹爪气缸松开位报警延时
T0398 BOOL  ; 复检夹爪柔性感应报警延时
T0399 BOOL  ; 复测腔体移栽气缸缩回位报警延时
T0400 BOOL  ; 复测腔体移栽气缸伸出位报警延时
T0401 BOOL  ; 复测腔体顶升气缸缩回位报警延时
T0402 BOOL  ; 复测腔体顶升气缸伸出位报警延时
T0403 BOOL  ; 复测腔体氦检阀开到位报警延时
T0404 BOOL  ; 复测腔体氦检阀关到位报警延时
T0405 BOOL  ; 复测腔体感应有料感应报警延时
T0407 BOOL  ; 出料配对位有料感应2报警延时
T0414 BOOL  ; 测伺服X轴准备好信号报警延时
T0415 BOOL  ; 复测伺服X轴故障信号报警延时
T0416 BOOL  ; 复测伺服Z轴准备好信号报警延时
T0417 BOOL  ; 复测伺服Z轴故障信号报警延时
T0428 BOOL  ; 复测缓存拨料气缸缩回位报警延时
T0429 BOOL  ; 复测缓存拨料气缸伸出位报警延时
T0430 BOOL  ; 复测缓存顶升气缸缩回位报警延时
T0431 BOOL  ; 复测缓存顶升气缸伸出位报警延时
T0432 BOOL  ; 复测缓存#1有料感应1报警延时
T0433 BOOL  ; 复测缓存#1有料感应2报警延时
T0434 BOOL  ; 复测缓存#1有料感应3报警延时
T0435 BOOL  ; 复测缓存#1有料感应4报警延时
T0436 BOOL  ; 复测缓存#2有料感应1报警延时
T0437 BOOL  ; 复测缓存#2有料感应2报警延时
T0438 BOOL  ; 复测缓存#2有料感应3报警延时
T0439 BOOL  ; 复测缓存#2有料感应4报警延时
T0440 BOOL  ; #1腔体破真空阀开到位报警延时
T0441 BOOL  ; #1腔体破真空阀关到位报警延时
T0442 BOOL  ; #1腔体顶部吹气开到位报警延时
T0443 BOOL  ; #1腔体顶部吹气关到位报警延时
T0444 BOOL  ; #2腔体抽真空阀开到位报警延时
T0445 BOOL  ; #2腔体抽真空阀关到位报警延时
T0446 BOOL  ; #2-1腔体阀开到位报警延时
T0447 BOOL  ; #2-1腔体阀关到位报警延时
T0448 BOOL  ; #2-2腔体阀开到位报警延时
T0449 BOOL  ; #2-2腔体阀关到位报警延时
T0450 BOOL  ; #2腔体破真空阀开到位报警延时
T0451 BOOL  ; #2腔体破真空阀关到位报警延时
T0452 BOOL  ; #2腔体顶部吹气开到位报警延时
T0453 BOOL  ; #2腔体顶部吹气关到位报警延时
T0454 BOOL  ; #3腔体抽真空阀开到位报警延时
T0455 BOOL  ; #3腔体抽真空阀关到位报警延时
T0456 BOOL  ; #3-1腔体阀开到位报警延时
T0457 BOOL  ; #3-1腔体阀关到位报警延时
T0458 BOOL  ; #3-2腔体阀开到位报警延时
T0459 BOOL  ; #3-2腔体阀关到位报警延时
T0460 BOOL  ; #3腔体破真空阀开到位报警延时
T0461 BOOL  ; #3腔体破真空阀关到位报警延时
T0462 BOOL  ; #3腔体顶部吹气开到位报警延时
T0463 BOOL  ; #3腔体顶部吹气关到位报警延时
T0464 BOOL  ; #1-1电池抽真空阀开到位报警延时
T0465 BOOL  ; #1-1电池抽真空阀关到位报警延时
T0466 BOOL  ; #1-2电池抽真空阀开到位报警延时
T0467 BOOL  ; #1-2电池抽真空阀关到位报警延时
T0468 BOOL  ; #1-1电池注氦阀开到位报警延时
T0469 BOOL  ; #1-1电池注氦阀关到位报警延时
T0470 BOOL  ; 复测腔体破真空阀开到位报警延时
T0472 BOOL  ; #1-1电池破真空阀开到位报警延时
T0473 BOOL  ; #1-1电池破真空阀关到位报警延时
T0474 BOOL  ; #1-2电池破真空阀开到位报警延时
T0475 BOOL  ; #1-2电池破真空阀关到位报警延时
T0478 BOOL  ; 复测电池破真空阀开到位报警延时
T0480 BOOL  ; 复测夹爪有料记忆报警延时
T0484 BOOL  ; #2-1电池破真空阀开到位报警延时
T0485 BOOL  ; #2-1电池破真空阀关到位报警延时
T0486 BOOL  ; #2-2电池破真空阀开到位报警延时
T0487 BOOL  ; #2-2电池破真空阀关到位报警延时
T0496 BOOL  ; #3-1电池破真空阀开到位报警延时
T0497 BOOL  ; #3-1电池破真空阀关到位报警延时
T0498 BOOL  ; #3-2电池破真空阀开到位报警延时
T0499 BOOL  ; #3-2电池破真空阀关到位报警延时
T0500 BOOL  ; #1扫码阻挡气缸缩回延时[A]
T0501 BOOL  ; #1扫码阻挡气缸伸出延时[A]
T0502 BOOL  ; #1隔离气缸缩回延时[A]
T0503 BOOL  ; #1隔离气缸伸出延时[A]
T0504 BOOL  ; #2扫码阻挡气缸缩回延时[A]
T0505 BOOL  ; #2扫码阻挡气缸伸出延时[A]
T0506 BOOL  ; #2隔离气缸缩回延时[A]
T0507 BOOL  ; #2隔离气缸伸出延时[A]
T0508 BOOL  ; #1进料夹爪夹紧延时[A]
T0509 BOOL  ; #1进料夹爪松开延时[A]
T0510 BOOL  ; #2进料夹爪夹紧延时[A]
T0511 BOOL  ; #2进料夹爪松开延时[A]
T0512 BOOL  ; 进料夹爪变距气缸伸出延时[A]
T0513 BOOL  ; 进料夹爪变距气缸缩回延时[A]
T0514 BOOL  ; #1出料夹爪夹紧延时[A]
T0515 BOOL  ; #1出料夹爪松开延时[A]
T0516 BOOL  ; #2出料夹爪夹紧延时[A]
T0517 BOOL  ; #2出料夹爪松开延时[A]
T0518 BOOL  ; 出料夹爪变距气缸伸出延时[A]
T0519 BOOL  ; 出料夹爪变距气缸缩回延时[A]
T0520 BOOL  ; #1腔体平移一级气缸缩回延时[A]
T0521 BOOL  ; #1腔体平移一级气缸伸出延时[A]
T0522 BOOL  ; #1腔体平移二级气缸缩回延时[A]
T0523 BOOL  ; #1腔体平移二级气缸伸出延时[A]
T0524 BOOL  ; #1腔体顶伸气缸上升延时[A]
T0525 BOOL  ; #1腔体顶伸气缸下降延时[A]
T0526 BOOL  ; #1腔体氦检阀开延时[A]
T0527 BOOL  ; 清氦保护阀开1延时[A]
T0528 BOOL  ; #1腔体抽真空阀开延时[A]
T0529 BOOL  ; #1腔体破真空挡板阀开延时[A]
T0530 BOOL  ; 0延时[A]
T0531 BOOL  ; #1腔体破真空吹气阀开延时[A]
T0532 BOOL  ; #1腔体顶部吹气开延时[A]
T0533 BOOL  ; #2腔体平移一级气缸缩回延时[A]
T0534 BOOL  ; #2腔体平移一级气缸伸出延时[A]
T0535 BOOL  ; #2腔体平移二级气缸缩回延时[A]
T0536 BOOL  ; #2腔体平移二级气缸伸出延时[A]
T0537 BOOL  ; #2腔体顶伸气缸上升延时[A]
T0538 BOOL  ; #2腔体顶伸气缸下降延时[A]
T0539 BOOL  ; #2腔体氦检阀开延时[A]
T0540 BOOL  ; 清氦抽气阀开1延时[A]
T0541 BOOL  ; #2腔体抽真空阀开延时[A]
T0542 BOOL  ; #2腔体破真空挡板阀开延时[A]
T0543 BOOL  ; 0延时[A]
T0544 BOOL  ; #2腔体破真空吹气阀开延时[A]
T0545 BOOL  ; #2腔体顶部吹气开延时[A]
T0546 BOOL  ; #3腔体平移一级气缸缩回延时[A]
T0547 BOOL  ; #3腔体平移一级气缸伸出延时[A]
T0548 BOOL  ; #3腔体平移二级气缸缩回延时[A]
T0549 BOOL  ; #3腔体平移二级气缸伸出延时[A]
T0550 BOOL  ; #3腔体顶伸气缸上升延时[A]
T0551 BOOL  ; #3腔体顶伸气缸下降延时[A]
T0552 BOOL  ; #3腔体氦检阀开延时[A]
T0553 BOOL  ; 清氦保护阀开2 延时[A]
T0554 BOOL  ; #3腔体抽真空阀开延时[A]
T0555 BOOL  ; #3腔体破真空挡板阀开延时[A]
T0556 BOOL  ; 0延时[A]
T0557 BOOL  ; #3腔体破真空吹气阀开延时[A]
T0558 BOOL  ; #3腔体顶部吹气开延时[A]
T0559 BOOL  ; 进料伺服X轴使能延时[A]
T0560 BOOL  ; 进料伺服X轴故障复位延时[A]
T0561 BOOL  ; 进料伺服Z轴使能延时[A]
T0562 BOOL  ; 进料伺服Z轴故障复位延时[A]
T0563 BOOL  ; 进料伺服Z轴刹车延时[A]
T0564 BOOL  ; 出料伺服X轴使能延时[A]
T0565 BOOL  ; 出料伺服X轴故障复位延时[A]
T0566 BOOL  ; 出料伺服Z轴使能延时[A]
T0567 BOOL  ; 出料伺服Z轴故障复位延时[A]
T0568 BOOL  ; 出料伺服Z轴刹车延时[A]
T0569 BOOL  ; 腔体抽真空泵M1启动延时[A]
T0570 BOOL  ; 腔体抽真空泵M2启动延时[A]
T0571 BOOL  ; 氦检前置泵M3启动延时[A]
T0572 BOOL  ; 氦检仪供电延时[A]
T0573 BOOL  ; 启动按钮指示灯延时[A]
T0574 BOOL  ; 停止按钮指示灯延时[A]
T0575 BOOL  ; 复位按钮指示灯延时[A]
T0576 BOOL  ; 蜂鸣器延时[A]
T0577 BOOL  ; 三色灯（红）延时[A]
T0578 BOOL  ; 三色灯（绿）延时[A]
T0579 BOOL  ; 三色灯（黄）延时[A]
T0580 BOOL  ; 进料拉带电机1启动延时[A]
T0581 BOOL  ; 扫码NG拉带电机启动延时[A]
T0582 BOOL  ; 氦检NG拉带电机启动延时[A]
T0583 BOOL  ; 进料对接输出延时[A]
T0584 BOOL  ; 出料对接输出延时[A]
T0585 BOOL  ; 0延时[A]
T0586 BOOL  ; 0延时[A]
T0587 BOOL  ; #1腔体底部吹气开延时[A]
T0588 BOOL  ; #2腔体底部吹气开延时[A]
T0589 BOOL  ; #3腔体底部吹气开延时[A]
T0590 BOOL  ; #4腔体底部吹气开延时[A]
T0591 BOOL  ; 复测腔体底部吹气开延时[A]
T0592 BOOL  ; 复测缓存拨料气缸缩回位延时[A]
T0593 BOOL  ; 复测缓存拨料气缸伸出位延时[A]
T0594 BOOL  ; 复测缓存顶升气缸缩回位延时[A]
T0595 BOOL  ; 复测缓存顶升气缸伸出位延时[A]
T0596 BOOL  ; #4腔体平移一级气缸缩回延时[A]
T0597 BOOL  ; #4腔体平移一级气缸伸出延时[A]
T0598 BOOL  ; #4腔体平移二级气缸缩回延时[A]
T0599 BOOL  ; #4腔体平移二级气缸伸出延时[A]
T0600 BOOL  ; #4腔体顶伸气缸上升延时[A]
T0601 BOOL  ; #4腔体顶伸气缸下降延时[A]
T0602 BOOL  ; #4腔体氦检阀开延时[A]
T0603 BOOL  ; 清氦抽气阀开2延时[A]
T0604 BOOL  ; #4腔体抽真空阀开延时[A]
T0605 BOOL  ; #4腔体破真空挡板阀开延时[A]
T0606 BOOL  ; 0延时[A]
T0607 BOOL  ; #4腔体破真空吹气阀开延时[A]
T0608 BOOL  ; #4腔体顶部吹气开延时[A]
T0609 BOOL  ; 进料拉带电机2启动延时[A]
T0610 BOOL  ; 0延时[A]
T0611 BOOL  ; 复测夹爪气缸缩回位延时[A]
T0612 BOOL  ; 复测夹爪气缸伸出位延时[A]
T0613 BOOL  ; 复测腔体移栽气缸缩回位延时[A]
T0614 BOOL  ; 复测腔体移栽气缸伸出位延时[A]
T0615 BOOL  ; 复测腔体顶升气缸缩回位延时[A]
T0616 BOOL  ; 复测腔体顶升气缸伸出位延时[A]
T0617 BOOL  ; 复测腔体氦检阀开延时[A]
T0618 BOOL  ; 复测腔体抽真空阀开延时[A]
T0619 BOOL  ; 复测腔体破真空挡板阀开延时[A]
T0620 BOOL  ; 复测腔体破真空吹气阀开延时[A]
T0621 BOOL  ; 复测腔体顶部吹气开延时[A]
T0622 BOOL  ; 0延时[A]
T0623 BOOL  ; 复测伺服X轴使能延时[A]
T0624 BOOL  ; 复测伺服X轴故障复位延时[A]
T0625 BOOL  ; 复测伺服Z轴使能延时[A]
T0626 BOOL  ; 复测伺服Z轴故障复位延时[A]
T0627 BOOL  ; 复测伺服Z轴伺服刹车延时[A]
T0628 BOOL  ; #1-1电池抽真空阀开延时[A]
T0629 BOOL  ; #1-2电池抽真空阀开延时[A]
T0630 BOOL  ; #1-1电池注氦阀开延时[A]
T0631 BOOL  ; #1-2电池注氦阀开延时[A]
T0632 BOOL  ; #1-1电池破真空阀开延时[A]
T0633 BOOL  ; #1-2电池破真空阀开延时[A]
T0634 BOOL  ; #2-1电池抽真空阀开延时[A]
T0635 BOOL  ; #2-2电池抽真空阀开延时[A]
T0636 BOOL  ; #2-1电池注氦阀开延时[A]
T0637 BOOL  ; #2-2电池注氦阀开延时[A]
T0638 BOOL  ; #2-1电池破真空阀开延时[A]
T0639 BOOL  ; #2-2电池破真空阀开延时[A]
T0640 BOOL  ; #3-1电池抽真空阀开延时[A]
T0641 BOOL  ; #3-2电池抽真空阀开延时[A]
T0642 BOOL  ; #3-1电池注氦阀开延时[A]
T0643 BOOL  ; #3-2电池注氦阀开延时[A]
T0644 BOOL  ; #3-1电池破真空阀开延时[A]
T0645 BOOL  ; #3-2电池破真空阀开延时[A]
T0646 BOOL  ; #4-1电池抽真空阀开延时[A]
T0647 BOOL  ; #4-2电池抽真空阀开延时[A]
T0648 BOOL  ; #4-1电池注氦阀开延时[A]
T0649 BOOL  ; #4-2电池注氦阀开延时[A]
T0650 BOOL  ; #4-1电池破真空阀开延时[A]
T0651 BOOL  ; #4-2电池破真空阀开延时[A]
T0652 BOOL  ; 复测电池抽真空阀延时[A]
T0653 BOOL  ; 复测电池抽注氦阀延时[A]
T0654 BOOL  ; 复测电池破真空阀延时[A]
T0655 BOOL  ; 0延时[A]
T0656 BOOL  ; 0延时[A]
T0657 BOOL  ; 0延时[A]
T0658 BOOL  ; 0延时[A]
T0659 BOOL  ; 0延时[A]
T0686 BOOL  ; #1腔体氦检阀关延时[A]
T0687 BOOL  ; 氦检仪真空阀关延时[A]
T0688 BOOL  ; #1腔体抽真空阀关延时[A]
T0689 BOOL  ; #1-1腔体阀关延时[A]
T0690 BOOL  ; #1-2腔体阀关延时[A]
T0691 BOOL  ; #1腔体破真空阀关延时[A]
T0692 BOOL  ; #1腔体吹气阀关延时[A]
T0693 BOOL  ; 延时[A]
T0694 BOOL  ; 延时[A]
T0695 BOOL  ; 延时[A]
T0696 BOOL  ; 延时[A]
T0697 BOOL  ; #1扫码位有料延时延时[A]
T0698 BOOL  ; #2扫码位有料延时延时[A]
T0699 BOOL  ; #2腔体氦检阀关延时[A]
T0700 BOOL  ; 复检清洁阀关延时[A]
T0701 BOOL  ; #2腔体抽真空阀关延时[A]
T0702 BOOL  ; #2-1腔体阀关延时[A]
T0703 BOOL  ; #2-2腔体阀关延时[A]
T0704 BOOL  ; #2腔体破真空阀关延时[A]
T0705 BOOL  ; #2腔体吹气阀关延时[A]
T0706 BOOL  ; 0延时[A]
T0707 BOOL  ; 延时[A]
T0708 BOOL  ; 延时[A]
T0709 BOOL  ; 延时[A]
T0710 BOOL  ; 延时[A]
T0711 BOOL  ; 延时[A]
T0712 BOOL  ; #3腔体氦检阀关延时[A]
T0713 BOOL  ; 0延时[A]
T0714 BOOL  ; #3腔体抽真空阀关延时[A]
T0715 BOOL  ; #3-1腔体阀关延时[A]
T0716 BOOL  ; #3-2腔体阀关延时[A]
T0717 BOOL  ; #3腔体破真空阀关延时[A]
T0718 BOOL  ; #3腔体吹气阀关延时[A]
T0719 BOOL  ; 延时[A]
T0720 BOOL  ; 延时[A]
T0721 BOOL  ; 延时[A]
T0722 BOOL  ; 延时[A]
T0723 BOOL  ; 延时[A]
T0724 BOOL  ; 延时[A]
T0725 BOOL  ; 延时[A]
T0726 BOOL  ; 延时[A]
T0727 BOOL  ; 延时[A]
T0728 BOOL  ; 延时[A]
T0729 BOOL  ; 腔体抽真空泵M1停止延时[A]
T0730 BOOL  ; 腔体抽真空泵M2停止延时[A]
T0731 BOOL  ; 氦检前置泵停止延时[A]
T0732 BOOL  ; 氦检仪停电延时[A]
T0733 BOOL  ; 延时[A]
T0734 BOOL  ; 延时[A]
T0735 BOOL  ; 延时[A]
T0736 BOOL  ; 延时[A]
T0737 BOOL  ; 延时[A]
T0738 BOOL  ; 延时[A]
T0739 BOOL  ; 延时[A]
T0740 BOOL  ; 进料拉带电机停止延时[A]
T0741 BOOL  ; 扫码NG拉带电机停止延时[A]
T0742 BOOL  ; 氦检NG拉带电机停止延时[A]
T0743 BOOL  ; 0延时[A]
T0744 BOOL  ; 延时[A]
T0745 BOOL  ; 延时[A]
T0746 BOOL  ; 延时[A]
T0747 BOOL  ; 延时[A]
T0748 BOOL  ; 延时[A]
T0749 BOOL  ; 延时[A]
T0750 BOOL  ; 延时[A]
T0751 BOOL  ; 延时[A]
T0752 BOOL  ; 延时[A]
T0753 BOOL  ; 延时[A]
T0754 BOOL  ; 延时[A]
T0755 BOOL  ; 延时[A]
T0756 BOOL  ; #1-1电池抽真空阀关延时[A]
T0757 BOOL  ; #1-2电池抽真空阀关延时[A]
T0758 BOOL  ; #1-1电池注氦阀关延时[A]
T0759 BOOL  ; #1-2电池注氦阀关延时[A]
T0760 BOOL  ; #1-1电池破真空阀关延时[A]
T0761 BOOL  ; #1-2电池破真空阀关延时[A]
T0762 BOOL  ; #2-1电池抽真空阀关延时[A]
T0763 BOOL  ; #2-2电池抽真空阀关延时[A]
T0764 BOOL  ; #2-1电池注氦阀关延时[A]
T0765 BOOL  ; #2-2电池注氦阀关延时[A]
T0766 BOOL  ; #2-1电池破真空阀关延时[A]
T0767 BOOL  ; #2-2电池破真空阀关延时[A]
T0768 BOOL  ; #3-1电池抽真空阀关延时[A]
T0769 BOOL  ; #3-2电池抽真空阀关延时[A]
T0770 BOOL  ; #3-1电池注氦阀关延时[A]
T0771 BOOL  ; #3-2电池注氦阀关延时[A]
T0772 BOOL  ; #3-1电池破真空阀关延时[A]
T0773 BOOL  ; #3-2电池破真空阀关延时[A]
T0774 BOOL  ; #4-1电池抽真空阀关延时[A]
T0775 BOOL  ; #4-2电池抽真空阀关延时[A]
T0776 BOOL  ; #4-1电池注氦阀关延时[A]
T0777 BOOL  ; #4-2电池注氦阀关延时[A]
T0778 BOOL  ; #4-1电池破真空阀关延时[A]
T0779 BOOL  ; #4-2电池破真空阀关延时[A]
T0780 BOOL  ; 复测电池抽真空阀关延时[A]
T0781 BOOL  ; 复测电池抽注氦阀关延时[A]
T0782 BOOL  ; 复测电池破真空阀关延时[A]
T0783 BOOL  ; 复测腔体氦检阀关延时[A]
T0784 BOOL  ; 0延时[A]
T0785 BOOL  ; 复测腔体抽真空阀关延时[A]
T0786 BOOL  ; 复测腔体破真空阀关延时[A]
T0787 BOOL  ; 复测腔体破真空阀关延时[A]
T0788 BOOL  ; 复测腔体顶部吹气关延时[A]
T0795 BOOL  ; #1腔体吹气阀关（底部清洁）延时[A]
T0796 BOOL  ; #2腔体吹气阀关（底部清洁）延时[A]
T0797 BOOL  ; #3腔体吹气阀关（底部清洁）延时[A]
T0798 BOOL  ; #4腔体吹气阀关（底部清洁）延时[A]
T0799 BOOL  ; 复测腔体吹气阀关（底部清洁）延时[A]
T1000 BOOL  ; #1扫码阻挡气缸缩回位感应延时[0000.00]
T1001 BOOL  ; #1扫码阻挡气缸伸出位感应延时[0000.01]
T1002 BOOL  ; #1隔离气缸缩回位感应延时[0000.02]
T1003 BOOL  ; 0感应延时[0000.03]
T1004 BOOL  ; #2扫码阻挡气缸缩回位感应延时[0000.04]
T1005 BOOL  ; #2扫码阻挡气缸伸出位感应延时[0000.05]
T1006 BOOL  ; #2隔离气缸缩回位感应延时[0000.06]
T1007 BOOL  ; 0感应延时[0000.07]
T1008 BOOL  ; #1进料夹爪夹紧位感应延时[0000.08]
T1009 BOOL  ; #1进料夹爪松开位感应延时[0000.09]
T1010 BOOL  ; #2进料夹爪夹紧位感应延时[0000.10]
T1011 BOOL  ; #2进料夹爪松开位感应延时[0000.11]
T1012 BOOL  ; 进料夹爪变距气缸伸出位感应延时[0000.12]
T1013 BOOL  ; 进料夹爪变距气缸缩回位感应延时[0000.13]
T1014 BOOL  ; #1出料夹爪夹紧位感应延时[0000.14]
T1015 BOOL  ; #1出料夹爪松开位感应延时[0000.15]
T1016 BOOL  ; #2出料夹爪夹紧位感应延时[0001.00]
T1017 BOOL  ; #2出料夹爪松开位感应延时[0001.01]
T1018 BOOL  ; 出料夹爪变距气缸伸出位感应延时[0001.02]
T1019 BOOL  ; 出料夹爪变距气缸缩回位感应延时[0001.03]
T1020 BOOL  ; #1腔体平移一级气缸缩回位感应延时[0001.04]
T1021 BOOL  ; #1腔体平移一级气缸伸出位感应延时[0001.05]
T1022 BOOL  ; #1腔体平移二级气缸缩回位感应延时[0001.06]
T1023 BOOL  ; #1腔体平移二级气缸伸出位感应延时[0001.07]
T1024 BOOL  ; #1腔体顶伸气缸上升位感应延时[0001.08]
T1025 BOOL  ; #1腔体顶伸气缸下降位感应延时[0001.09]
T1026 BOOL  ; #1腔体氦检阀开到位感应延时[0001.10]
T1027 BOOL  ; #1腔体氦检阀关到位感应延时[0001.11]
T1028 BOOL  ; 0感应延时[0001.12]
T1029 BOOL  ; 0感应延时[0001.13]
T1030 BOOL  ; 0感应延时[0001.14]
T1031 BOOL  ; 0感应延时[0001.15]
T1032 BOOL  ; 0感应延时[0002.00]
T1033 BOOL  ; #2腔体平移一级气缸缩回位感应延时[0002.01]
T1034 BOOL  ; #2腔体平移一级气缸伸出位感应延时[0002.02]
T1035 BOOL  ; #2腔体平移二级气缸缩回位感应延时[0002.03]
T1036 BOOL  ; #2腔体平移二级气缸伸出位感应延时[0002.04]
T1037 BOOL  ; #2腔体顶伸气缸上升位感应延时[0002.05]
T1038 BOOL  ; #2腔体顶伸气缸下降位感应延时[0002.06]
T1039 BOOL  ; #2腔体氦检阀开到位感应延时[0002.07]
T1040 BOOL  ; #2腔体氦检阀关到位感应延时[0002.08]
T1041 BOOL  ; 0感应延时[0002.09]
T1042 BOOL  ; 0感应延时[0002.10]
T1043 BOOL  ; 0感应延时[0002.11]
T1044 BOOL  ; 0感应延时[0002.12]
T1045 BOOL  ; 0感应延时[0002.13]
T1046 BOOL  ; #3腔体平移一级气缸缩回位感应延时[0002.14]
T1047 BOOL  ; #3腔体平移一级气缸伸出位感应延时[0002.15]
T1048 BOOL  ; #3腔体平移二级气缸缩回位感应延时[0003.00]
T1049 BOOL  ; #3腔体平移二级气缸伸出位感应延时[0003.01]
T1050 BOOL  ; #3腔体顶伸气缸上升位感应延时[0003.02]
T1051 BOOL  ; #3腔体顶伸气缸下降位感应延时[0003.03]
T1052 BOOL  ; #3腔体氦检阀开到位感应延时[0003.04]
T1053 BOOL  ; #3腔体氦检阀关到位感应延时[0003.05]
T1054 BOOL  ; 氦检仪准备好了信号感应延时[0003.06]
T1055 BOOL  ; 氦检仪故障信号感应延时[0003.07]
T1056 BOOL  ; 0感应延时[0003.08]
T1057 BOOL  ; 0感应延时[0003.09]
T1058 BOOL  ; 0感应延时[0003.10]
T1059 BOOL  ; 进料伺服X轴准备好了信号感应延时[0003.11]
T1060 BOOL  ; 进料伺服X轴故障信号感应延时[0003.12]
T1061 BOOL  ; 进料伺服Z轴准备好了信号感应延时[0003.13]
T1062 BOOL  ; 进料伺服Z轴故障信号感应延时[0003.14]
T1063 BOOL  ; 0感应延时[0003.15]
T1064 BOOL  ; 出料伺服X轴准备好了信号感应延时[0004.00]
T1065 BOOL  ; 出料伺服X轴故障信号感应延时[0004.01]
T1066 BOOL  ; 出料伺服Z轴准备好了信号感应延时[0004.02]
T1067 BOOL  ; 出料伺服Z轴故障信号感应延时[0004.03]
T1068 BOOL  ; 0感应延时[0004.04]
T1069 BOOL  ; 腔体抽真空泵运行信号感应延时[0004.05]
T1070 BOOL  ; 腔体抽真空泵过载信号感应延时[0004.06]
T1071 BOOL  ; 氦检前置泵运行信号感应延时[0004.07]
T1072 BOOL  ; 氦检前置泵过载信号感应延时[0004.08]
T1073 BOOL  ; 启动按钮感应延时[0004.09]
T1074 BOOL  ; 停止按钮感应延时[0004.10]
T1075 BOOL  ; 复位按钮感应延时[0004.11]
T1076 BOOL  ; 急停按钮感应延时[0004.12]
T1077 BOOL  ; 手自动选择感应延时[0004.13]
T1078 BOOL  ; #1进料夹爪防下坠感应感应延时[0004.14]
T1079 BOOL  ; #2进料夹爪防下坠感应感应延时[0004.15]
T1080 BOOL  ; #1出料夹爪防下坠感应感应延时[0005.00]
T1081 BOOL  ; #2出料夹爪防下坠感应感应延时[0005.01]
T1082 BOOL  ; 0感应延时[0005.02]
T1083 BOOL  ; 进料对接输入感应延时[0005.03]
T1084 BOOL  ; 出料对接输入感应延时[0005.04]
T1085 BOOL  ; 0感应延时[0005.05]
T1086 BOOL  ; 0感应延时[0005.06]
T1087 BOOL  ; 设备总气压信号感应延时[0005.07]
T1088 BOOL  ; #1来料位有料感应感应延时[0005.08]
T1089 BOOL  ; #2来料位有料感应感应延时[0005.09]
T1090 BOOL  ; #1隔离位有料感应感应延时[0005.10]
T1091 BOOL  ; #2隔离位有料感应感应延时[0005.11]
T1092 BOOL  ; #1扫码位有料感应感应延时[0005.12]
T1093 BOOL  ; #2扫码位有料感应感应延时[0005.13]
T1094 BOOL  ; #1-1进料位有料感应感应延时[0005.14]
T1095 BOOL  ; #1-2进料位有料感应感应延时[0005.15]
T1096 BOOL  ; #2-1进料位有料感应感应延时[0006.00]
T1097 BOOL  ; #2-2进料位有料感应感应延时[0006.01]
T1098 BOOL  ; 进料夹爪柔性感应感应延时[0006.02]
T1099 BOOL  ; 出料夹爪柔性感应感应延时[0006.03]
T1100 BOOL  ; #1进料夹爪对应腔体有料感应感应延时[0006.04]
T1101 BOOL  ; #2进料夹爪对应腔体有料感应感应延时[0006.05]
T1102 BOOL  ; 扫码NG放料#1位有料感应感应延时[0006.06]
T1103 BOOL  ; 扫码NG放料#2位有料感应感应延时[0006.07]
T1104 BOOL  ; 扫码NG料满位有料感应感应延时[0006.08]
T1105 BOOL  ; 进料配对位有料感应感应延时[0006.09]
T1106 BOOL  ; 出料配对位有料感应感应延时[0006.10]
T1107 BOOL  ; 氦检NG放料#1位有料感应感应延时[0006.11]
T1108 BOOL  ; 氦检NG放料#2位有料感应感应延时[0006.12]
T1109 BOOL  ; 氦检NG料满位有料感应感应延时[0006.13]
T1110 BOOL  ; #1-1出料位有料感应感应延时[0006.14]
T1111 BOOL  ; #1-2出料位有料感应感应延时[0006.15]
T1112 BOOL  ; #2-1出料位有料感应感应延时[0007.00]
T1113 BOOL  ; #2-2出料位有料感应感应延时[0007.01]
T1114 BOOL  ; #1门磁开关感应延时[0007.02]
T1115 BOOL  ; #2门磁开关感应延时[0007.03]
T1116 BOOL  ; #3门磁开关感应延时[0007.04]
T1117 BOOL  ; #4门磁开关感应延时[0007.05]
T1118 BOOL  ; #5门磁开关感应延时[0007.06]
T1119 BOOL  ; #6门磁开关感应延时[0007.07]
T1120 BOOL  ; #7门磁开关感应延时[0007.08]
T1121 BOOL  ; #8门磁开关感应延时[0007.09]
T1122 BOOL  ; #9门磁开关感应延时[0007.10]
T1123 BOOL  ; #10门磁开关感应延时[0007.11]
T1124 BOOL  ; #11门磁开关感应延时[0007.12]
T1125 BOOL  ; #12门磁开关感应延时[0007.13]
T1126 BOOL  ; #13门磁开关感应延时[0007.14]
T1127 BOOL  ; #14门磁开关感应延时[0007.15]
T1163 BOOL  ; $?St$Bk?_#[193] / #1隔离气缸伸出位感应延时 / $?St$Bk?_#[193]
T1167 BOOL  ; $?St$Bk?_#[194] / #2隔离气缸伸出位感应延时 / $?St$Bk?_#[194]
T1220 BOOL  ; 进料伺服X轴停止延时
T1221 BOOL  ; 进料伺服Z轴停止延时
T1222 BOOL  ; 出料伺服X轴停止延时
T1223 BOOL  ; 出料伺服Z轴停止延时
T1224 BOOL  ; 复测移载伺服X轴停止延时
T1225 BOOL  ; 复测移载伺服Z轴停止延时
T1326 BOOL  ; 清氦保护阀2开到位感应延时[0000.06]
T1327 BOOL  ; 清氦保护阀2阀关到位感应延时[0000.07]
T1328 BOOL  ; 清氦抽真空阀2开到位感应延时[0000.08]
T1329 BOOL  ; 清氦抽真空阀2关到位感应延时[0000.09]
T1330 BOOL  ; 清氦保护阀1开到位感应延时[0000.10]
T1331 BOOL  ; 清氦保护阀1阀关到位感应延时[0000.11]
T1332 BOOL  ; 清氦抽真空阀1开到位感应延时[0000.12]
T1333 BOOL  ; 清氦抽真空阀1关到位感应延时[0000.13]
T1334 BOOL  ; #1腔体抽真空阀开到位感应延时
T1335 BOOL  ; #1腔体抽真空阀关到位感应延时
T1336 BOOL  ; #1-1腔体阀开到位感应延时
T1337 BOOL  ; #1-1腔体阀关到位感应延时
T1338 BOOL  ; #1-2腔体阀开到位感应延时
T1339 BOOL  ; #1-2腔体阀关到位感应延时
T1340 BOOL  ; #1腔体破真空阀开到位感应延时
T1341 BOOL  ; #1腔体破真空阀关到位感应延时
T1342 BOOL  ; #1腔体吹气阀开到位感应延时
T1343 BOOL  ; #1腔体吹气阀关到位感应延时
T1344 BOOL  ; #2腔体抽真空阀开到位感应延时
T1345 BOOL  ; #2腔体抽真空阀关到位感应延时
T1346 BOOL  ; #2-1腔体阀开到位感应延时
T1347 BOOL  ; #2-1腔体阀关到位感应延时
T1348 BOOL  ; #2-2腔体阀开到位感应延时
T1349 BOOL  ; #2-2腔体阀关到位感应延时
T1350 BOOL  ; #2腔体破真空阀开到位感应延时
T1351 BOOL  ; #2腔体破真空阀关到位感应延时
T1352 BOOL  ; #2腔体吹气阀开到位感应延时
T1353 BOOL  ; #2腔体吹气阀关到位感应延时
T1354 BOOL  ; #3腔体抽真空阀开到位感应延时
T1355 BOOL  ; #3腔体抽真空阀关到位感应延时
T1356 BOOL  ; #3-1腔体阀开到位感应延时
T1357 BOOL  ; #3-1腔体阀关到位感应延时
T1358 BOOL  ; #3-2腔体阀开到位感应延时
T1359 BOOL  ; #3-2腔体阀关到位感应延时
T1360 BOOL  ; #3腔体破真空阀开到位感应延时
T1361 BOOL  ; #3腔体破真空阀关到位感应延时
T1362 BOOL  ; #3腔体吹气阀开到位感应延时
T1363 BOOL  ; #3腔体吹气阀关到位感应延时
T1364 BOOL  ; #1-1电池抽真空阀开到位感应延时
T1365 BOOL  ; #1-1电池抽真空阀关到位感应延时
T1366 BOOL  ; #1-2电池抽真空阀开到位感应延时
T1367 BOOL  ; #1-2电池抽真空阀关到位感应延时
T1368 BOOL  ; #1-1电池注氦阀开到位感应延时
T1369 BOOL  ; #1-1电池注氦阀关到位感应延时
T1370 BOOL  ; #1-2电池注氦阀开到位感应延时
T1371 BOOL  ; #1-2电池注氦阀关到位感应延时
T1372 BOOL  ; #1-1电池破真空阀开到位感应延时
T1373 BOOL  ; #1-1电池破真空阀关到位感应延时
T1374 BOOL  ; #1-2电池破真空阀开到位感应延时
T1375 BOOL  ; #1-2电池破真空阀关到位感应延时
T1376 BOOL  ; #2-1电池抽真空阀开到位感应延时
T1377 BOOL  ; #2-1电池抽真空阀关到位感应延时
T1378 BOOL  ; #2-2电池抽真空阀开到位感应延时
T1379 BOOL  ; #2-2电池抽真空阀关到位感应延时
T1380 BOOL  ; #2-1电池注氦阀开到位感应延时
T1381 BOOL  ; #2-1电池注氦阀关到位感应延时
T1382 BOOL  ; #2-2电池注氦阀开到位感应延时
T1383 BOOL  ; #2-2电池注氦阀关到位感应延时
T1384 BOOL  ; #2-1电池破真空阀开到位感应延时
T1385 BOOL  ; #2-1电池破真空阀关到位感应延时
T1386 BOOL  ; #2-2电池破真空阀开到位感应延时
T1387 BOOL  ; #2-2电池破真空阀关到位感应延时
T1388 BOOL  ; #3-1电池抽真空阀开到位感应延时
T1389 BOOL  ; #3-1电池抽真空阀关到位感应延时
T1390 BOOL  ; #3-2电池抽真空阀开到位感应延时
T1391 BOOL  ; #3-2电池抽真空阀关到位感应延时
T1392 BOOL  ; #3-1电池注氦阀开到位感应延时
T1393 BOOL  ; #3-1电池注氦阀关到位感应延时
T1394 BOOL  ; #3-2电池注氦阀开到位感应延时
T1395 BOOL  ; #3-2电池注氦阀关到位感应延时
T1396 BOOL  ; #3-1电池破真空阀开到位感应延时
T1397 BOOL  ; #3-1电池破真空阀关到位感应延时
T1398 BOOL  ; #3-2电池破真空阀开到位感应延时
T1399 BOOL  ; #3-2电池破真空阀关到位感应延时
T1400 BOOL  ; #15门磁开关感应延时[0030.00]
T1401 BOOL  ; #16门磁开关感应延时[0030.01]
T1404 BOOL  ; #4腔体平移一级气缸缩回位感应延时[0030.04]
T1405 BOOL  ; #4腔体平移一级气缸伸出位感应延时[0030.05]
T1406 BOOL  ; #4腔体平移二级气缸缩回位感应延时[0030.06]
T1407 BOOL  ; #4腔体平移二级气缸伸出位感应延时[0030.07]
T1408 BOOL  ; #4腔体顶伸气缸上升位感应延时[0030.08]
T1409 BOOL  ; #4腔体顶伸气缸下降位感应延时[0030.09]
T1410 BOOL  ; #4腔体氦检阀开到位感应延时[0030.10]
T1411 BOOL  ; #4腔体氦检阀关到位感应延时[0030.11]
T1416 BOOL  ; 复测夹爪气缸夹紧位感应延时[0031.00]
T1417 BOOL  ; 复测夹爪气缸松开位感应延时[0031.01]
T1418 BOOL  ; 复检夹爪柔性感应感应延时[0031.02]
T1419 BOOL  ; 复测腔体移栽气缸缩回位感应延时[0031.03]
T1420 BOOL  ; 复测腔体移栽气缸伸出位感应延时[0031.04]
T1421 BOOL  ; 复测腔体顶升气缸缩回位感应延时[0031.05]
T1422 BOOL  ; 复测腔体顶升气缸伸出位感应延时[0031.06]
T1423 BOOL  ; 复测腔体氦检阀开到位感应延时[0031.07]
T1424 BOOL  ; 复测腔体氦检阀关到位感应延时[0031.08]
T1425 BOOL  ; 复测腔体感应有料感应感应延时[0031.09]
T1426 BOOL  ; 0感应延时[0031.10]
T1427 BOOL  ; 出料配对位有料感应2感应延时[0031.11]
T1428 BOOL  ; 0感应延时[0031.12]
T1429 BOOL  ; 0感应延时[0031.13]
T1430 BOOL  ; 0感应延时[0031.14]
T1431 BOOL  ; 0感应延时[0031.15]
T1432 BOOL  ; 腔体抽真空泵M2运行信号感应延时[0032.00]
T1433 BOOL  ; 腔体抽真空泵M2过载信号感应延时[0032.01]
T1434 BOOL  ; 测伺服X轴准备好信号感应延时[0032.02]
T1435 BOOL  ; 复测伺服X轴故障信号感应延时[0032.03]
T1436 BOOL  ; 复测伺服Z轴准备好信号感应延时[0032.04]
T1437 BOOL  ; 复测伺服Z轴故障信号感应延时[0032.05]
T1438 BOOL  ; 0感应延时[0032.06]
T1439 BOOL  ; 0感应延时[0032.07]
T1440 BOOL  ; 0感应延时[0032.08]
T1441 BOOL  ; 0感应延时[0032.09]
T1442 BOOL  ; 设备真空压力信号#1感应延时[0032.10]
T1443 BOOL  ; 设备真空压力信号#2感应延时[0032.11]
T1444 BOOL  ; 设备氦气压力信号#1感应延时[0032.12]
T1445 BOOL  ; 设备氦气压力信号#2感应延时[0032.13]
T1446 BOOL  ; 设备注氦压力调节阀#1感应延时[0032.14]
T1447 BOOL  ; 设备注氦压力调节阀#2感应延时[0032.15]
T1448 BOOL  ; 复测缓存拨料气缸缩回位感应延时[0033.00]
T1449 BOOL  ; 复测缓存拨料气缸伸出位感应延时[0033.01]
T1450 BOOL  ; 复测缓存顶升气缸缩回位感应延时[0033.02]
T1451 BOOL  ; 复测缓存顶升气缸伸出位感应延时[0033.03]
T1452 BOOL  ; 复测缓存#1有料感应1感应延时[0033.04]
T1453 BOOL  ; 复测缓存#1有料感应2感应延时[0033.05]
T1454 BOOL  ; 复测缓存#1有料感应3感应延时[0033.06]
T1455 BOOL  ; 复测缓存#1有料感应4感应延时[0033.07]
T1456 BOOL  ; 复测缓存#2有料感应1感应延时[0033.08]
T1457 BOOL  ; 复测缓存#2有料感应2感应延时[0033.09]
T1458 BOOL  ; 复测缓存#2有料感应3感应延时[0033.10]
T1459 BOOL  ; 复测缓存#2有料感应4感应延时[0033.11]
T1464 BOOL  ; #4腔体抽真空阀开到位感应延时[0000.00]
T1465 BOOL  ; #4腔体抽真空阀关到位感应延时[0000.01]
T1466 BOOL  ; #4-1腔体阀开到位感应延时[0000.02]
T1467 BOOL  ; #4-1腔体阀关到位感应延时[0000.03]
T1468 BOOL  ; #4-2腔体阀开到位感应延时[0000.04]
T1469 BOOL  ; #4-2腔体阀关到位感应延时[0000.05]
T1470 BOOL  ; #4腔体破真空阀开到位感应延时[0000.06]
T1471 BOOL  ; #4腔体破真空阀关到位感应延时[0000.07]
T1472 BOOL  ; #4腔体吹气阀开到位感应延时[0000.08]
T1473 BOOL  ; #4腔体吹气阀关到位感应延时[0000.09]
T1474 BOOL  ; #4-1电池抽真空阀开到位感应延时[0000.10]
T1475 BOOL  ; #4-1电池抽真空阀关到位感应延时[0000.11]
T1476 BOOL  ; #4-2电池抽真空阀开到位感应延时[0000.12]
T1477 BOOL  ; #4-2电池抽真空阀关到位感应延时[0000.13]
T1478 BOOL  ; #4-1电池注氦阀开到位感应延时[0000.14]
T1479 BOOL  ; #4-1电池注氦阀关到位感应延时[0000.15]
T1480 BOOL  ; #4-2电池注氦阀开到位感应延时[0000.00]
T1481 BOOL  ; #4-2电池注氦阀关到位感应延时[0000.01]
T1482 BOOL  ; #4-1电池破真空阀开到位感应延时[0000.02]
T1483 BOOL  ; #4-1电池破真空阀关到位感应延时[0000.03]
T1484 BOOL  ; #4-2电池破真空阀开到位感应延时[0000.04]
T1485 BOOL  ; #4-2电池破真空阀关到位感应延时[0000.05]
T1486 BOOL  ; 复测腔体抽真空阀开到位感应延时[0000.06]
T1487 BOOL  ; 复测腔体抽真空阀关到位感应延时[0000.07]
T1488 BOOL  ; #3腔体顶伸气缸上升位感应延时[0003.02]_1
T1489 BOOL  ; #3腔体顶伸气缸下降位感应延时[0003.03]_1
T1490 BOOL  ; 复测腔体破真空阀开到位感应延时[0000.10]
T1491 BOOL  ; 复测腔体破真空阀关到位感应延时[0000.11]
T1492 BOOL  ; 复测腔体吹气阀开到位感应延时[0000.12]
T1493 BOOL  ; 复测腔体吹气阀关到位感应延时[0000.13]
T1494 BOOL  ; 复测电池抽真空阀开到位感应延时[0000.14]
T1495 BOOL  ; 复测电池抽真空阀关到位感应延时[0000.15]
T1496 BOOL  ; 复测电池抽注氦阀开到位感应延时[0000.00]
T1497 BOOL  ; 复测电池抽注氦阀关到位感应延时[0000.01]
T1498 BOOL  ; 复测电池破真空阀开到位感应延时[0000.02]
T1499 BOOL  ; 复测电池破真空阀关到位感应延时[0000.03]
T1500 BOOL  ; 进料拉带机构开始运行条件延时
T1509 BOOL  ; 进料拉带机构复位完成延时
T1520 BOOL  ; 进料伺服机构开始运行条件1延时（进料拉带取料）
T1521 BOOL  ; 进料伺服机构开始运行条件2延时（扫码NG放料）
T1522 BOOL  ; 进料伺服机构开始运行条件3延时（扫码配对取/放料）
T1523 BOOL  ; 进料伺服机构开始运行条件4延时（腔体放料）
T1527 BOOL  ; 进料伺服X轴定位延时
T1528 BOOL  ; 进料伺服Z轴定位延时
T1529 BOOL  ; 进料伺服机构复位完成延时
T1530 BOOL  ; #1腔体机构开始运行条件延时(自动步)
T1531 BOOL  ; #1腔体机构数据初始化延时（自动步）
T1535 BOOL  ; #1腔体机构开始运行条件延时（自动单检步）
T1536 BOOL  ; #1腔体机构开始运行延时（清氦步）
T1539 BOOL  ; #1腔体机构复位完成延时
T1540 BOOL  ; 除#1氦检阀均关闭
T1542 BOOL  ; 真空屏蔽时#1腔5S默认到达抽真空阀值
T1550 BOOL  ; #2腔体机构开始运行条件延时(自动步)
T1551 BOOL  ; #2腔体机构数据初始化延时（自动步）
T1555 BOOL  ; #2腔体机构开始运行条件延时（自动单检步）
T1556 BOOL  ; #2腔体机构开始运行延时（清氦步）
T1559 BOOL  ; #2腔体机构复位完成延时
T1560 BOOL  ; 除#2氦检阀均关闭
T1562 BOOL  ; 真空屏蔽时#2腔5S默认到达抽真空阀值
T1570 BOOL  ; #3腔体机构开始运行条件延时(自动步)
T1571 BOOL  ; #3腔体机构数据初始化延时（自动步）
T1575 BOOL  ; #3腔体机构开始运行条件延时（自动单检步）
T1576 BOOL  ; #3腔体机构开始运行延时（清氦步）
T1579 BOOL  ; #3腔体机构复位完成延时
T1580 BOOL  ; 除#3氦检阀均关闭
T1582 BOOL  ; 真空屏蔽时#3腔5S默认到达抽真空阀值
T1590 BOOL  ; 出料夹爪初始状态
T1600 BOOL  ; 自动模式下X模组定位需求
T1601 BOOL  ; 自动模式下Z模组定位需求
T1602 BOOL  ; 下料模组初始化X轴到待机位
T1603 BOOL  ; 下料模组初始化z轴到待机位
T1604 BOOL  ; 出料Z模组归零触发延迟
T1605 BOOL  ; 出料X模组归零触发延迟
T1606 BOOL  ; 出料Z模组柔性报警处理延迟
T1607 BOOL  ; 手动跟踪Z模组联动
T1608 BOOL  ; 手动跟踪X模组联动
T1609 BOOL  ; 跟踪需求触发延迟
T1610 BOOL  ; #4腔体机构开始运行条件延时(自动步)
T1611 BOOL  ; #4腔体机构数据初始化延时（自动步）
T1615 BOOL  ; #4腔体机构开始运行条件延时（自动单检步）
T1616 BOOL  ; #4腔体机构开始运行延时（清氦步）
T1619 BOOL  ; #4腔体机构复位完成延时
T1620 BOOL  ; 除#4氦检阀均关闭
T1622 BOOL  ; 真空屏蔽时#4腔5S默认到达抽真空阀值
T1630 BOOL  ; 复测移栽机构：取/放待测料开始运行延时
T1631 BOOL  ; 复测移栽机构：取/放已测料开始运行延时
T1632 BOOL  ; 复测移栽机构：缓存开始运行延时
T1649 BOOL  ; 氦检移栽机构：在初始位延时
T1650 BOOL  ; 复检腔体机构：开始运行条件延时(自动步)
T1656 BOOL  ; 复检腔体机构：开始运行延时（清氦步）
T1658 BOOL  ; 下料Z轴手动下降前安全判断失败延时
T1659 BOOL  ; 复测移载机构：正常腔体待料条件延时(启动复测)
T1660 BOOL  ; 除复检腔氦检阀全部关闭
T1662 BOOL  ; 真空屏蔽时复测腔5S默认到达抽真空阀值
T1669 BOOL  ; 复检腔体机构：初始位延时
T1700 BOOL  ; 扫码数据初始化延时
T1701 BOOL  ; 扫码触发前延时
T1720 BOOL  ; #1出料夹爪有料出站就绪通知延时
T1721 BOOL  ; #2出料夹爪有料出站就绪通知延时
T1900 BOOL  ; #1-1腔体抽真空阈值到达延时（测试）
T1901 BOOL  ; #1-1腔体抽真空时间上限到达延时（测试）
T1902 BOOL  ; #1-1腔体破真空阈值到达延时（测试）
T1904 BOOL  ; #1-1腔体氦检时间（测试）
T1905 BOOL  ; #1-1腔体抽气阀关闭延时（测试）
